FUNCTION_BLOCK "FB32_AXIS"   // FB32, LAD
{ S7_Optimized_Access := 'FALSE' }
AUTHOR : ETXETAR
VERSION : 1.0
// stored: AutoNumber false, IsIECCheckEnabled false, SetENOAutomatically false, UDAEnableTagReadback false
   VAR_INPUT
      OPTIONS_0 : Byte := 2#0000_0000;   // OPTIONS 0
      OPTIONS_1 : Byte := 2#0000_0000;   // OPTIONS 1
      SAFETY_BYPASS : Bool;   // MUST BE ALWAYS OFF, ACTIVATE ONLY FOR TEST
      OPTIMIZATION_BYPASS : Bool;   // MUST BE ALWAYS OFF, ACTIVATE ONLY FOR OPTIMIZATION TEST
      AX_ENABLE : Bool;   // AXIS ENABLE
      TEST_STOP_BRAKE_TEST_AX_NUM : Bool;   // TEST STOP BRAKE TEST AXIS NUMBER
      PARAMETER_SET_0 : Bool;   // PARAMETER SET [0] SELECTION
      PARAMETER_SET_1 : Bool;   // PARAMETER SET [1] SELECTION
      PARAMETER_SET_2 : Bool;   // PARAMETER SET [2] SELECTION
      PARAMETER_SET_3 : Bool;   // PARAMETER SET [3] SELECTION
      MOVE_AXIS : Bool;   // MOVE AXIS INPUT
      SAFE_ENABLED : Bool;   // SAFE ENABLED
      FEED_HOLD_COND : Bool;   // FEED HOLD CONDITIONS INPUT
      AX_TORQUE_ENABLE : Bool;   // AXIS TORQUE ENABLE
      MPP_AXIS_SELECTED : Bool;   // MPP AXIS SELECTED
      HMI_AXIS_SELECTED : Bool;   // HMI AXIS SELECTED
      HMI_REQ_LINE : Bool;   // HMI REQUEST LINE
      JOG_MINUS_REQ_NOT_FC18 : Bool;   // JOG MINUS REQUEST NOT FC18, THIS LINE MOVES THE AXIS WITHOUT FC18
      JOG_PLUS_REQ_NOT_FC18 : Bool;   // JOG PLUS REQUEST NOT FC18, THIS LINE MOVES THE AXIS WITHOUT FC18
      JOG_MINUS_REQ_FC18 : Bool;   // JOG MINUS REQUEST FOR FC18, THIS LINE MOVES THE AXIS WITH FC18
      JOG_PLUS_REQ_FC18 : Bool;   // JOG PLUS REQUEST FOR FC18, THIS LINE MOVES THE AXIS WITH FC18
      FC18_EXTERNAL_POS : Real;   // FC18 EXTERNAL POSITION
      AUTO_RETURN_COMMAND : Bool;   // AUTO RETURN COMMAND
      AUTO_ADVANCE_COMMAND : Bool;   // AUTO ADVANCE COMMAND
      DELETE_DISTANCE_TO_GO : Bool;   // DELETE DISTANCE TO GO CONDITIONS
      FEED_OVERRIDE : Byte;   // FEED OVERRIDE
      FEED_OVER_ACTIVE : Bool;   // FEED OVER ACTIVE
      READ_POS : DWord;   // READ POSITION
      UNIT_ALARM : UInt;   // UNIT NUMBER MIN. NUMBER=1 MAX. NUMBER=4
      STATION_ALARM : UInt;   // STATION NUMBER MIN. NUMBER=0 MAX. NUMBER=4
   END_VAR
   VAR_OUTPUT
      MOTOR_ACTIVE : Bool;   // MOTOR ACTIVE
      MOVE_AX : Bool;   // MOVE AXIS
      FEED_HOLD_CONDITIONS : Bool;   // FEED HOLD CONDITIONS
      ACTIVE_PARAMETER_SET : Byte;   // ACTIVE PARAMETER SET
      AX_NOT_REFERENCE_ALM : Bool;   // AXIS NOT REFERENCE / AXIS NOT REFERENCED ALARM
      AX_B_NOT_IN_PST_180_90_ALM : Bool;   // AXIS B NO IN POSITION 180º-90ª / AXIS B NOT IN PST 180 90 ALARM
      MAST_SLAVE_MODE_NOT_ACTIV_ALM : Bool;   // MASTER SLAVE MODE NOT ACTIVE ALARM
      AX_TORQUE_EXCEEDED_ALM : Bool;   // AXIS TORQUE EXCEEDED ALARM
      AXIS_POS : Real;   // AXIS POSITION
      HMI_MOTION_EXECUTABILITY_LEFT : Bool;   // HMI MOTION EXECUTABILITY LEFT
      HMI_MOTION_EXECUTABILITY_RIGHT : Bool;   // HMI MOTION EXECUTABILITY RIGHT
      HMI_MOTION_END_POS_LEFT : Bool;   // HMI MOTION END POSITION LEFT
      HMI_MOTION_END_POS_RIGHT : Bool;   // HMI MOTION END POSITION RIGHT
      HMI_MOTION_ACTIVE_LEFT : Bool;   // HMI MOTION ACTIVE LEFT
      HMI_MOTION_ACTIVE_RIGHT : Bool;   // HMI MOTION ACTIVE RIGHT
   END_VAR
   VAR_IN_OUT
      AxisDB : "LBP_typeAxisX";
   END_VAR
   VAR DB_SPECIFIC
      AXIS { S7_SetPoint := 'True'} : "AXIS";
      TIMER_PULSES_ENABLE { S7_SetPoint := 'True'} : TOF_TIME;
   END_VAR
   VAR
      SAFETY_POSITIONS { S7_SetPoint := 'True'} : "FB33_SAFETY_POSITIONS";
   END_VAR
   VAR_TEMP
      INPUTS_MASK : Byte;   // INPUT MASK
      O_BYTE_0 : Struct   // OPTIONS BYTE 0
         MEASURING_SYSTEM_2 : Bool;   // MEASURING SYSTEM 2 OPTION / ALWAYS ON OR ALWAYS OFF
         ENABLE_FC18 : Bool;   // ENABLE FC18 OPTION
         FC18_EXTERNAL_POSITION : Bool;   // FC18 EXTERNAL POSITION OPTION
         AXIS_B_ENABLE_FAULTS : Bool;   // AXIS B ENABLE FAULTS OPTION
         SPARE_4 : Bool;   // SPARE OPTION
         SPARE_5 : Bool;   // SPARE OPTION
         SPARE_6 : Bool;   // SPARE OPTION
         SPARE_7 : Bool;   // SPARE OPTION
      END_STRUCT;
      O_BYTE_1 : Struct   // OPTIONS BYTE 0
         AXIS_ROLLER : Bool;   // AXIS ROLLER OPTION / ALWAYS ON OR ALWAYS OFF
         MASTER_AXIS : Bool;   // MASTER AXIS OPTION
         SLAVE_AXIS : Bool;   // SLAVE AXIS OPTION
         MASTER_SLAVE_INDPNDNT_HT10 : Bool;   // MASTER SLAVE INDEPENDENT MOVEMENT HT10 OPTION
         GANTRY_MODE_MASTER_AXIS : Bool;   // GANTRY MODE MASTER AXIS OPTION
         SPARE_5 : Bool;   // SPARE OPTION
         SPARE_6 : Bool;   // SPARE OPTION
         SPARE_7 : Bool;   // SPARE OPTION
      END_STRUCT;
      FC18_STATE : Byte;   // FC 18 STATE
      DB_NUMBER : DInt;   // DB NUMBER FOR ALARMS AND HELP DECODING
      AXIS_NUMBER_FC18 : Int;   // AXIS NUMBER FC18
   END_VAR
   // TIMER_PULSES_ENABLE.PT := T#1s;
   VAR_TEMP   // added for the SCL form of the ladder/FBD networks
      _w1 : Bool;
      _w2 : Bool;
      _w3 : Bool;
      _w4 : Bool;
      _w5 : Bool;
      _w6 : Bool;
      _w7 : Bool;
      _w8 : Bool;
      _w9 : Bool;
      _w10 : Bool;
      _w11 : Bool;
      _w12 : Bool;
      _w13 : Bool;
      _w14 : Bool;
      _w15 : Bool;
   END_VAR
BEGIN

NETWORK
TITLE = READ INSTANCE DB
//READ DB NUMBER
      L     DINO;
      +     10#800000;
      T     #DB_NUMBER;
//READ AXIS NUMBER
      L     DINO;
      L     10#130;
      -I;
      T     #AXIS_NUMBER_FC18;


REGION Network 2: OPTIONS
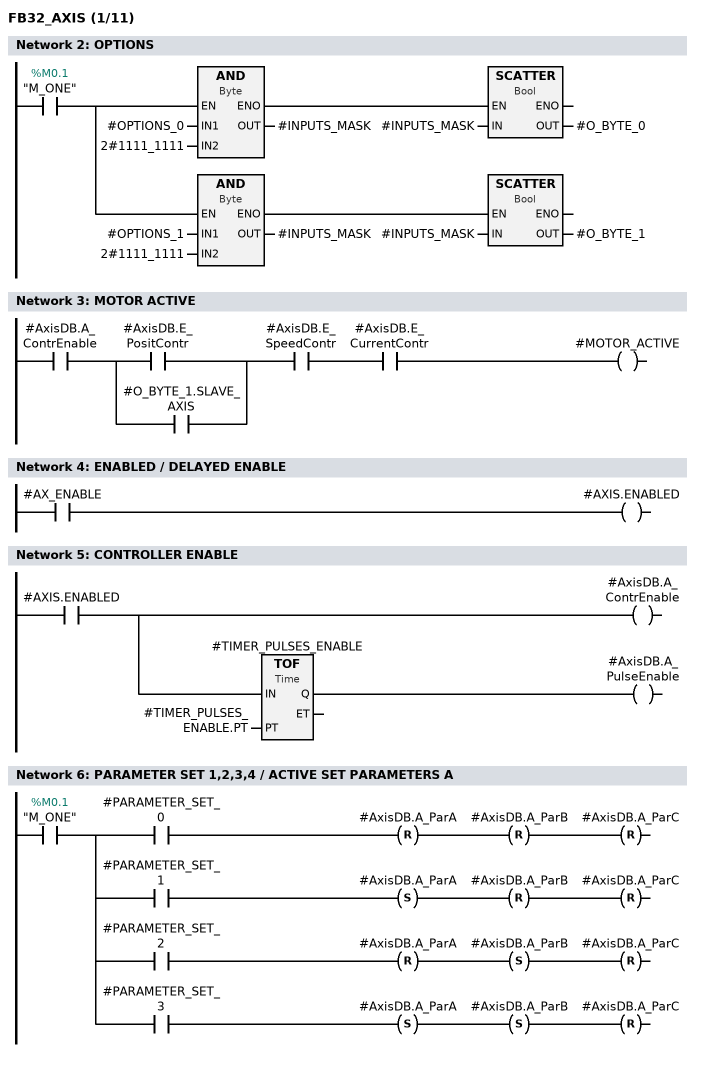
   RUNG wire#powerrail
      Contact( "M_ONE" )
      wire#w1
      { S7_Templates := "SrcType := Byte"; S7_GenerateENO := "TRUE" } And(in1 := #OPTIONS_0, in2 := 2#1111_1111, out => #INPUTS_MASK)
      { S7_Templates := "[dest_type := Bool, src_type := Byte]" } SCATTER(IN := #INPUTS_MASK, OUT => #O_BYTE_0)
   END_RUNG
   RUNG wire#w1
      { S7_Templates := "SrcType := Byte"; S7_GenerateENO := "TRUE" } And(in1 := #OPTIONS_1, in2 := 2#1111_1111, out => #INPUTS_MASK)
      { S7_Templates := "[dest_type := Bool, src_type := Byte]" } SCATTER(IN := #INPUTS_MASK, OUT => #O_BYTE_1)
   END_RUNG
   // the same network as SCL:
   IF "M_ONE" THEN #INPUTS_MASK := #OPTIONS_0 AND 2#1111_1111; END_IF;
   #_w1 := "M_ONE";
   IF #_w1 THEN
       SCATTER(IN := #INPUTS_MASK, OUT => #O_BYTE_0);
       #INPUTS_MASK := #OPTIONS_1 AND 2#1111_1111;
       SCATTER(IN := #INPUTS_MASK, OUT => #O_BYTE_1);
   END_IF;
END_REGION

REGION Network 3: MOTOR ACTIVE
   RUNG wire#powerrail
      Contact( #AxisDB.A_ContrEnable )
      wire#w1
      Contact( #AxisDB.E_PositContr )
      wire#w2
      Contact( #AxisDB.E_SpeedContr )
      Contact( #AxisDB.E_CurrentContr )
      Coil( #MOTOR_ACTIVE )
   END_RUNG
   RUNG wire#w1
      Contact( #O_BYTE_1.SLAVE_AXIS )
   END_RUNG wire#w2
   // the same network as SCL:
   #MOTOR_ACTIVE := #AxisDB.A_ContrEnable AND (#AxisDB.E_PositContr OR #O_BYTE_1.SLAVE_AXIS) AND #AxisDB.E_SpeedContr AND #AxisDB.E_CurrentContr;
END_REGION

REGION Network 4: ENABLED / DELAYED ENABLE
   RUNG wire#powerrail
      Contact( #AX_ENABLE )
      Coil( #AXIS.ENABLED )
   END_RUNG
   // the same network as SCL:
   #AXIS.ENABLED := #AX_ENABLE;
END_REGION

REGION Network 5: CONTROLLER ENABLE
   RUNG wire#powerrail
      Contact( #AXIS.ENABLED )
      wire#w1
      Coil( #AxisDB.A_ContrEnable )
   END_RUNG
   RUNG wire#w1
      { S7_Templates := "time_type := Time" } #TIMER_PULSES_ENABLE.TOF(pt := #TIMER_PULSES_ENABLE.PT, et =>)
      Coil( #AxisDB.A_PulseEnable )
   END_RUNG
   // the same network as SCL:
   #AxisDB.A_ContrEnable := #AXIS.ENABLED;
   #TIMER_PULSES_ENABLE(IN := #AXIS.ENABLED, PT := #TIMER_PULSES_ENABLE.PT);   // TOF
   #AxisDB.A_PulseEnable := #TIMER_PULSES_ENABLE.Q;
END_REGION

REGION Network 6: PARAMETER SET 1,2,3,4 / ACTIVE SET PARAMETERS A
   RUNG wire#powerrail
      Contact( "M_ONE" )
      wire#w1
      Contact( #PARAMETER_SET_0 )
      R_Coil( #AxisDB.A_ParA )
      R_Coil( #AxisDB.A_ParB )
      R_Coil( #AxisDB.A_ParC )
   END_RUNG
   RUNG wire#w1
      Contact( #PARAMETER_SET_1 )
      S_Coil( #AxisDB.A_ParA )
      R_Coil( #AxisDB.A_ParB )
      R_Coil( #AxisDB.A_ParC )
   END_RUNG
   RUNG wire#w1
      Contact( #PARAMETER_SET_2 )
      R_Coil( #AxisDB.A_ParA )
      S_Coil( #AxisDB.A_ParB )
      R_Coil( #AxisDB.A_ParC )
   END_RUNG
   RUNG wire#w1
      Contact( #PARAMETER_SET_3 )
      S_Coil( #AxisDB.A_ParA )
      S_Coil( #AxisDB.A_ParB )
      R_Coil( #AxisDB.A_ParC )
   END_RUNG
   // the same network as SCL:
   IF "M_ONE" AND #PARAMETER_SET_0 THEN
       #AxisDB.A_ParA := FALSE;
       #AxisDB.A_ParB := FALSE;
       #AxisDB.A_ParC := FALSE;
   END_IF;
   IF "M_ONE" AND #PARAMETER_SET_1 THEN
       #AxisDB.A_ParA := TRUE;
       #AxisDB.A_ParB := FALSE;
       #AxisDB.A_ParC := FALSE;
   END_IF;
   IF "M_ONE" AND #PARAMETER_SET_2 THEN
       #AxisDB.A_ParA := FALSE;
       #AxisDB.A_ParB := TRUE;
       #AxisDB.A_ParC := FALSE;
   END_IF;
   IF "M_ONE" AND #PARAMETER_SET_3 THEN
       #AxisDB.A_ParA := TRUE;
       #AxisDB.A_ParB := TRUE;
       #AxisDB.A_ParC := FALSE;
   END_IF;
END_REGION

REGION Network 7: ACTIVE PARAMETER SET 1,2,3,4
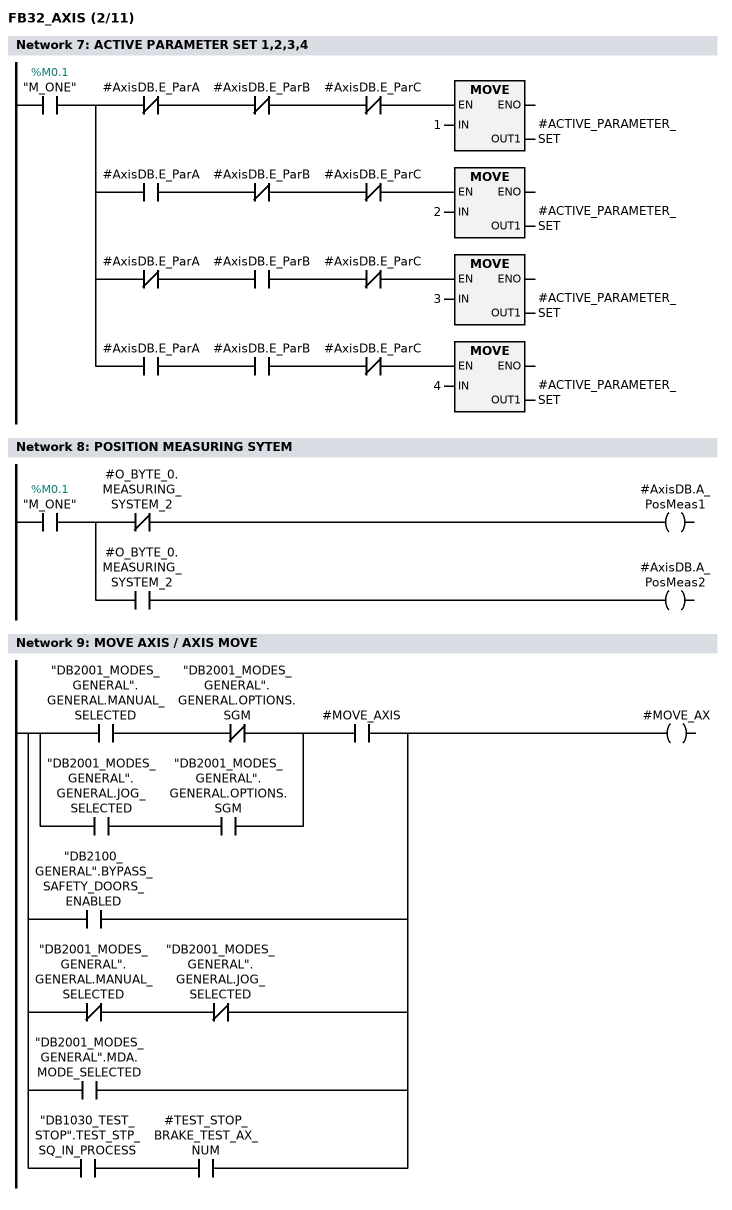
   RUNG wire#powerrail
      Contact( "M_ONE" )
      wire#w1
      I_Contact( #AxisDB.E_ParA )
      I_Contact( #AxisDB.E_ParB )
      I_Contact( #AxisDB.E_ParC )
      Move(in := 1, out1 => #ACTIVE_PARAMETER_SET)
   END_RUNG
   RUNG wire#w1
      Contact( #AxisDB.E_ParA )
      I_Contact( #AxisDB.E_ParB )
      I_Contact( #AxisDB.E_ParC )
      Move(in := 2, out1 => #ACTIVE_PARAMETER_SET)
   END_RUNG
   RUNG wire#w1
      I_Contact( #AxisDB.E_ParA )
      Contact( #AxisDB.E_ParB )
      I_Contact( #AxisDB.E_ParC )
      Move(in := 3, out1 => #ACTIVE_PARAMETER_SET)
   END_RUNG
   RUNG wire#w1
      Contact( #AxisDB.E_ParA )
      Contact( #AxisDB.E_ParB )
      I_Contact( #AxisDB.E_ParC )
      Move(in := 4, out1 => #ACTIVE_PARAMETER_SET)
   END_RUNG
   // the same network as SCL:
   IF "M_ONE" AND NOT #AxisDB.E_ParA AND NOT #AxisDB.E_ParB AND NOT #AxisDB.E_ParC THEN
       #ACTIVE_PARAMETER_SET := 1;
   END_IF;
   IF "M_ONE" AND #AxisDB.E_ParA AND NOT #AxisDB.E_ParB AND NOT #AxisDB.E_ParC THEN
       #ACTIVE_PARAMETER_SET := 2;
   END_IF;
   IF "M_ONE" AND NOT #AxisDB.E_ParA AND #AxisDB.E_ParB AND NOT #AxisDB.E_ParC THEN
       #ACTIVE_PARAMETER_SET := 3;
   END_IF;
   IF "M_ONE" AND #AxisDB.E_ParA AND #AxisDB.E_ParB AND NOT #AxisDB.E_ParC THEN
       #ACTIVE_PARAMETER_SET := 4;
   END_IF;
END_REGION

REGION Network 8: POSITION MEASURING SYTEM
   RUNG wire#powerrail
      Contact( "M_ONE" )
      wire#w1
      I_Contact( #O_BYTE_0.MEASURING_SYSTEM_2 )
      Coil( #AxisDB.A_PosMeas1 )
   END_RUNG
   RUNG wire#w1
      Contact( #O_BYTE_0.MEASURING_SYSTEM_2 )
      Coil( #AxisDB.A_PosMeas2 )
   END_RUNG
   // the same network as SCL:
   #AxisDB.A_PosMeas1 := "M_ONE" AND NOT #O_BYTE_0.MEASURING_SYSTEM_2;
   #AxisDB.A_PosMeas2 := "M_ONE" AND #O_BYTE_0.MEASURING_SYSTEM_2;
END_REGION

REGION Network 9: MOVE AXIS / AXIS MOVE
   RUNG wire#powerrail
      Contact( "DB2001_MODES_GENERAL".GENERAL.MANUAL_SELECTED )
      I_Contact( "DB2001_MODES_GENERAL".GENERAL.OPTIONS.SGM )
      wire#w1
      Contact( #MOVE_AXIS )
      wire#w2
      Coil( #MOVE_AX )
   END_RUNG
   RUNG wire#powerrail
      Contact( "DB2001_MODES_GENERAL".GENERAL.JOG_SELECTED )
      Contact( "DB2001_MODES_GENERAL".GENERAL.OPTIONS.SGM )
   END_RUNG wire#w1
   RUNG wire#powerrail
      Contact( "DB2100_GENERAL".BYPASS_SAFETY_DOORS_ENABLED )
   END_RUNG wire#w2
   RUNG wire#powerrail
      I_Contact( "DB2001_MODES_GENERAL".GENERAL.MANUAL_SELECTED )
      I_Contact( "DB2001_MODES_GENERAL".GENERAL.JOG_SELECTED )
   END_RUNG wire#w2
   RUNG wire#powerrail
      Contact( "DB2001_MODES_GENERAL".MDA.MODE_SELECTED )
   END_RUNG wire#w2
   RUNG wire#powerrail
      Contact( "DB1030_TEST_STOP".TEST_STP_SQ_IN_PROCESS )
      Contact( #TEST_STOP_BRAKE_TEST_AX_NUM )
   END_RUNG wire#w2
   // the same network as SCL:
   #MOVE_AX := ((("DB2001_MODES_GENERAL".GENERAL.MANUAL_SELECTED AND NOT "DB2001_MODES_GENERAL".GENERAL.OPTIONS.SGM) OR ("DB2001_MODES_GENERAL".GENERAL.JOG_SELECTED AND "DB2001_MODES_GENERAL".GENERAL.OPTIONS.SGM)) AND #MOVE_AXIS) OR "DB2100_GENERAL".BYPASS_SAFETY_DOORS_ENABLED OR (NOT "DB2001_MODES_GENERAL".GENERAL.MANUAL_SELECTED AND NOT "DB2001_MODES_GENERAL".GENERAL.JOG_SELECTED) OR "DB2001_MODES_GENERAL".MDA.MODE_SELECTED OR ("DB1030_TEST_STOP".TEST_STP_SQ_IN_PROCESS AND #TEST_STOP_BRAKE_TEST_AX_NUM);
END_REGION

REGION Network 10: FEED HOLD CONDITIONS
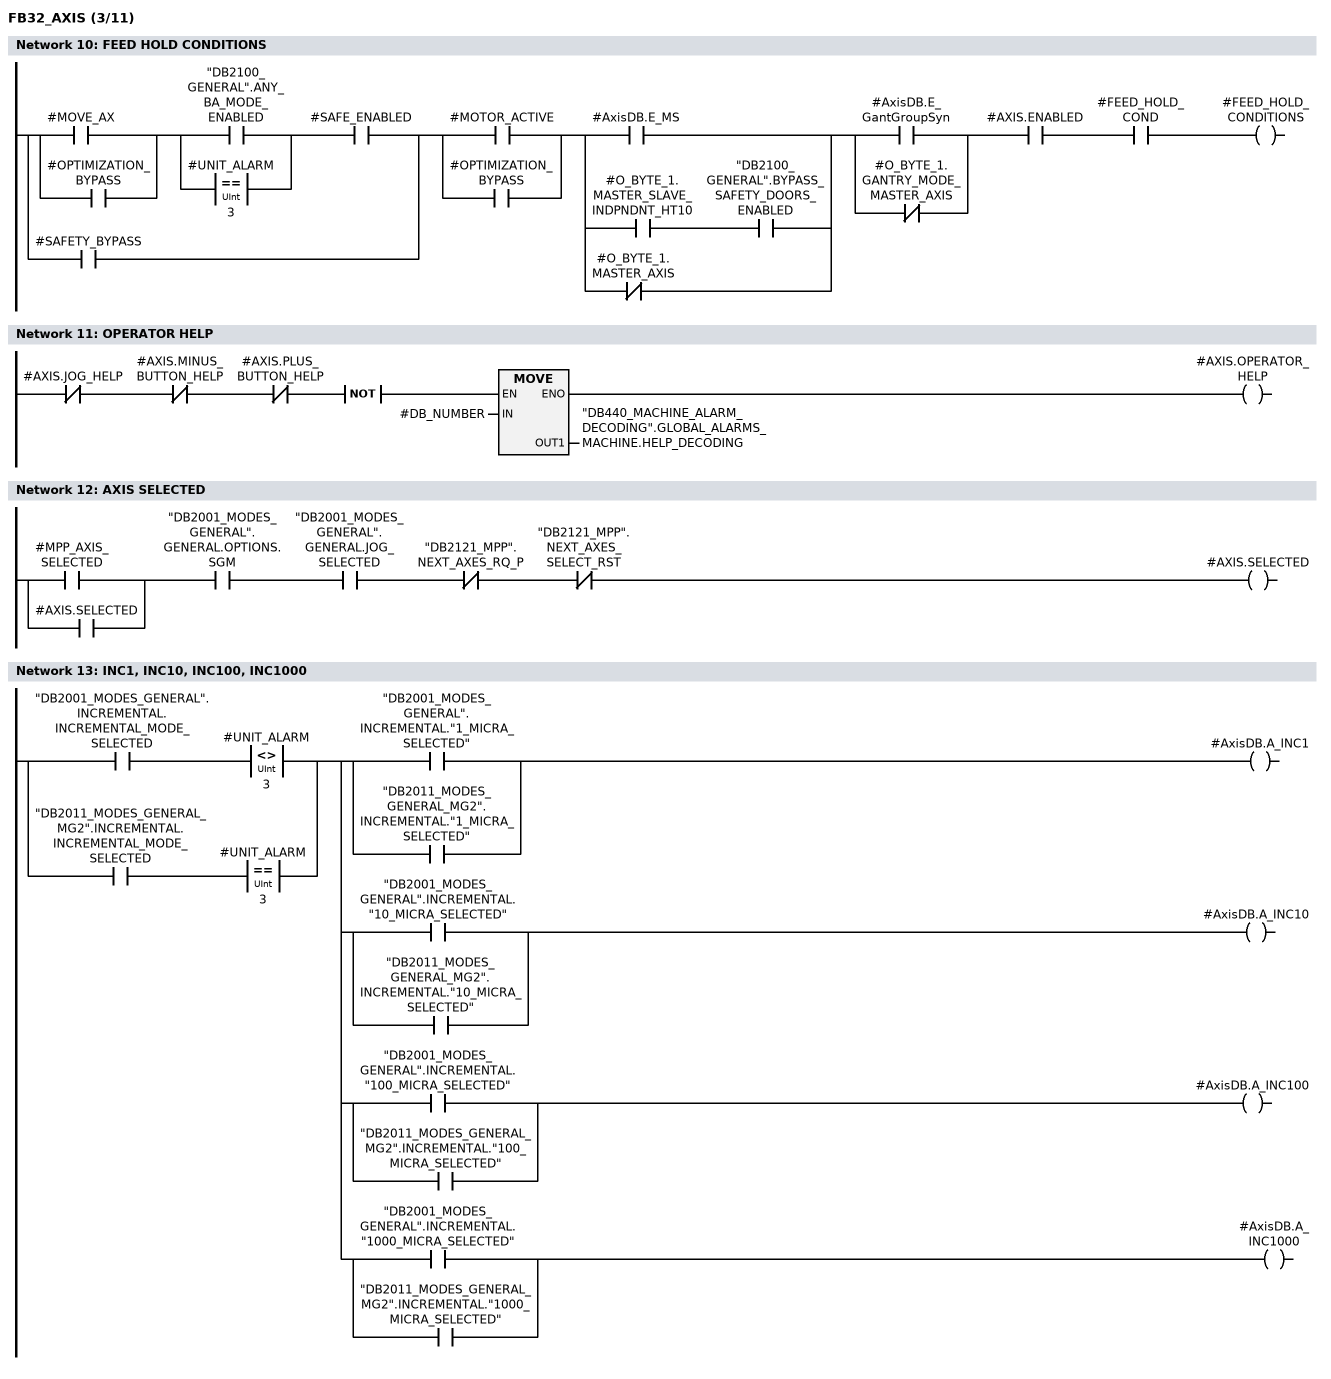
   RUNG wire#powerrail
      Contact( #MOVE_AX )
      wire#w1
      Contact( "DB2100_GENERAL".ANY_BA_MODE_ENABLED )
      wire#w2
      Contact( #SAFE_ENABLED )
      wire#w3
      Contact( #MOTOR_ACTIVE )
      wire#w4
      Contact( #AxisDB.E_MS )
      wire#w5
      Contact( #AxisDB.E_GantGroupSyn )
      wire#w6
      Contact( #AXIS.ENABLED )
      Contact( #FEED_HOLD_COND )
      Coil( #FEED_HOLD_CONDITIONS )
   END_RUNG
   RUNG wire#powerrail
      Contact( #OPTIMIZATION_BYPASS )
   END_RUNG wire#w1
   RUNG wire#w1
      { S7_Templates := "SrcType := UInt" } EQ_Contact(in1 := #UNIT_ALARM, in2 := 3)
   END_RUNG wire#w2
   RUNG wire#powerrail
      Contact( #SAFETY_BYPASS )
   END_RUNG wire#w3
   RUNG wire#w3
      Contact( #OPTIMIZATION_BYPASS )
   END_RUNG wire#w4
   RUNG wire#w4
      Contact( #O_BYTE_1.MASTER_SLAVE_INDPNDNT_HT10 )
      Contact( "DB2100_GENERAL".BYPASS_SAFETY_DOORS_ENABLED )
   END_RUNG wire#w5
   RUNG wire#w4
      I_Contact( #O_BYTE_1.MASTER_AXIS )
   END_RUNG wire#w5
   RUNG wire#w5
      I_Contact( #O_BYTE_1.GANTRY_MODE_MASTER_AXIS )
   END_RUNG wire#w6
   // the same network as SCL:
   #FEED_HOLD_CONDITIONS := (((#MOVE_AX OR #OPTIMIZATION_BYPASS) AND ("DB2100_GENERAL".ANY_BA_MODE_ENABLED OR (#UNIT_ALARM = 3)) AND #SAFE_ENABLED) OR #SAFETY_BYPASS) AND (#MOTOR_ACTIVE OR #OPTIMIZATION_BYPASS) AND (#AxisDB.E_MS OR (#O_BYTE_1.MASTER_SLAVE_INDPNDNT_HT10 AND "DB2100_GENERAL".BYPASS_SAFETY_DOORS_ENABLED) OR NOT #O_BYTE_1.MASTER_AXIS) AND (#AxisDB.E_GantGroupSyn OR NOT #O_BYTE_1.GANTRY_MODE_MASTER_AXIS) AND #AXIS.ENABLED AND #FEED_HOLD_COND;
END_REGION

REGION Network 11: OPERATOR HELP
   RUNG wire#powerrail
      I_Contact( #AXIS.JOG_HELP )
      I_Contact( #AXIS.MINUS_BUTTON_HELP )
      I_Contact( #AXIS.PLUS_BUTTON_HELP )
      Not()
      { S7_GenerateENO := "TRUE" } Move(in := #DB_NUMBER, out1 => "DB440_MACHINE_ALARM_DECODING".GLOBAL_ALARMS_MACHINE.HELP_DECODING)
      Coil( #AXIS.OPERATOR_HELP )
   END_RUNG
   // the same network as SCL:
   // ENO of a box is taken as its EN; it also drops when the box reports an error
   #_w1 := NOT (NOT #AXIS.JOG_HELP AND NOT #AXIS.MINUS_BUTTON_HELP AND NOT #AXIS.PLUS_BUTTON_HELP);
   IF #_w1 THEN "DB440_MACHINE_ALARM_DECODING".GLOBAL_ALARMS_MACHINE.HELP_DECODING := #DB_NUMBER; END_IF;
   #AXIS.OPERATOR_HELP := #_w1;
END_REGION

REGION Network 12: AXIS SELECTED
   RUNG wire#powerrail
      Contact( #MPP_AXIS_SELECTED )
      wire#w1
      Contact( "DB2001_MODES_GENERAL".GENERAL.OPTIONS.SGM )
      Contact( "DB2001_MODES_GENERAL".GENERAL.JOG_SELECTED )
      I_Contact( "DB2121_MPP".NEXT_AXES_RQ_P )
      I_Contact( "DB2121_MPP".NEXT_AXES_SELECT_RST )
      Coil( #AXIS.SELECTED )
   END_RUNG
   RUNG wire#powerrail
      Contact( #AXIS.SELECTED )
   END_RUNG wire#w1
   // the same network as SCL:
   #AXIS.SELECTED := (#MPP_AXIS_SELECTED OR #AXIS.SELECTED) AND "DB2001_MODES_GENERAL".GENERAL.OPTIONS.SGM AND "DB2001_MODES_GENERAL".GENERAL.JOG_SELECTED AND NOT "DB2121_MPP".NEXT_AXES_RQ_P AND NOT "DB2121_MPP".NEXT_AXES_SELECT_RST;
END_REGION

REGION Network 13: INC1, INC10, INC100, INC1000
   RUNG wire#powerrail
      Contact( "DB2001_MODES_GENERAL".INCREMENTAL.INCREMENTAL_MODE_SELECTED )
      { S7_Templates := "SrcType := UInt" } NE_Contact(in1 := #UNIT_ALARM, in2 := 3)
      wire#w1
      Contact( "DB2001_MODES_GENERAL".INCREMENTAL."1_MICRA_SELECTED" )
      wire#w2
      Coil( #AxisDB.A_INC1 )
   END_RUNG
   RUNG wire#powerrail
      Contact( "DB2011_MODES_GENERAL_MG2".INCREMENTAL.INCREMENTAL_MODE_SELECTED )
      { S7_Templates := "SrcType := UInt" } EQ_Contact(in1 := #UNIT_ALARM, in2 := 3)
   END_RUNG wire#w1
   RUNG wire#w1
      Contact( "DB2011_MODES_GENERAL_MG2".INCREMENTAL."1_MICRA_SELECTED" )
   END_RUNG wire#w2
   RUNG wire#w1
      Contact( "DB2001_MODES_GENERAL".INCREMENTAL."10_MICRA_SELECTED" )
      wire#w3
      Coil( #AxisDB.A_INC10 )
   END_RUNG
   RUNG wire#w1
      Contact( "DB2011_MODES_GENERAL_MG2".INCREMENTAL."10_MICRA_SELECTED" )
   END_RUNG wire#w3
   RUNG wire#w1
      Contact( "DB2001_MODES_GENERAL".INCREMENTAL."100_MICRA_SELECTED" )
      wire#w4
      Coil( #AxisDB.A_INC100 )
   END_RUNG
   RUNG wire#w1
      Contact( "DB2011_MODES_GENERAL_MG2".INCREMENTAL."100_MICRA_SELECTED" )
   END_RUNG wire#w4
   RUNG wire#w1
      Contact( "DB2001_MODES_GENERAL".INCREMENTAL."1000_MICRA_SELECTED" )
      wire#w5
      Coil( #AxisDB.A_INC1000 )
   END_RUNG
   RUNG wire#w1
      Contact( "DB2011_MODES_GENERAL_MG2".INCREMENTAL."1000_MICRA_SELECTED" )
   END_RUNG wire#w5
   // the same network as SCL:
   #_w1 := ("DB2001_MODES_GENERAL".INCREMENTAL.INCREMENTAL_MODE_SELECTED AND (#UNIT_ALARM <> 3)) OR ("DB2011_MODES_GENERAL_MG2".INCREMENTAL.INCREMENTAL_MODE_SELECTED AND (#UNIT_ALARM = 3));
   #AxisDB.A_INC1 := #_w1 AND ("DB2001_MODES_GENERAL".INCREMENTAL."1_MICRA_SELECTED" OR "DB2011_MODES_GENERAL_MG2".INCREMENTAL."1_MICRA_SELECTED");
   #AxisDB.A_INC10 := #_w1 AND ("DB2001_MODES_GENERAL".INCREMENTAL."10_MICRA_SELECTED" OR "DB2011_MODES_GENERAL_MG2".INCREMENTAL."10_MICRA_SELECTED");
   #AxisDB.A_INC100 := #_w1 AND ("DB2001_MODES_GENERAL".INCREMENTAL."100_MICRA_SELECTED" OR "DB2011_MODES_GENERAL_MG2".INCREMENTAL."100_MICRA_SELECTED");
   #AxisDB.A_INC1000 := #_w1 AND ("DB2001_MODES_GENERAL".INCREMENTAL."1000_MICRA_SELECTED" OR "DB2011_MODES_GENERAL_MG2".INCREMENTAL."1000_MICRA_SELECTED");
END_REGION

REGION Network 14: ACTIVATE HANDWHEEL / ACTIVATE HANDWHEEL 1
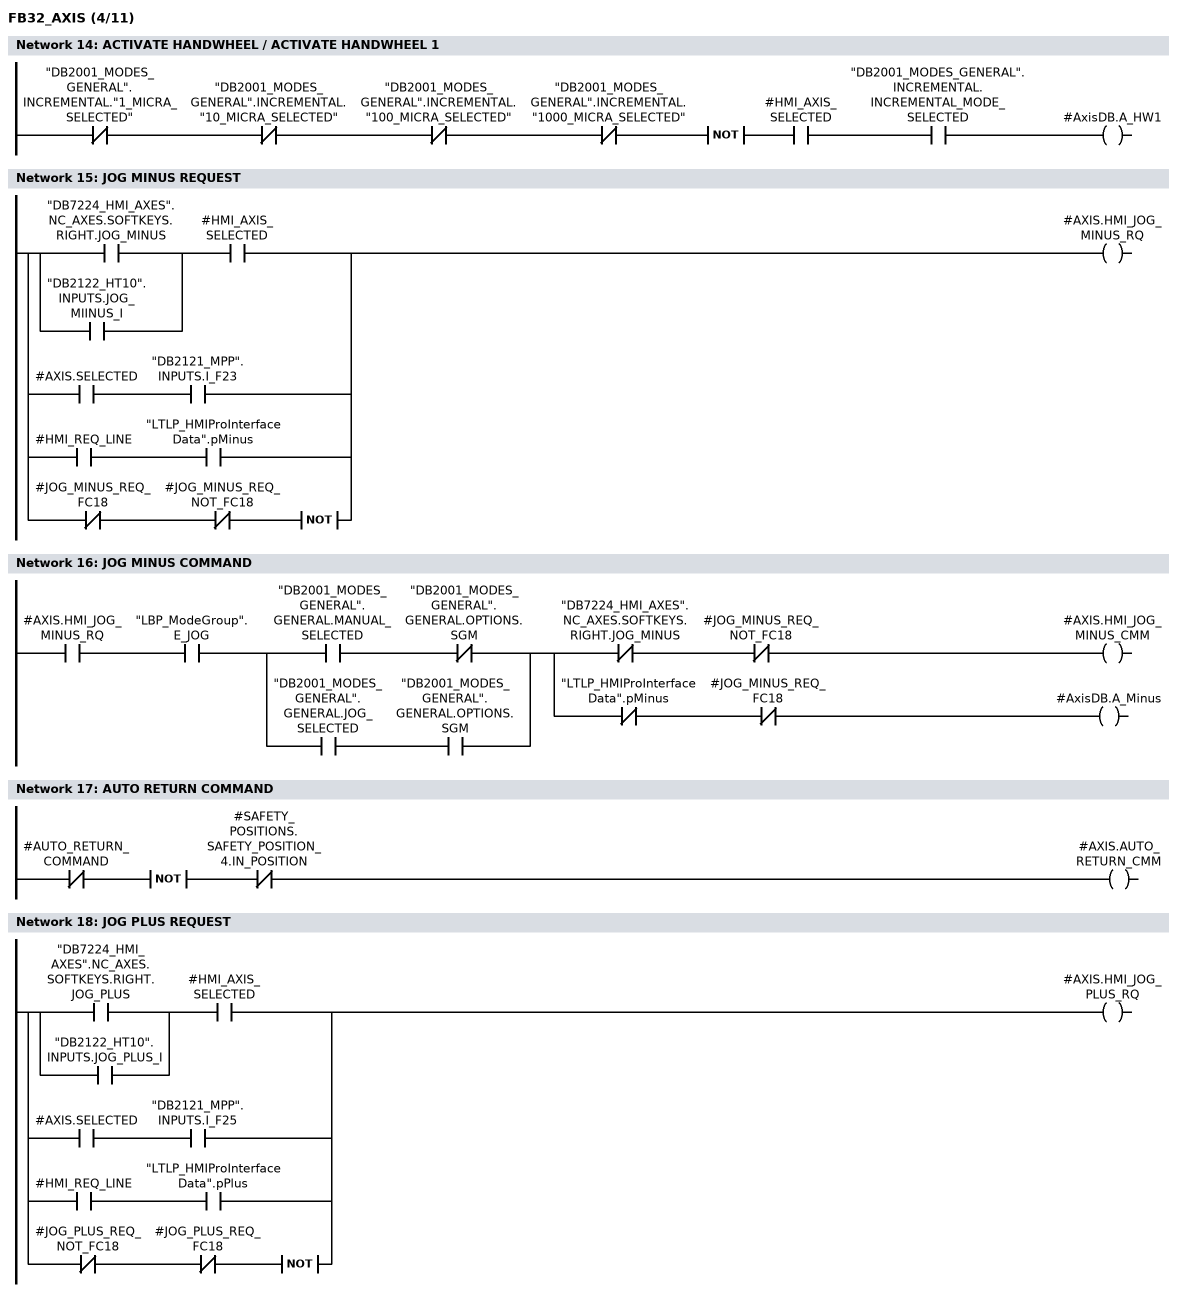
   RUNG wire#powerrail
      I_Contact( "DB2001_MODES_GENERAL".INCREMENTAL."1_MICRA_SELECTED" )
      I_Contact( "DB2001_MODES_GENERAL".INCREMENTAL."10_MICRA_SELECTED" )
      I_Contact( "DB2001_MODES_GENERAL".INCREMENTAL."100_MICRA_SELECTED" )
      I_Contact( "DB2001_MODES_GENERAL".INCREMENTAL."1000_MICRA_SELECTED" )
      Not()
      Contact( #HMI_AXIS_SELECTED )
      Contact( "DB2001_MODES_GENERAL".INCREMENTAL.INCREMENTAL_MODE_SELECTED )
      Coil( #AxisDB.A_HW1 )
   END_RUNG
   // the same network as SCL:
   #AxisDB.A_HW1 := NOT (NOT "DB2001_MODES_GENERAL".INCREMENTAL."1_MICRA_SELECTED" AND NOT "DB2001_MODES_GENERAL".INCREMENTAL."10_MICRA_SELECTED" AND NOT "DB2001_MODES_GENERAL".INCREMENTAL."100_MICRA_SELECTED" AND NOT "DB2001_MODES_GENERAL".INCREMENTAL."1000_MICRA_SELECTED") AND #HMI_AXIS_SELECTED AND "DB2001_MODES_GENERAL".INCREMENTAL.INCREMENTAL_MODE_SELECTED;
END_REGION

REGION Network 15: JOG MINUS REQUEST
   RUNG wire#powerrail
      Contact( "DB7224_HMI_AXES".NC_AXES.SOFTKEYS.RIGHT.JOG_MINUS )
      wire#w1
      Contact( #HMI_AXIS_SELECTED )
      wire#w2
      Coil( #AXIS.HMI_JOG_MINUS_RQ )
   END_RUNG
   RUNG wire#powerrail
      Contact( "DB2122_HT10".INPUTS.JOG_MIINUS_I )
   END_RUNG wire#w1
   RUNG wire#powerrail
      Contact( #AXIS.SELECTED )
      Contact( "DB2121_MPP".INPUTS.I_F23 )
   END_RUNG wire#w2
   RUNG wire#powerrail
      Contact( #HMI_REQ_LINE )
      Contact( "LTLP_HMIProInterfaceData".pMinus )
   END_RUNG wire#w2
   RUNG wire#powerrail
      I_Contact( #JOG_MINUS_REQ_FC18 )
      I_Contact( #JOG_MINUS_REQ_NOT_FC18 )
      Not()
   END_RUNG wire#w2
   // the same network as SCL:
   #AXIS.HMI_JOG_MINUS_RQ := (("DB7224_HMI_AXES".NC_AXES.SOFTKEYS.RIGHT.JOG_MINUS OR "DB2122_HT10".INPUTS.JOG_MIINUS_I) AND #HMI_AXIS_SELECTED) OR (#AXIS.SELECTED AND "DB2121_MPP".INPUTS.I_F23) OR (#HMI_REQ_LINE AND "LTLP_HMIProInterfaceData".pMinus) OR NOT (NOT #JOG_MINUS_REQ_FC18 AND NOT #JOG_MINUS_REQ_NOT_FC18);
END_REGION

REGION Network 16: JOG MINUS COMMAND
   RUNG wire#powerrail
      Contact( #AXIS.HMI_JOG_MINUS_RQ )
      Contact( "LBP_ModeGroup".E_JOG )
      wire#w1
      Contact( "DB2001_MODES_GENERAL".GENERAL.MANUAL_SELECTED )
      I_Contact( "DB2001_MODES_GENERAL".GENERAL.OPTIONS.SGM )
      wire#w2
      I_Contact( "DB7224_HMI_AXES".NC_AXES.SOFTKEYS.RIGHT.JOG_MINUS )
      I_Contact( #JOG_MINUS_REQ_NOT_FC18 )
      Coil( #AXIS.HMI_JOG_MINUS_CMM )
   END_RUNG
   RUNG wire#w1
      Contact( "DB2001_MODES_GENERAL".GENERAL.JOG_SELECTED )
      Contact( "DB2001_MODES_GENERAL".GENERAL.OPTIONS.SGM )
   END_RUNG wire#w2
   RUNG wire#w2
      I_Contact( "LTLP_HMIProInterfaceData".pMinus )
      I_Contact( #JOG_MINUS_REQ_FC18 )
      Coil( #AxisDB.A_Minus )
   END_RUNG
   // the same network as SCL:
   #_w1 := #AXIS.HMI_JOG_MINUS_RQ AND "LBP_ModeGroup".E_JOG AND (("DB2001_MODES_GENERAL".GENERAL.MANUAL_SELECTED AND NOT "DB2001_MODES_GENERAL".GENERAL.OPTIONS.SGM) OR ("DB2001_MODES_GENERAL".GENERAL.JOG_SELECTED AND "DB2001_MODES_GENERAL".GENERAL.OPTIONS.SGM));
   #AXIS.HMI_JOG_MINUS_CMM := #_w1 AND NOT "DB7224_HMI_AXES".NC_AXES.SOFTKEYS.RIGHT.JOG_MINUS AND NOT #JOG_MINUS_REQ_NOT_FC18;
   #AxisDB.A_Minus := #_w1 AND NOT "LTLP_HMIProInterfaceData".pMinus AND NOT #JOG_MINUS_REQ_FC18;
END_REGION

REGION Network 17: AUTO RETURN COMMAND
   RUNG wire#powerrail
      I_Contact( #AUTO_RETURN_COMMAND )
      Not()
      I_Contact( #SAFETY_POSITIONS.SAFETY_POSITION_4.IN_POSITION )
      Coil( #AXIS.AUTO_RETURN_CMM )
   END_RUNG
   // the same network as SCL:
   #AXIS.AUTO_RETURN_CMM := NOT (NOT #AUTO_RETURN_COMMAND) AND NOT #SAFETY_POSITIONS.SAFETY_POSITION_4.IN_POSITION;
END_REGION

REGION Network 18: JOG PLUS REQUEST
   RUNG wire#powerrail
      Contact( "DB7224_HMI_AXES".NC_AXES.SOFTKEYS.RIGHT.JOG_PLUS )
      wire#w1
      Contact( #HMI_AXIS_SELECTED )
      wire#w2
      Coil( #AXIS.HMI_JOG_PLUS_RQ )
   END_RUNG
   RUNG wire#powerrail
      Contact( "DB2122_HT10".INPUTS.JOG_PLUS_I )
   END_RUNG wire#w1
   RUNG wire#powerrail
      Contact( #AXIS.SELECTED )
      Contact( "DB2121_MPP".INPUTS.I_F25 )
   END_RUNG wire#w2
   RUNG wire#powerrail
      Contact( #HMI_REQ_LINE )
      Contact( "LTLP_HMIProInterfaceData".pPlus )
   END_RUNG wire#w2
   RUNG wire#powerrail
      I_Contact( #JOG_PLUS_REQ_NOT_FC18 )
      I_Contact( #JOG_PLUS_REQ_FC18 )
      Not()
   END_RUNG wire#w2
   // the same network as SCL:
   #AXIS.HMI_JOG_PLUS_RQ := (("DB7224_HMI_AXES".NC_AXES.SOFTKEYS.RIGHT.JOG_PLUS OR "DB2122_HT10".INPUTS.JOG_PLUS_I) AND #HMI_AXIS_SELECTED) OR (#AXIS.SELECTED AND "DB2121_MPP".INPUTS.I_F25) OR (#HMI_REQ_LINE AND "LTLP_HMIProInterfaceData".pPlus) OR NOT (NOT #JOG_PLUS_REQ_NOT_FC18 AND NOT #JOG_PLUS_REQ_FC18);
END_REGION

REGION Network 19: JOG PLUS COMMAND
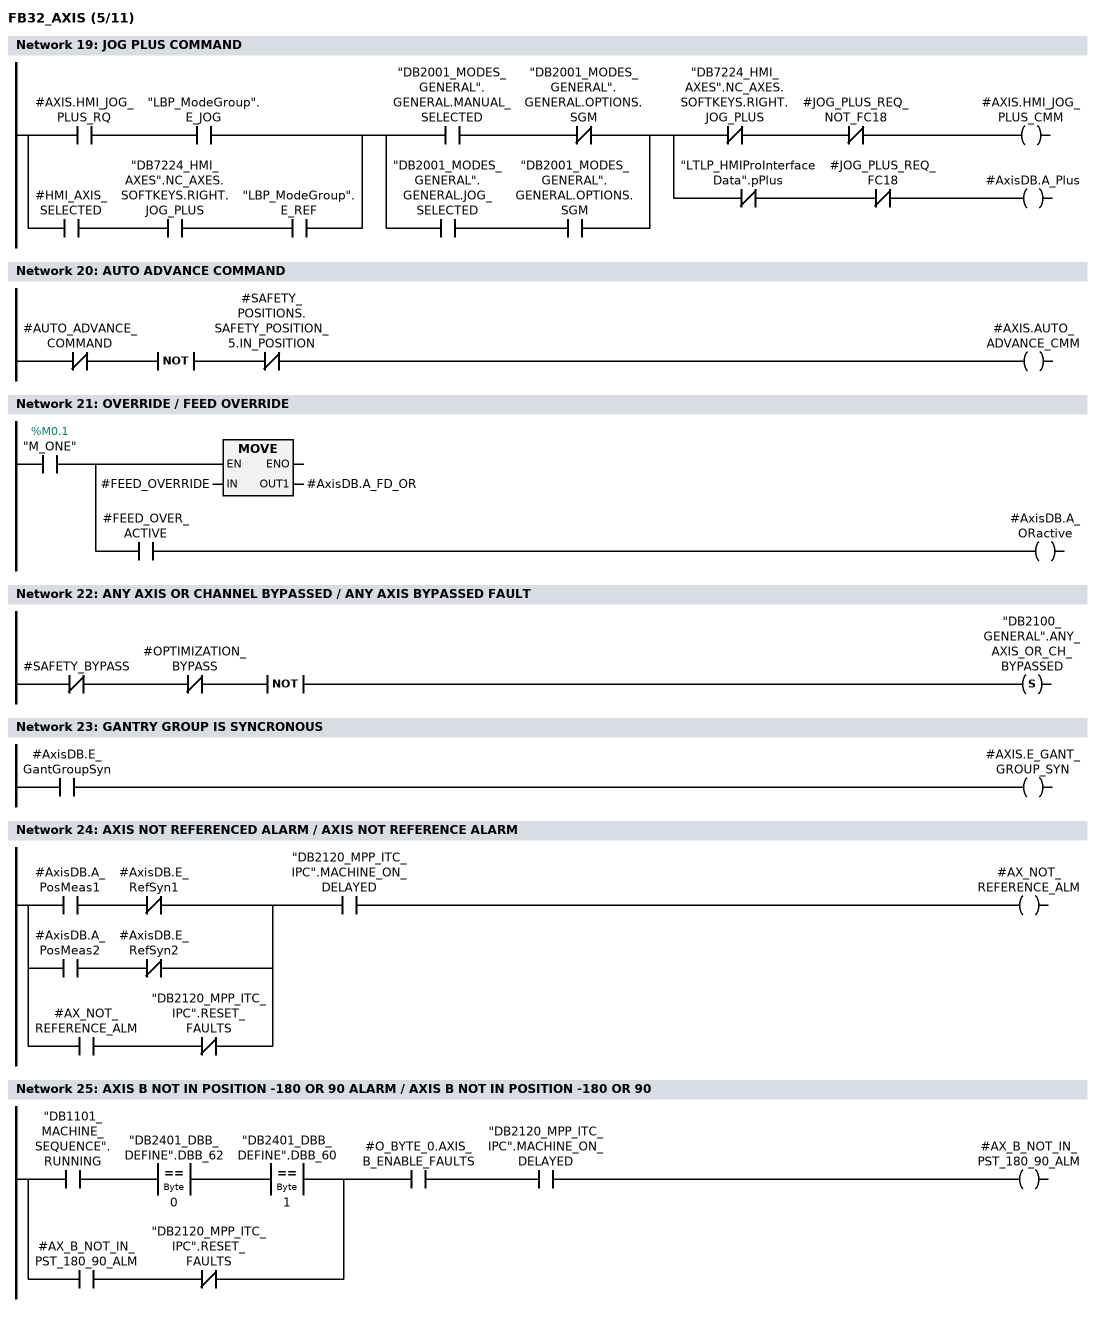
   RUNG wire#powerrail
      Contact( #AXIS.HMI_JOG_PLUS_RQ )
      Contact( "LBP_ModeGroup".E_JOG )
      wire#w1
      Contact( "DB2001_MODES_GENERAL".GENERAL.MANUAL_SELECTED )
      I_Contact( "DB2001_MODES_GENERAL".GENERAL.OPTIONS.SGM )
      wire#w2
      I_Contact( "DB7224_HMI_AXES".NC_AXES.SOFTKEYS.RIGHT.JOG_PLUS )
      I_Contact( #JOG_PLUS_REQ_NOT_FC18 )
      Coil( #AXIS.HMI_JOG_PLUS_CMM )
   END_RUNG
   RUNG wire#powerrail
      Contact( #HMI_AXIS_SELECTED )
      Contact( "DB7224_HMI_AXES".NC_AXES.SOFTKEYS.RIGHT.JOG_PLUS )
      Contact( "LBP_ModeGroup".E_REF )
   END_RUNG wire#w1
   RUNG wire#w1
      Contact( "DB2001_MODES_GENERAL".GENERAL.JOG_SELECTED )
      Contact( "DB2001_MODES_GENERAL".GENERAL.OPTIONS.SGM )
   END_RUNG wire#w2
   RUNG wire#w2
      I_Contact( "LTLP_HMIProInterfaceData".pPlus )
      I_Contact( #JOG_PLUS_REQ_FC18 )
      Coil( #AxisDB.A_Plus )
   END_RUNG
   // the same network as SCL:
   #_w1 := ((#AXIS.HMI_JOG_PLUS_RQ AND "LBP_ModeGroup".E_JOG) OR (#HMI_AXIS_SELECTED AND "DB7224_HMI_AXES".NC_AXES.SOFTKEYS.RIGHT.JOG_PLUS AND "LBP_ModeGroup".E_REF)) AND (("DB2001_MODES_GENERAL".GENERAL.MANUAL_SELECTED AND NOT "DB2001_MODES_GENERAL".GENERAL.OPTIONS.SGM) OR ("DB2001_MODES_GENERAL".GENERAL.JOG_SELECTED AND "DB2001_MODES_GENERAL".GENERAL.OPTIONS.SGM));
   #AXIS.HMI_JOG_PLUS_CMM := #_w1 AND NOT "DB7224_HMI_AXES".NC_AXES.SOFTKEYS.RIGHT.JOG_PLUS AND NOT #JOG_PLUS_REQ_NOT_FC18;
   #AxisDB.A_Plus := #_w1 AND NOT "LTLP_HMIProInterfaceData".pPlus AND NOT #JOG_PLUS_REQ_FC18;
END_REGION

REGION Network 20: AUTO ADVANCE COMMAND
   RUNG wire#powerrail
      I_Contact( #AUTO_ADVANCE_COMMAND )
      Not()
      I_Contact( #SAFETY_POSITIONS.SAFETY_POSITION_5.IN_POSITION )
      Coil( #AXIS.AUTO_ADVANCE_CMM )
   END_RUNG
   // the same network as SCL:
   #AXIS.AUTO_ADVANCE_CMM := NOT (NOT #AUTO_ADVANCE_COMMAND) AND NOT #SAFETY_POSITIONS.SAFETY_POSITION_5.IN_POSITION;
END_REGION

REGION Network 21: OVERRIDE / FEED OVERRIDE
   RUNG wire#powerrail
      Contact( "M_ONE" )
      wire#w1
      { S7_GenerateENO := "TRUE" } Move(in := #FEED_OVERRIDE, out1 => #AxisDB.A_FD_OR)
   END_RUNG
   RUNG wire#w1
      Contact( #FEED_OVER_ACTIVE )
      Coil( #AxisDB.A_ORactive )
   END_RUNG
   // the same network as SCL:
   IF "M_ONE" THEN #AxisDB.A_FD_OR := #FEED_OVERRIDE; END_IF;
   #AxisDB.A_ORactive := "M_ONE" AND #FEED_OVER_ACTIVE;
END_REGION

REGION Network 22: ANY AXIS OR CHANNEL BYPASSED / ANY AXIS BYPASSED FAULT
   RUNG wire#powerrail
      I_Contact( #SAFETY_BYPASS )
      I_Contact( #OPTIMIZATION_BYPASS )
      Not()
      S_Coil( "DB2100_GENERAL".ANY_AXIS_OR_CH_BYPASSED )
   END_RUNG
   // the same network as SCL:
   IF NOT (NOT #SAFETY_BYPASS AND NOT #OPTIMIZATION_BYPASS) THEN
       "DB2100_GENERAL".ANY_AXIS_OR_CH_BYPASSED := TRUE;
   END_IF;
END_REGION

REGION Network 23: GANTRY GROUP IS SYNCRONOUS
   RUNG wire#powerrail
      Contact( #AxisDB.E_GantGroupSyn )
      Coil( #AXIS.E_GANT_GROUP_SYN )
   END_RUNG
   // the same network as SCL:
   #AXIS.E_GANT_GROUP_SYN := #AxisDB.E_GantGroupSyn;
END_REGION

REGION Network 24: AXIS NOT REFERENCED ALARM / AXIS NOT REFERENCE ALARM
   RUNG wire#powerrail
      Contact( #AxisDB.A_PosMeas1 )
      I_Contact( #AxisDB.E_RefSyn1 )
      wire#w1
      Contact( "DB2120_MPP_ITC_IPC".MACHINE_ON_DELAYED )
      Coil( #AX_NOT_REFERENCE_ALM )
   END_RUNG
   RUNG wire#powerrail
      Contact( #AxisDB.A_PosMeas2 )
      I_Contact( #AxisDB.E_RefSyn2 )
   END_RUNG wire#w1
   RUNG wire#powerrail
      Contact( #AX_NOT_REFERENCE_ALM )
      I_Contact( "DB2120_MPP_ITC_IPC".RESET_FAULTS )
   END_RUNG wire#w1
   // the same network as SCL:
   #AX_NOT_REFERENCE_ALM := ((#AxisDB.A_PosMeas1 AND NOT #AxisDB.E_RefSyn1) OR (#AxisDB.A_PosMeas2 AND NOT #AxisDB.E_RefSyn2) OR (#AX_NOT_REFERENCE_ALM AND NOT "DB2120_MPP_ITC_IPC".RESET_FAULTS)) AND "DB2120_MPP_ITC_IPC".MACHINE_ON_DELAYED;
END_REGION

REGION Network 25: AXIS B NOT IN POSITION -180 OR 90 ALARM / AXIS B NOT IN POSITION -180 OR 90
   RUNG wire#powerrail
      Contact( "DB1101_MACHINE_SEQUENCE".RUNNING )
      { S7_Templates := "SrcType := Byte" } EQ_Contact(in1 := "DB2401_DBB_DEFINE".DBB_62, in2 := 0)
      { S7_Templates := "SrcType := Byte" } EQ_Contact(in1 := "DB2401_DBB_DEFINE".DBB_60, in2 := 1)
      wire#w1
      Contact( #O_BYTE_0.AXIS_B_ENABLE_FAULTS )
      Contact( "DB2120_MPP_ITC_IPC".MACHINE_ON_DELAYED )
      Coil( #AX_B_NOT_IN_PST_180_90_ALM )
   END_RUNG
   RUNG wire#powerrail
      Contact( #AX_B_NOT_IN_PST_180_90_ALM )
      I_Contact( "DB2120_MPP_ITC_IPC".RESET_FAULTS )
   END_RUNG wire#w1
   // the same network as SCL:
   #AX_B_NOT_IN_PST_180_90_ALM := (("DB1101_MACHINE_SEQUENCE".RUNNING AND ("DB2401_DBB_DEFINE".DBB_62 = 0) AND ("DB2401_DBB_DEFINE".DBB_60 = 1)) OR (#AX_B_NOT_IN_PST_180_90_ALM AND NOT "DB2120_MPP_ITC_IPC".RESET_FAULTS)) AND #O_BYTE_0.AXIS_B_ENABLE_FAULTS AND "DB2120_MPP_ITC_IPC".MACHINE_ON_DELAYED;
END_REGION

REGION Network 26: MASTER SLAVE MODE NOT ACTIVE ALARM / AXIS NOT REFERENCE ALARM
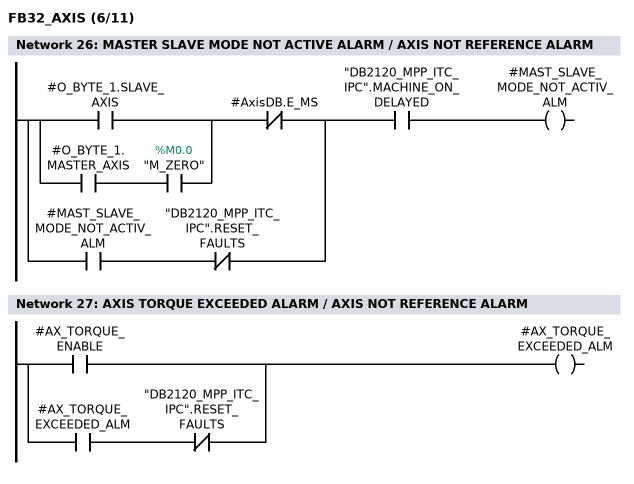
   RUNG wire#powerrail
      Contact( #O_BYTE_1.SLAVE_AXIS )
      wire#w1
      I_Contact( #AxisDB.E_MS )
      wire#w2
      Contact( "DB2120_MPP_ITC_IPC".MACHINE_ON_DELAYED )
      Coil( #MAST_SLAVE_MODE_NOT_ACTIV_ALM )
   END_RUNG
   RUNG wire#powerrail
      Contact( #O_BYTE_1.MASTER_AXIS )
      Contact( "M_ZERO" )
   END_RUNG wire#w1
   RUNG wire#powerrail
      Contact( #MAST_SLAVE_MODE_NOT_ACTIV_ALM )
      I_Contact( "DB2120_MPP_ITC_IPC".RESET_FAULTS )
   END_RUNG wire#w2
   // the same network as SCL:
   #MAST_SLAVE_MODE_NOT_ACTIV_ALM := (((#O_BYTE_1.SLAVE_AXIS OR (#O_BYTE_1.MASTER_AXIS AND "M_ZERO")) AND NOT #AxisDB.E_MS) OR (#MAST_SLAVE_MODE_NOT_ACTIV_ALM AND NOT "DB2120_MPP_ITC_IPC".RESET_FAULTS)) AND "DB2120_MPP_ITC_IPC".MACHINE_ON_DELAYED;
END_REGION

REGION Network 27: AXIS TORQUE EXCEEDED ALARM / AXIS NOT REFERENCE ALARM
   RUNG wire#powerrail
      Contact( #AX_TORQUE_ENABLE )
      wire#w1
      Coil( #AX_TORQUE_EXCEEDED_ALM )
   END_RUNG
   RUNG wire#powerrail
      Contact( #AX_TORQUE_EXCEEDED_ALM )
      I_Contact( "DB2120_MPP_ITC_IPC".RESET_FAULTS )
   END_RUNG wire#w1
   // the same network as SCL:
   #AX_TORQUE_EXCEEDED_ALM := #AX_TORQUE_ENABLE OR (#AX_TORQUE_EXCEEDED_ALM AND NOT "DB2120_MPP_ITC_IPC".RESET_FAULTS);
END_REGION

REGION Network 28: IMMEDIATE STOP AND STOP END OF CYCLE ALARMS / IMMEDIATE STOP & STOP END OF CYCLE ALARMS
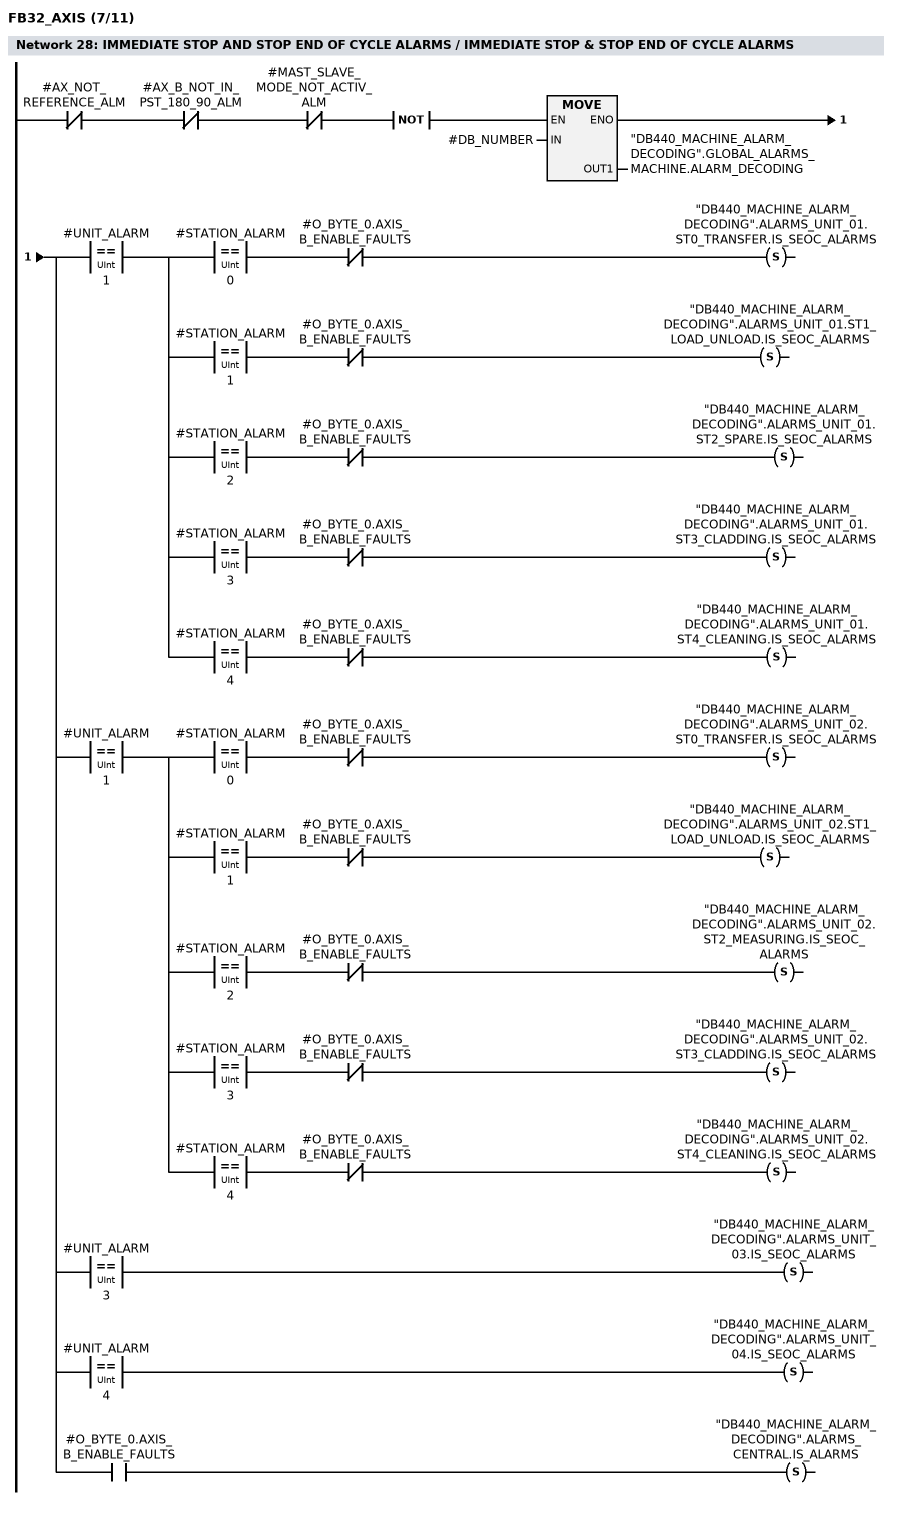
   RUNG wire#powerrail
      I_Contact( #AX_NOT_REFERENCE_ALM )
      I_Contact( #AX_B_NOT_IN_PST_180_90_ALM )
      I_Contact( #MAST_SLAVE_MODE_NOT_ACTIV_ALM )
      Not()
      { S7_GenerateENO := "TRUE" } Move(in := #DB_NUMBER, out1 => "DB440_MACHINE_ALARM_DECODING".GLOBAL_ALARMS_MACHINE.ALARM_DECODING)
      wire#w1
      { S7_Templates := "SrcType := UInt" } EQ_Contact(in1 := #UNIT_ALARM, in2 := 1)
      wire#w2
      { S7_Templates := "SrcType := UInt" } EQ_Contact(in1 := #STATION_ALARM, in2 := 0)
      I_Contact( #O_BYTE_0.AXIS_B_ENABLE_FAULTS )
      S_Coil( "DB440_MACHINE_ALARM_DECODING".ALARMS_UNIT_01.ST0_TRANSFER.IS_SEOC_ALARMS )
   END_RUNG
   RUNG wire#w2
      { S7_Templates := "SrcType := UInt" } EQ_Contact(in1 := #STATION_ALARM, in2 := 1)
      I_Contact( #O_BYTE_0.AXIS_B_ENABLE_FAULTS )
      S_Coil( "DB440_MACHINE_ALARM_DECODING".ALARMS_UNIT_01.ST1_LOAD_UNLOAD.IS_SEOC_ALARMS )
   END_RUNG
   RUNG wire#w2
      { S7_Templates := "SrcType := UInt" } EQ_Contact(in1 := #STATION_ALARM, in2 := 2)
      I_Contact( #O_BYTE_0.AXIS_B_ENABLE_FAULTS )
      S_Coil( "DB440_MACHINE_ALARM_DECODING".ALARMS_UNIT_01.ST2_SPARE.IS_SEOC_ALARMS )
   END_RUNG
   RUNG wire#w2
      { S7_Templates := "SrcType := UInt" } EQ_Contact(in1 := #STATION_ALARM, in2 := 3)
      I_Contact( #O_BYTE_0.AXIS_B_ENABLE_FAULTS )
      S_Coil( "DB440_MACHINE_ALARM_DECODING".ALARMS_UNIT_01.ST3_CLADDING.IS_SEOC_ALARMS )
   END_RUNG
   RUNG wire#w2
      { S7_Templates := "SrcType := UInt" } EQ_Contact(in1 := #STATION_ALARM, in2 := 4)
      I_Contact( #O_BYTE_0.AXIS_B_ENABLE_FAULTS )
      S_Coil( "DB440_MACHINE_ALARM_DECODING".ALARMS_UNIT_01.ST4_CLEANING.IS_SEOC_ALARMS )
   END_RUNG
   RUNG wire#w1
      { S7_Templates := "SrcType := UInt" } EQ_Contact(in1 := #UNIT_ALARM, in2 := 1)
      wire#w3
      { S7_Templates := "SrcType := UInt" } EQ_Contact(in1 := #STATION_ALARM, in2 := 0)
      I_Contact( #O_BYTE_0.AXIS_B_ENABLE_FAULTS )
      S_Coil( "DB440_MACHINE_ALARM_DECODING".ALARMS_UNIT_02.ST0_TRANSFER.IS_SEOC_ALARMS )
   END_RUNG
   RUNG wire#w3
      { S7_Templates := "SrcType := UInt" } EQ_Contact(in1 := #STATION_ALARM, in2 := 1)
      I_Contact( #O_BYTE_0.AXIS_B_ENABLE_FAULTS )
      S_Coil( "DB440_MACHINE_ALARM_DECODING".ALARMS_UNIT_02.ST1_LOAD_UNLOAD.IS_SEOC_ALARMS )
   END_RUNG
   RUNG wire#w3
      { S7_Templates := "SrcType := UInt" } EQ_Contact(in1 := #STATION_ALARM, in2 := 2)
      I_Contact( #O_BYTE_0.AXIS_B_ENABLE_FAULTS )
      S_Coil( "DB440_MACHINE_ALARM_DECODING".ALARMS_UNIT_02.ST2_MEASURING.IS_SEOC_ALARMS )
   END_RUNG
   RUNG wire#w3
      { S7_Templates := "SrcType := UInt" } EQ_Contact(in1 := #STATION_ALARM, in2 := 3)
      I_Contact( #O_BYTE_0.AXIS_B_ENABLE_FAULTS )
      S_Coil( "DB440_MACHINE_ALARM_DECODING".ALARMS_UNIT_02.ST3_CLADDING.IS_SEOC_ALARMS )
   END_RUNG
   RUNG wire#w3
      { S7_Templates := "SrcType := UInt" } EQ_Contact(in1 := #STATION_ALARM, in2 := 4)
      I_Contact( #O_BYTE_0.AXIS_B_ENABLE_FAULTS )
      S_Coil( "DB440_MACHINE_ALARM_DECODING".ALARMS_UNIT_02.ST4_CLEANING.IS_SEOC_ALARMS )
   END_RUNG
   RUNG wire#w1
      { S7_Templates := "SrcType := UInt" } EQ_Contact(in1 := #UNIT_ALARM, in2 := 3)
      S_Coil( "DB440_MACHINE_ALARM_DECODING".ALARMS_UNIT_03.IS_SEOC_ALARMS )
   END_RUNG
   RUNG wire#w1
      { S7_Templates := "SrcType := UInt" } EQ_Contact(in1 := #UNIT_ALARM, in2 := 4)
      S_Coil( "DB440_MACHINE_ALARM_DECODING".ALARMS_UNIT_04.IS_SEOC_ALARMS )
   END_RUNG
   RUNG wire#w1
      Contact( #O_BYTE_0.AXIS_B_ENABLE_FAULTS )
      S_Coil( "DB440_MACHINE_ALARM_DECODING".ALARMS_CENTRAL.IS_ALARMS )
   END_RUNG
   // the same network as SCL:
   // ENO of a box is taken as its EN; it also drops when the box reports an error
   #_w1 := NOT (NOT #AX_NOT_REFERENCE_ALM AND NOT #AX_B_NOT_IN_PST_180_90_ALM AND NOT #MAST_SLAVE_MODE_NOT_ACTIV_ALM);
   IF #_w1 THEN "DB440_MACHINE_ALARM_DECODING".GLOBAL_ALARMS_MACHINE.ALARM_DECODING := #DB_NUMBER; END_IF;
   #_w2 := #_w1 AND (#UNIT_ALARM = 1);
   IF #_w2 AND (#STATION_ALARM = 0) AND NOT #O_BYTE_0.AXIS_B_ENABLE_FAULTS THEN
       "DB440_MACHINE_ALARM_DECODING".ALARMS_UNIT_01.ST0_TRANSFER.IS_SEOC_ALARMS := TRUE;
   END_IF;
   IF #_w2 AND (#STATION_ALARM = 1) AND NOT #O_BYTE_0.AXIS_B_ENABLE_FAULTS THEN
       "DB440_MACHINE_ALARM_DECODING".ALARMS_UNIT_01.ST1_LOAD_UNLOAD.IS_SEOC_ALARMS := TRUE;
   END_IF;
   IF #_w2 AND (#STATION_ALARM = 2) AND NOT #O_BYTE_0.AXIS_B_ENABLE_FAULTS THEN
       "DB440_MACHINE_ALARM_DECODING".ALARMS_UNIT_01.ST2_SPARE.IS_SEOC_ALARMS := TRUE;
   END_IF;
   IF #_w2 AND (#STATION_ALARM = 3) AND NOT #O_BYTE_0.AXIS_B_ENABLE_FAULTS THEN
       "DB440_MACHINE_ALARM_DECODING".ALARMS_UNIT_01.ST3_CLADDING.IS_SEOC_ALARMS := TRUE;
   END_IF;
   IF #_w2 AND (#STATION_ALARM = 4) AND NOT #O_BYTE_0.AXIS_B_ENABLE_FAULTS THEN
       "DB440_MACHINE_ALARM_DECODING".ALARMS_UNIT_01.ST4_CLEANING.IS_SEOC_ALARMS := TRUE;
   END_IF;
   #_w3 := #_w1 AND (#UNIT_ALARM = 1);
   IF #_w3 AND (#STATION_ALARM = 0) AND NOT #O_BYTE_0.AXIS_B_ENABLE_FAULTS THEN
       "DB440_MACHINE_ALARM_DECODING".ALARMS_UNIT_02.ST0_TRANSFER.IS_SEOC_ALARMS := TRUE;
   END_IF;
   IF #_w3 AND (#STATION_ALARM = 1) AND NOT #O_BYTE_0.AXIS_B_ENABLE_FAULTS THEN
       "DB440_MACHINE_ALARM_DECODING".ALARMS_UNIT_02.ST1_LOAD_UNLOAD.IS_SEOC_ALARMS := TRUE;
   END_IF;
   IF #_w3 AND (#STATION_ALARM = 2) AND NOT #O_BYTE_0.AXIS_B_ENABLE_FAULTS THEN
       "DB440_MACHINE_ALARM_DECODING".ALARMS_UNIT_02.ST2_MEASURING.IS_SEOC_ALARMS := TRUE;
   END_IF;
   IF #_w3 AND (#STATION_ALARM = 3) AND NOT #O_BYTE_0.AXIS_B_ENABLE_FAULTS THEN
       "DB440_MACHINE_ALARM_DECODING".ALARMS_UNIT_02.ST3_CLADDING.IS_SEOC_ALARMS := TRUE;
   END_IF;
   IF #_w3 AND (#STATION_ALARM = 4) AND NOT #O_BYTE_0.AXIS_B_ENABLE_FAULTS THEN
       "DB440_MACHINE_ALARM_DECODING".ALARMS_UNIT_02.ST4_CLEANING.IS_SEOC_ALARMS := TRUE;
   END_IF;
   IF #_w1 AND (#UNIT_ALARM = 3) THEN
       "DB440_MACHINE_ALARM_DECODING".ALARMS_UNIT_03.IS_SEOC_ALARMS := TRUE;
   END_IF;
   IF #_w1 AND (#UNIT_ALARM = 4) THEN
       "DB440_MACHINE_ALARM_DECODING".ALARMS_UNIT_04.IS_SEOC_ALARMS := TRUE;
   END_IF;
   IF #_w1 AND #O_BYTE_0.AXIS_B_ENABLE_FAULTS THEN
       "DB440_MACHINE_ALARM_DECODING".ALARMS_CENTRAL.IS_ALARMS := TRUE;
   END_IF;
END_REGION

REGION Network 29: RETURN HOME POSITION AND STOP END OF CYCLE ALARMS
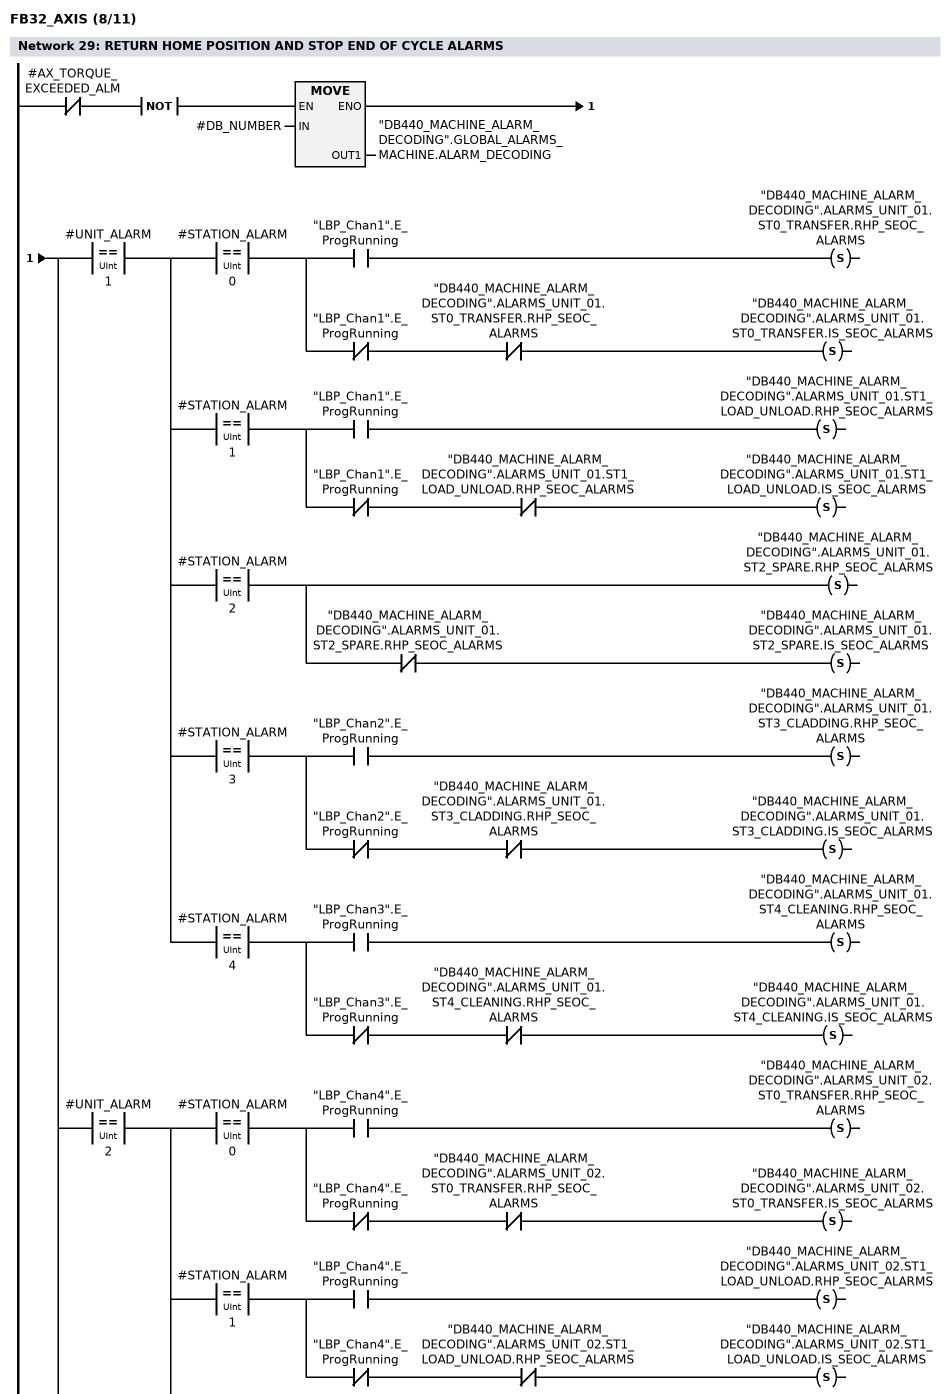
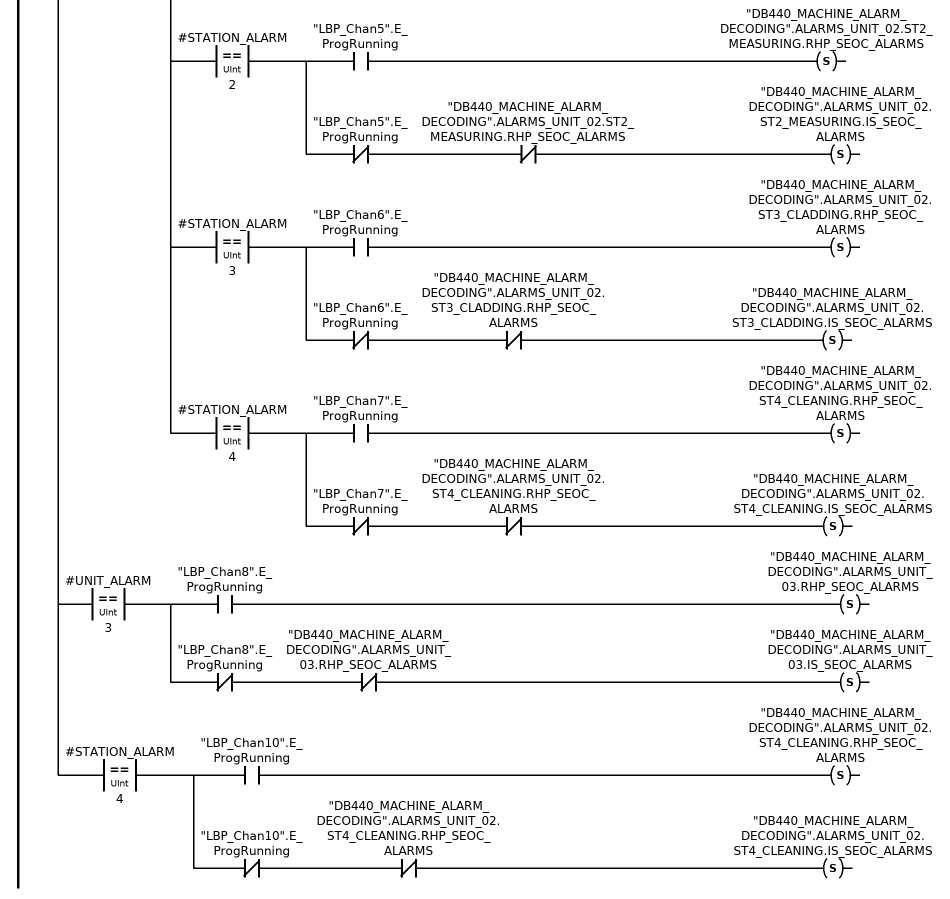
   RUNG wire#powerrail
      I_Contact( #AX_TORQUE_EXCEEDED_ALM )
      Not()
      { S7_GenerateENO := "TRUE" } Move(in := #DB_NUMBER, out1 => "DB440_MACHINE_ALARM_DECODING".GLOBAL_ALARMS_MACHINE.ALARM_DECODING)
      wire#w1
      { S7_Templates := "SrcType := UInt" } EQ_Contact(in1 := #UNIT_ALARM, in2 := 1)
      wire#w2
      { S7_Templates := "SrcType := UInt" } EQ_Contact(in1 := #STATION_ALARM, in2 := 0)
      wire#w3
      Contact( "LBP_Chan1".E_ProgRunning )
      S_Coil( "DB440_MACHINE_ALARM_DECODING".ALARMS_UNIT_01.ST0_TRANSFER.RHP_SEOC_ALARMS )
   END_RUNG
   RUNG wire#w3
      I_Contact( "LBP_Chan1".E_ProgRunning )
      I_Contact( "DB440_MACHINE_ALARM_DECODING".ALARMS_UNIT_01.ST0_TRANSFER.RHP_SEOC_ALARMS )
      S_Coil( "DB440_MACHINE_ALARM_DECODING".ALARMS_UNIT_01.ST0_TRANSFER.IS_SEOC_ALARMS )
   END_RUNG
   RUNG wire#w2
      { S7_Templates := "SrcType := UInt" } EQ_Contact(in1 := #STATION_ALARM, in2 := 1)
      wire#w4
      Contact( "LBP_Chan1".E_ProgRunning )
      S_Coil( "DB440_MACHINE_ALARM_DECODING".ALARMS_UNIT_01.ST1_LOAD_UNLOAD.RHP_SEOC_ALARMS )
   END_RUNG
   RUNG wire#w4
      I_Contact( "LBP_Chan1".E_ProgRunning )
      I_Contact( "DB440_MACHINE_ALARM_DECODING".ALARMS_UNIT_01.ST1_LOAD_UNLOAD.RHP_SEOC_ALARMS )
      S_Coil( "DB440_MACHINE_ALARM_DECODING".ALARMS_UNIT_01.ST1_LOAD_UNLOAD.IS_SEOC_ALARMS )
   END_RUNG
   RUNG wire#w2
      { S7_Templates := "SrcType := UInt" } EQ_Contact(in1 := #STATION_ALARM, in2 := 2)
      wire#w5
      S_Coil( "DB440_MACHINE_ALARM_DECODING".ALARMS_UNIT_01.ST2_SPARE.RHP_SEOC_ALARMS )
   END_RUNG
   RUNG wire#w5
      I_Contact( "DB440_MACHINE_ALARM_DECODING".ALARMS_UNIT_01.ST2_SPARE.RHP_SEOC_ALARMS )
      S_Coil( "DB440_MACHINE_ALARM_DECODING".ALARMS_UNIT_01.ST2_SPARE.IS_SEOC_ALARMS )
   END_RUNG
   RUNG wire#w2
      { S7_Templates := "SrcType := UInt" } EQ_Contact(in1 := #STATION_ALARM, in2 := 3)
      wire#w6
      Contact( "LBP_Chan2".E_ProgRunning )
      S_Coil( "DB440_MACHINE_ALARM_DECODING".ALARMS_UNIT_01.ST3_CLADDING.RHP_SEOC_ALARMS )
   END_RUNG
   RUNG wire#w6
      I_Contact( "LBP_Chan2".E_ProgRunning )
      I_Contact( "DB440_MACHINE_ALARM_DECODING".ALARMS_UNIT_01.ST3_CLADDING.RHP_SEOC_ALARMS )
      S_Coil( "DB440_MACHINE_ALARM_DECODING".ALARMS_UNIT_01.ST3_CLADDING.IS_SEOC_ALARMS )
   END_RUNG
   RUNG wire#w2
      { S7_Templates := "SrcType := UInt" } EQ_Contact(in1 := #STATION_ALARM, in2 := 4)
      wire#w7
      Contact( "LBP_Chan3".E_ProgRunning )
      S_Coil( "DB440_MACHINE_ALARM_DECODING".ALARMS_UNIT_01.ST4_CLEANING.RHP_SEOC_ALARMS )
   END_RUNG
   RUNG wire#w7
      I_Contact( "LBP_Chan3".E_ProgRunning )
      I_Contact( "DB440_MACHINE_ALARM_DECODING".ALARMS_UNIT_01.ST4_CLEANING.RHP_SEOC_ALARMS )
      S_Coil( "DB440_MACHINE_ALARM_DECODING".ALARMS_UNIT_01.ST4_CLEANING.IS_SEOC_ALARMS )
   END_RUNG
   RUNG wire#w1
      { S7_Templates := "SrcType := UInt" } EQ_Contact(in1 := #UNIT_ALARM, in2 := 2)
      wire#w8
      { S7_Templates := "SrcType := UInt" } EQ_Contact(in1 := #STATION_ALARM, in2 := 0)
      wire#w9
      Contact( "LBP_Chan4".E_ProgRunning )
      S_Coil( "DB440_MACHINE_ALARM_DECODING".ALARMS_UNIT_02.ST0_TRANSFER.RHP_SEOC_ALARMS )
   END_RUNG
   RUNG wire#w9
      I_Contact( "LBP_Chan4".E_ProgRunning )
      I_Contact( "DB440_MACHINE_ALARM_DECODING".ALARMS_UNIT_02.ST0_TRANSFER.RHP_SEOC_ALARMS )
      S_Coil( "DB440_MACHINE_ALARM_DECODING".ALARMS_UNIT_02.ST0_TRANSFER.IS_SEOC_ALARMS )
   END_RUNG
   RUNG wire#w8
      { S7_Templates := "SrcType := UInt" } EQ_Contact(in1 := #STATION_ALARM, in2 := 1)
      wire#w10
      Contact( "LBP_Chan4".E_ProgRunning )
      S_Coil( "DB440_MACHINE_ALARM_DECODING".ALARMS_UNIT_02.ST1_LOAD_UNLOAD.RHP_SEOC_ALARMS )
   END_RUNG
   RUNG wire#w10
      I_Contact( "LBP_Chan4".E_ProgRunning )
      I_Contact( "DB440_MACHINE_ALARM_DECODING".ALARMS_UNIT_02.ST1_LOAD_UNLOAD.RHP_SEOC_ALARMS )
      S_Coil( "DB440_MACHINE_ALARM_DECODING".ALARMS_UNIT_02.ST1_LOAD_UNLOAD.IS_SEOC_ALARMS )
   END_RUNG
   RUNG wire#w8
      { S7_Templates := "SrcType := UInt" } EQ_Contact(in1 := #STATION_ALARM, in2 := 2)
      wire#w11
      Contact( "LBP_Chan5".E_ProgRunning )
      S_Coil( "DB440_MACHINE_ALARM_DECODING".ALARMS_UNIT_02.ST2_MEASURING.RHP_SEOC_ALARMS )
   END_RUNG
   RUNG wire#w11
      I_Contact( "LBP_Chan5".E_ProgRunning )
      I_Contact( "DB440_MACHINE_ALARM_DECODING".ALARMS_UNIT_02.ST2_MEASURING.RHP_SEOC_ALARMS )
      S_Coil( "DB440_MACHINE_ALARM_DECODING".ALARMS_UNIT_02.ST2_MEASURING.IS_SEOC_ALARMS )
   END_RUNG
   RUNG wire#w8
      { S7_Templates := "SrcType := UInt" } EQ_Contact(in1 := #STATION_ALARM, in2 := 3)
      wire#w12
      Contact( "LBP_Chan6".E_ProgRunning )
      S_Coil( "DB440_MACHINE_ALARM_DECODING".ALARMS_UNIT_02.ST3_CLADDING.RHP_SEOC_ALARMS )
   END_RUNG
   RUNG wire#w12
      I_Contact( "LBP_Chan6".E_ProgRunning )
      I_Contact( "DB440_MACHINE_ALARM_DECODING".ALARMS_UNIT_02.ST3_CLADDING.RHP_SEOC_ALARMS )
      S_Coil( "DB440_MACHINE_ALARM_DECODING".ALARMS_UNIT_02.ST3_CLADDING.IS_SEOC_ALARMS )
   END_RUNG
   RUNG wire#w8
      { S7_Templates := "SrcType := UInt" } EQ_Contact(in1 := #STATION_ALARM, in2 := 4)
      wire#w13
      Contact( "LBP_Chan7".E_ProgRunning )
      S_Coil( "DB440_MACHINE_ALARM_DECODING".ALARMS_UNIT_02.ST4_CLEANING.RHP_SEOC_ALARMS )
   END_RUNG
   RUNG wire#w13
      I_Contact( "LBP_Chan7".E_ProgRunning )
      I_Contact( "DB440_MACHINE_ALARM_DECODING".ALARMS_UNIT_02.ST4_CLEANING.RHP_SEOC_ALARMS )
      S_Coil( "DB440_MACHINE_ALARM_DECODING".ALARMS_UNIT_02.ST4_CLEANING.IS_SEOC_ALARMS )
   END_RUNG
   RUNG wire#w1
      { S7_Templates := "SrcType := UInt" } EQ_Contact(in1 := #UNIT_ALARM, in2 := 3)
      wire#w14
      Contact( "LBP_Chan8".E_ProgRunning )
      S_Coil( "DB440_MACHINE_ALARM_DECODING".ALARMS_UNIT_03.RHP_SEOC_ALARMS )
   END_RUNG
   RUNG wire#w14
      I_Contact( "LBP_Chan8".E_ProgRunning )
      I_Contact( "DB440_MACHINE_ALARM_DECODING".ALARMS_UNIT_03.RHP_SEOC_ALARMS )
      S_Coil( "DB440_MACHINE_ALARM_DECODING".ALARMS_UNIT_03.IS_SEOC_ALARMS )
   END_RUNG
   RUNG wire#w1
      { S7_Templates := "SrcType := UInt" } EQ_Contact(in1 := #STATION_ALARM, in2 := 4)
      wire#w15
      Contact( "LBP_Chan10".E_ProgRunning )
      S_Coil( "DB440_MACHINE_ALARM_DECODING".ALARMS_UNIT_02.ST4_CLEANING.RHP_SEOC_ALARMS )
   END_RUNG
   RUNG wire#w15
      I_Contact( "LBP_Chan10".E_ProgRunning )
      I_Contact( "DB440_MACHINE_ALARM_DECODING".ALARMS_UNIT_02.ST4_CLEANING.RHP_SEOC_ALARMS )
      S_Coil( "DB440_MACHINE_ALARM_DECODING".ALARMS_UNIT_02.ST4_CLEANING.IS_SEOC_ALARMS )
   END_RUNG
   // the same network as SCL:
   // ENO of a box is taken as its EN; it also drops when the box reports an error
   #_w1 := NOT (NOT #AX_TORQUE_EXCEEDED_ALM);
   IF #_w1 THEN "DB440_MACHINE_ALARM_DECODING".GLOBAL_ALARMS_MACHINE.ALARM_DECODING := #DB_NUMBER; END_IF;
   #_w2 := #_w1 AND (#UNIT_ALARM = 1);
   #_w3 := #_w2 AND (#STATION_ALARM = 0);
   IF #_w3 AND "LBP_Chan1".E_ProgRunning THEN
       "DB440_MACHINE_ALARM_DECODING".ALARMS_UNIT_01.ST0_TRANSFER.RHP_SEOC_ALARMS := TRUE;
   END_IF;
   IF #_w3 AND NOT "LBP_Chan1".E_ProgRunning AND NOT "DB440_MACHINE_ALARM_DECODING".ALARMS_UNIT_01.ST0_TRANSFER.RHP_SEOC_ALARMS THEN
       "DB440_MACHINE_ALARM_DECODING".ALARMS_UNIT_01.ST0_TRANSFER.IS_SEOC_ALARMS := TRUE;
   END_IF;
   #_w4 := #_w2 AND (#STATION_ALARM = 1);
   IF #_w4 AND "LBP_Chan1".E_ProgRunning THEN
       "DB440_MACHINE_ALARM_DECODING".ALARMS_UNIT_01.ST1_LOAD_UNLOAD.RHP_SEOC_ALARMS := TRUE;
   END_IF;
   IF #_w4 AND NOT "LBP_Chan1".E_ProgRunning AND NOT "DB440_MACHINE_ALARM_DECODING".ALARMS_UNIT_01.ST1_LOAD_UNLOAD.RHP_SEOC_ALARMS THEN
       "DB440_MACHINE_ALARM_DECODING".ALARMS_UNIT_01.ST1_LOAD_UNLOAD.IS_SEOC_ALARMS := TRUE;
   END_IF;
   #_w5 := #_w2 AND (#STATION_ALARM = 2);
   IF #_w5 THEN "DB440_MACHINE_ALARM_DECODING".ALARMS_UNIT_01.ST2_SPARE.RHP_SEOC_ALARMS := TRUE; END_IF;
   IF #_w5 AND NOT "DB440_MACHINE_ALARM_DECODING".ALARMS_UNIT_01.ST2_SPARE.RHP_SEOC_ALARMS THEN
       "DB440_MACHINE_ALARM_DECODING".ALARMS_UNIT_01.ST2_SPARE.IS_SEOC_ALARMS := TRUE;
   END_IF;
   #_w6 := #_w2 AND (#STATION_ALARM = 3);
   IF #_w6 AND "LBP_Chan2".E_ProgRunning THEN
       "DB440_MACHINE_ALARM_DECODING".ALARMS_UNIT_01.ST3_CLADDING.RHP_SEOC_ALARMS := TRUE;
   END_IF;
   IF #_w6 AND NOT "LBP_Chan2".E_ProgRunning AND NOT "DB440_MACHINE_ALARM_DECODING".ALARMS_UNIT_01.ST3_CLADDING.RHP_SEOC_ALARMS THEN
       "DB440_MACHINE_ALARM_DECODING".ALARMS_UNIT_01.ST3_CLADDING.IS_SEOC_ALARMS := TRUE;
   END_IF;
   #_w7 := #_w2 AND (#STATION_ALARM = 4);
   IF #_w7 AND "LBP_Chan3".E_ProgRunning THEN
       "DB440_MACHINE_ALARM_DECODING".ALARMS_UNIT_01.ST4_CLEANING.RHP_SEOC_ALARMS := TRUE;
   END_IF;
   IF #_w7 AND NOT "LBP_Chan3".E_ProgRunning AND NOT "DB440_MACHINE_ALARM_DECODING".ALARMS_UNIT_01.ST4_CLEANING.RHP_SEOC_ALARMS THEN
       "DB440_MACHINE_ALARM_DECODING".ALARMS_UNIT_01.ST4_CLEANING.IS_SEOC_ALARMS := TRUE;
   END_IF;
   #_w8 := #_w1 AND (#UNIT_ALARM = 2);
   #_w9 := #_w8 AND (#STATION_ALARM = 0);
   IF #_w9 AND "LBP_Chan4".E_ProgRunning THEN
       "DB440_MACHINE_ALARM_DECODING".ALARMS_UNIT_02.ST0_TRANSFER.RHP_SEOC_ALARMS := TRUE;
   END_IF;
   IF #_w9 AND NOT "LBP_Chan4".E_ProgRunning AND NOT "DB440_MACHINE_ALARM_DECODING".ALARMS_UNIT_02.ST0_TRANSFER.RHP_SEOC_ALARMS THEN
       "DB440_MACHINE_ALARM_DECODING".ALARMS_UNIT_02.ST0_TRANSFER.IS_SEOC_ALARMS := TRUE;
   END_IF;
   #_w10 := #_w8 AND (#STATION_ALARM = 1);
   IF #_w10 AND "LBP_Chan4".E_ProgRunning THEN
       "DB440_MACHINE_ALARM_DECODING".ALARMS_UNIT_02.ST1_LOAD_UNLOAD.RHP_SEOC_ALARMS := TRUE;
   END_IF;
   IF #_w10 AND NOT "LBP_Chan4".E_ProgRunning AND NOT "DB440_MACHINE_ALARM_DECODING".ALARMS_UNIT_02.ST1_LOAD_UNLOAD.RHP_SEOC_ALARMS THEN
       "DB440_MACHINE_ALARM_DECODING".ALARMS_UNIT_02.ST1_LOAD_UNLOAD.IS_SEOC_ALARMS := TRUE;
   END_IF;
   #_w11 := #_w8 AND (#STATION_ALARM = 2);
   IF #_w11 AND "LBP_Chan5".E_ProgRunning THEN
       "DB440_MACHINE_ALARM_DECODING".ALARMS_UNIT_02.ST2_MEASURING.RHP_SEOC_ALARMS := TRUE;
   END_IF;
   IF #_w11 AND NOT "LBP_Chan5".E_ProgRunning AND NOT "DB440_MACHINE_ALARM_DECODING".ALARMS_UNIT_02.ST2_MEASURING.RHP_SEOC_ALARMS THEN
       "DB440_MACHINE_ALARM_DECODING".ALARMS_UNIT_02.ST2_MEASURING.IS_SEOC_ALARMS := TRUE;
   END_IF;
   #_w12 := #_w8 AND (#STATION_ALARM = 3);
   IF #_w12 AND "LBP_Chan6".E_ProgRunning THEN
       "DB440_MACHINE_ALARM_DECODING".ALARMS_UNIT_02.ST3_CLADDING.RHP_SEOC_ALARMS := TRUE;
   END_IF;
   IF #_w12 AND NOT "LBP_Chan6".E_ProgRunning AND NOT "DB440_MACHINE_ALARM_DECODING".ALARMS_UNIT_02.ST3_CLADDING.RHP_SEOC_ALARMS THEN
       "DB440_MACHINE_ALARM_DECODING".ALARMS_UNIT_02.ST3_CLADDING.IS_SEOC_ALARMS := TRUE;
   END_IF;
   #_w13 := #_w8 AND (#STATION_ALARM = 4);
   IF #_w13 AND "LBP_Chan7".E_ProgRunning THEN
       "DB440_MACHINE_ALARM_DECODING".ALARMS_UNIT_02.ST4_CLEANING.RHP_SEOC_ALARMS := TRUE;
   END_IF;
   IF #_w13 AND NOT "LBP_Chan7".E_ProgRunning AND NOT "DB440_MACHINE_ALARM_DECODING".ALARMS_UNIT_02.ST4_CLEANING.RHP_SEOC_ALARMS THEN
       "DB440_MACHINE_ALARM_DECODING".ALARMS_UNIT_02.ST4_CLEANING.IS_SEOC_ALARMS := TRUE;
   END_IF;
   #_w14 := #_w1 AND (#UNIT_ALARM = 3);
   IF #_w14 AND "LBP_Chan8".E_ProgRunning THEN
       "DB440_MACHINE_ALARM_DECODING".ALARMS_UNIT_03.RHP_SEOC_ALARMS := TRUE;
   END_IF;
   IF #_w14 AND NOT "LBP_Chan8".E_ProgRunning AND NOT "DB440_MACHINE_ALARM_DECODING".ALARMS_UNIT_03.RHP_SEOC_ALARMS THEN
       "DB440_MACHINE_ALARM_DECODING".ALARMS_UNIT_03.IS_SEOC_ALARMS := TRUE;
   END_IF;
   #_w15 := #_w1 AND (#STATION_ALARM = 4);
   IF #_w15 AND "LBP_Chan10".E_ProgRunning THEN
       "DB440_MACHINE_ALARM_DECODING".ALARMS_UNIT_02.ST4_CLEANING.RHP_SEOC_ALARMS := TRUE;
   END_IF;
   IF #_w15 AND NOT "LBP_Chan10".E_ProgRunning AND NOT "DB440_MACHINE_ALARM_DECODING".ALARMS_UNIT_02.ST4_CLEANING.RHP_SEOC_ALARMS THEN
       "DB440_MACHINE_ALARM_DECODING".ALARMS_UNIT_02.ST4_CLEANING.IS_SEOC_ALARMS := TRUE;
   END_IF;
END_REGION

REGION Network 30: PROGRAMMING FAULT
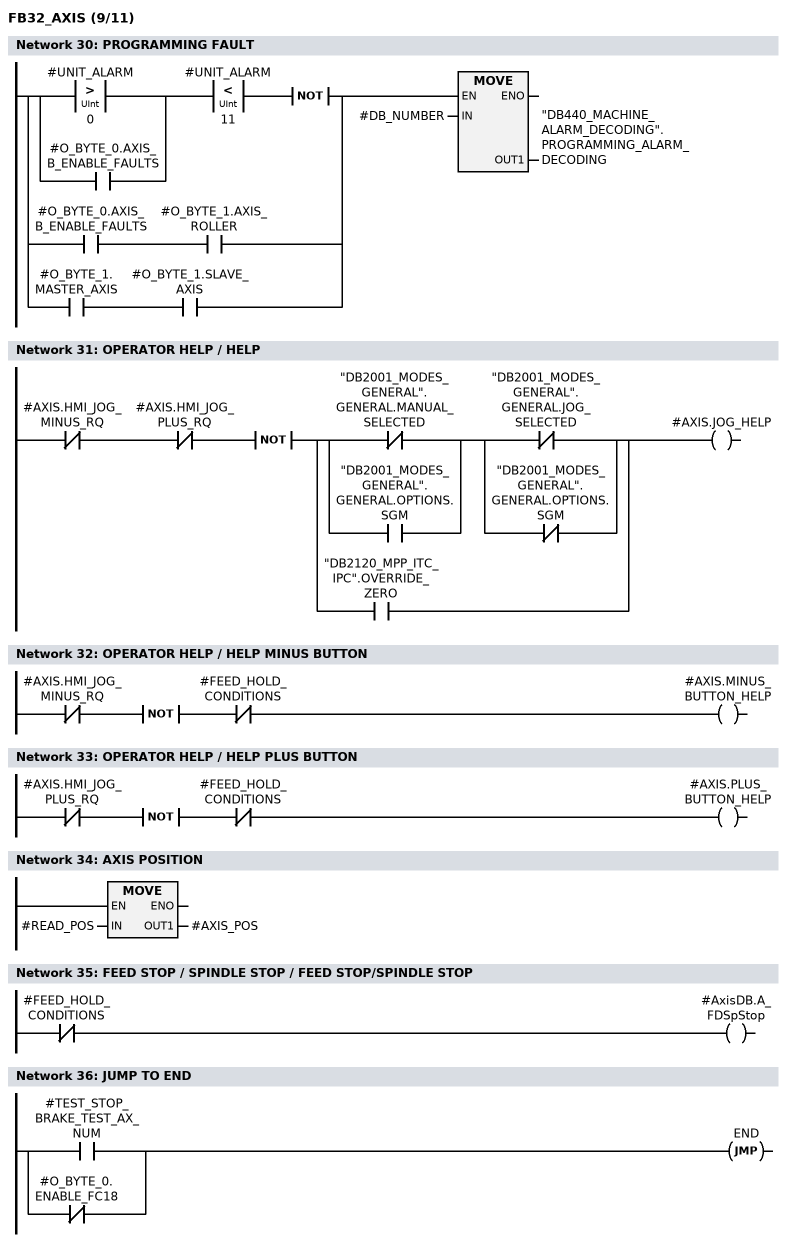
   RUNG wire#powerrail
      { S7_Templates := "SrcType := UInt" } GT_Contact(in1 := #UNIT_ALARM, in2 := 0)
      wire#w1
      { S7_Templates := "SrcType := UInt" } LT_Contact(in1 := #UNIT_ALARM, in2 := 11)
      Not()
      wire#w2
      Move(in := #DB_NUMBER, out1 => "DB440_MACHINE_ALARM_DECODING".PROGRAMMING_ALARM_DECODING)
   END_RUNG
   RUNG wire#powerrail
      Contact( #O_BYTE_0.AXIS_B_ENABLE_FAULTS )
   END_RUNG wire#w1
   RUNG wire#powerrail
      Contact( #O_BYTE_0.AXIS_B_ENABLE_FAULTS )
      Contact( #O_BYTE_1.AXIS_ROLLER )
   END_RUNG wire#w2
   RUNG wire#powerrail
      Contact( #O_BYTE_1.MASTER_AXIS )
      Contact( #O_BYTE_1.SLAVE_AXIS )
   END_RUNG wire#w2
   // the same network as SCL:
   IF NOT (((#UNIT_ALARM > 0) OR #O_BYTE_0.AXIS_B_ENABLE_FAULTS) AND (#UNIT_ALARM < 11)) OR (#O_BYTE_0.AXIS_B_ENABLE_FAULTS AND #O_BYTE_1.AXIS_ROLLER) OR (#O_BYTE_1.MASTER_AXIS AND #O_BYTE_1.SLAVE_AXIS) THEN
       "DB440_MACHINE_ALARM_DECODING".PROGRAMMING_ALARM_DECODING := #DB_NUMBER;
   END_IF;
END_REGION

REGION Network 31: OPERATOR HELP / HELP
   RUNG wire#powerrail
      I_Contact( #AXIS.HMI_JOG_MINUS_RQ )
      I_Contact( #AXIS.HMI_JOG_PLUS_RQ )
      Not()
      wire#w1
      I_Contact( "DB2001_MODES_GENERAL".GENERAL.MANUAL_SELECTED )
      wire#w2
      I_Contact( "DB2001_MODES_GENERAL".GENERAL.JOG_SELECTED )
      wire#w3
      Coil( #AXIS.JOG_HELP )
   END_RUNG
   RUNG wire#w1
      Contact( "DB2001_MODES_GENERAL".GENERAL.OPTIONS.SGM )
   END_RUNG wire#w2
   RUNG wire#w2
      I_Contact( "DB2001_MODES_GENERAL".GENERAL.OPTIONS.SGM )
   END_RUNG wire#w3
   RUNG wire#w1
      Contact( "DB2120_MPP_ITC_IPC".OVERRIDE_ZERO )
   END_RUNG wire#w3
   // the same network as SCL:
   #AXIS.JOG_HELP := NOT (NOT #AXIS.HMI_JOG_MINUS_RQ AND NOT #AXIS.HMI_JOG_PLUS_RQ) AND (((NOT "DB2001_MODES_GENERAL".GENERAL.MANUAL_SELECTED OR "DB2001_MODES_GENERAL".GENERAL.OPTIONS.SGM) AND (NOT "DB2001_MODES_GENERAL".GENERAL.JOG_SELECTED OR NOT "DB2001_MODES_GENERAL".GENERAL.OPTIONS.SGM)) OR "DB2120_MPP_ITC_IPC".OVERRIDE_ZERO);
END_REGION

REGION Network 32: OPERATOR HELP / HELP MINUS BUTTON
   RUNG wire#powerrail
      I_Contact( #AXIS.HMI_JOG_MINUS_RQ )
      Not()
      I_Contact( #FEED_HOLD_CONDITIONS )
      Coil( #AXIS.MINUS_BUTTON_HELP )
   END_RUNG
   // the same network as SCL:
   #AXIS.MINUS_BUTTON_HELP := NOT (NOT #AXIS.HMI_JOG_MINUS_RQ) AND NOT #FEED_HOLD_CONDITIONS;
END_REGION

REGION Network 33: OPERATOR HELP / HELP PLUS BUTTON
   RUNG wire#powerrail
      I_Contact( #AXIS.HMI_JOG_PLUS_RQ )
      Not()
      I_Contact( #FEED_HOLD_CONDITIONS )
      Coil( #AXIS.PLUS_BUTTON_HELP )
   END_RUNG
   // the same network as SCL:
   #AXIS.PLUS_BUTTON_HELP := NOT (NOT #AXIS.HMI_JOG_PLUS_RQ) AND NOT #FEED_HOLD_CONDITIONS;
END_REGION

REGION Network 34: AXIS POSITION
   RUNG wire#powerrail
      { S7_GenerateENO := "TRUE" } Move(in := #READ_POS, out1 => #AXIS_POS)
   END_RUNG
   // the same network as SCL:
   #AXIS_POS := #READ_POS;
END_REGION

REGION Network 35: FEED STOP / SPINDLE STOP / FEED STOP/SPINDLE STOP
   RUNG wire#powerrail
      I_Contact( #FEED_HOLD_CONDITIONS )
      Coil( #AxisDB.A_FDSpStop )
   END_RUNG
   // the same network as SCL:
   #AxisDB.A_FDSpStop := NOT #FEED_HOLD_CONDITIONS;
END_REGION

REGION Network 36: JUMP TO END
   RUNG wire#powerrail
      Contact( #TEST_STOP_BRAKE_TEST_AX_NUM )
      wire#w1
      JumpCoil( END )
   END_RUNG
   RUNG wire#powerrail
      I_Contact( #O_BYTE_0.ENABLE_FC18 )
   END_RUNG wire#w1
   // the same network as SCL:
   IF #TEST_STOP_BRAKE_TEST_AX_NUM OR NOT #O_BYTE_0.ENABLE_FC18 THEN GOTO END; END_IF;
END_REGION

REGION Network 37: POS TO GO / AXIS POSITION TO GO
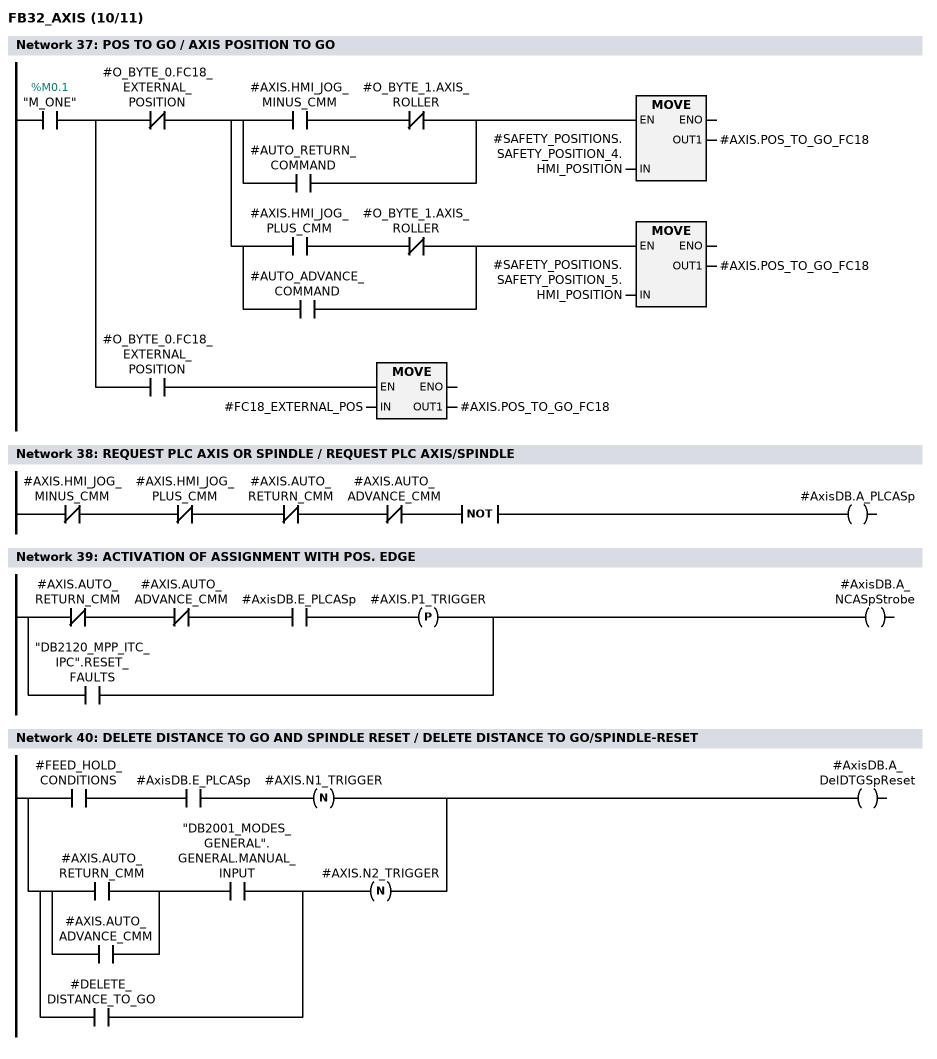
   RUNG wire#powerrail
      Contact( "M_ONE" )
      wire#w1
      I_Contact( #O_BYTE_0.FC18_EXTERNAL_POSITION )
      wire#w2
      Contact( #AXIS.HMI_JOG_MINUS_CMM )
      I_Contact( #O_BYTE_1.AXIS_ROLLER )
      wire#w3
      { S7_GenerateENO := "TRUE" } Move(in := #SAFETY_POSITIONS.SAFETY_POSITION_4.HMI_POSITION, out1 => #AXIS.POS_TO_GO_FC18)
   END_RUNG
   RUNG wire#w2
      Contact( #AUTO_RETURN_COMMAND )
   END_RUNG wire#w3
   RUNG wire#w2
      Contact( #AXIS.HMI_JOG_PLUS_CMM )
      I_Contact( #O_BYTE_1.AXIS_ROLLER )
      wire#w4
      { S7_GenerateENO := "TRUE" } Move(in := #SAFETY_POSITIONS.SAFETY_POSITION_5.HMI_POSITION, out1 => #AXIS.POS_TO_GO_FC18)
   END_RUNG
   RUNG wire#w2
      Contact( #AUTO_ADVANCE_COMMAND )
   END_RUNG wire#w4
   RUNG wire#w1
      Contact( #O_BYTE_0.FC18_EXTERNAL_POSITION )
      { S7_GenerateENO := "TRUE" } Move(in := #FC18_EXTERNAL_POS, out1 => #AXIS.POS_TO_GO_FC18)
   END_RUNG
   // the same network as SCL:
   #_w1 := "M_ONE" AND NOT #O_BYTE_0.FC18_EXTERNAL_POSITION;
   IF #_w1 AND ((#AXIS.HMI_JOG_MINUS_CMM AND NOT #O_BYTE_1.AXIS_ROLLER) OR #AUTO_RETURN_COMMAND) THEN
       #AXIS.POS_TO_GO_FC18 := #SAFETY_POSITIONS.SAFETY_POSITION_4.HMI_POSITION;
   END_IF;
   IF #_w1 AND ((#AXIS.HMI_JOG_PLUS_CMM AND NOT #O_BYTE_1.AXIS_ROLLER) OR #AUTO_ADVANCE_COMMAND) THEN
       #AXIS.POS_TO_GO_FC18 := #SAFETY_POSITIONS.SAFETY_POSITION_5.HMI_POSITION;
   END_IF;
   IF "M_ONE" AND #O_BYTE_0.FC18_EXTERNAL_POSITION THEN #AXIS.POS_TO_GO_FC18 := #FC18_EXTERNAL_POS; END_IF;
END_REGION

REGION Network 38: REQUEST PLC AXIS OR SPINDLE / REQUEST PLC AXIS/SPINDLE
   RUNG wire#powerrail
      I_Contact( #AXIS.HMI_JOG_MINUS_CMM )
      I_Contact( #AXIS.HMI_JOG_PLUS_CMM )
      I_Contact( #AXIS.AUTO_RETURN_CMM )
      I_Contact( #AXIS.AUTO_ADVANCE_CMM )
      Not()
      Coil( #AxisDB.A_PLCASp )
   END_RUNG
   // the same network as SCL:
   #AxisDB.A_PLCASp := NOT (NOT #AXIS.HMI_JOG_MINUS_CMM AND NOT #AXIS.HMI_JOG_PLUS_CMM AND NOT #AXIS.AUTO_RETURN_CMM AND NOT #AXIS.AUTO_ADVANCE_CMM);
END_REGION

REGION Network 39: ACTIVATION OF ASSIGNMENT WITH POS. EDGE
   RUNG wire#powerrail
      I_Contact( #AXIS.AUTO_RETURN_CMM )
      I_Contact( #AXIS.AUTO_ADVANCE_CMM )
      Contact( #AxisDB.E_PLCASp )
      P_Trig( #AXIS.P1_TRIGGER )
      wire#w1
      Coil( #AxisDB.A_NCASpStrobe )
   END_RUNG
   RUNG wire#powerrail
      Contact( "DB2120_MPP_ITC_IPC".RESET_FAULTS )
   END_RUNG wire#w1
   // the same network as SCL:
   #_w1 := NOT #AXIS.AUTO_RETURN_CMM AND NOT #AXIS.AUTO_ADVANCE_CMM AND #AxisDB.E_PLCASp;
   #_w2 := #_w1 AND NOT #AXIS.P1_TRIGGER;   // rising edge
   #AXIS.P1_TRIGGER := #_w1;
   #AxisDB.A_NCASpStrobe := #_w2 OR "DB2120_MPP_ITC_IPC".RESET_FAULTS;
END_REGION

REGION Network 40: DELETE DISTANCE TO GO AND SPINDLE RESET / DELETE DISTANCE TO GO/SPINDLE-RESET
   RUNG wire#powerrail
      Contact( #FEED_HOLD_CONDITIONS )
      Contact( #AxisDB.E_PLCASp )
      N_Trig( #AXIS.N1_TRIGGER )
      wire#w1
      Coil( #AxisDB.A_DelDTGSpReset )
   END_RUNG
   RUNG wire#powerrail
      Contact( #AXIS.AUTO_RETURN_CMM )
      wire#w2
      Contact( "DB2001_MODES_GENERAL".GENERAL.MANUAL_INPUT )
      wire#w3
      N_Trig( #AXIS.N2_TRIGGER )
   END_RUNG wire#w1
   RUNG wire#powerrail
      Contact( #AXIS.AUTO_ADVANCE_CMM )
   END_RUNG wire#w2
   RUNG wire#powerrail
      Contact( #DELETE_DISTANCE_TO_GO )
   END_RUNG wire#w3
   // the same network as SCL:
   #_w1 := #FEED_HOLD_CONDITIONS AND #AxisDB.E_PLCASp;
   #_w2 := NOT #_w1 AND #AXIS.N1_TRIGGER;   // falling edge
   #AXIS.N1_TRIGGER := #_w1;
   #_w3 := ((#AXIS.AUTO_RETURN_CMM OR #AXIS.AUTO_ADVANCE_CMM) AND "DB2001_MODES_GENERAL".GENERAL.MANUAL_INPUT) OR #DELETE_DISTANCE_TO_GO;
   #_w4 := NOT #_w3 AND #AXIS.N2_TRIGGER;   // falling edge
   #AXIS.N2_TRIGGER := #_w3;
   #AxisDB.A_DelDTGSpReset := #_w2 OR #_w4;
END_REGION

REGION Network 41: FC18
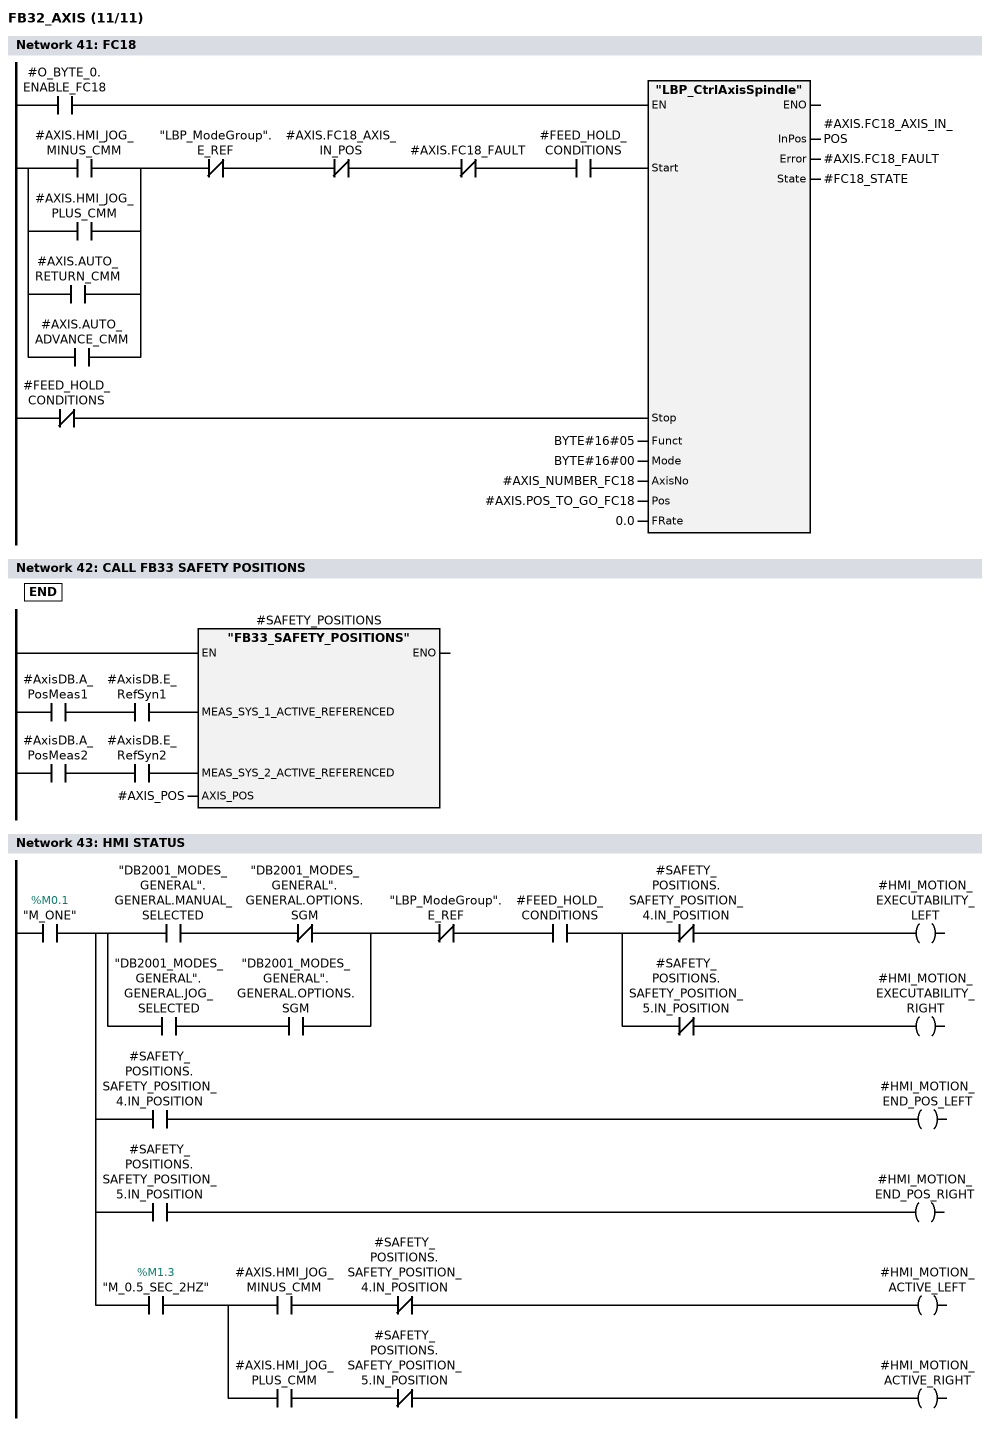
   RUNG wire#powerrail
      Contact( #O_BYTE_0.ENABLE_FC18 )
      "LBP_CtrlAxisSpindle"(Start := wire#w2, Stop := wire#w3, Funct := BYTE#16#05, Mode := BYTE#16#00, AxisNo := #AXIS_NUMBER_FC18, Pos := #AXIS.POS_TO_GO_FC18, FRate := 0.0, InPos => #AXIS.FC18_AXIS_IN_POS, Error => #AXIS.FC18_FAULT, State => #FC18_STATE)
   END_RUNG
   RUNG wire#powerrail
      Contact( #AXIS.HMI_JOG_MINUS_CMM )
      wire#w1
      I_Contact( "LBP_ModeGroup".E_REF )
      I_Contact( #AXIS.FC18_AXIS_IN_POS )
      I_Contact( #AXIS.FC18_FAULT )
      Contact( #FEED_HOLD_CONDITIONS )
   END_RUNG wire#w2
   RUNG wire#powerrail
      Contact( #AXIS.HMI_JOG_PLUS_CMM )
   END_RUNG wire#w1
   RUNG wire#powerrail
      Contact( #AXIS.AUTO_RETURN_CMM )
   END_RUNG wire#w1
   RUNG wire#powerrail
      Contact( #AXIS.AUTO_ADVANCE_CMM )
   END_RUNG wire#w1
   RUNG wire#powerrail
      I_Contact( #FEED_HOLD_CONDITIONS )
   END_RUNG wire#w3
   // the same network as SCL:
   IF #O_BYTE_0.ENABLE_FC18 THEN
       "LBP_CtrlAxisSpindle"(Start := (#AXIS.HMI_JOG_MINUS_CMM OR #AXIS.HMI_JOG_PLUS_CMM OR #AXIS.AUTO_RETURN_CMM OR #AXIS.AUTO_ADVANCE_CMM) AND NOT "LBP_ModeGroup".E_REF AND NOT #AXIS.FC18_AXIS_IN_POS AND NOT #AXIS.FC18_FAULT AND #FEED_HOLD_CONDITIONS,
                             Stop := NOT #FEED_HOLD_CONDITIONS,
                             Funct := BYTE#16#05,
                             Mode := BYTE#16#00,
                             AxisNo := #AXIS_NUMBER_FC18,
                             Pos := #AXIS.POS_TO_GO_FC18,
                             FRate := 0.0,
                             InPos => #AXIS.FC18_AXIS_IN_POS,
                             Error => #AXIS.FC18_FAULT,
                             State => #FC18_STATE);
   END_IF;
END_REGION

REGION Network 42: CALL FB33 SAFETY POSITIONS
   Label( END )
   RUNG wire#powerrail
      #SAFETY_POSITIONS(MEAS_SYS_1_ACTIVE_REFERENCED := wire#w1, MEAS_SYS_2_ACTIVE_REFERENCED := wire#w2, AXIS_POS := #AXIS_POS)
   END_RUNG
   RUNG wire#powerrail
      Contact( #AxisDB.A_PosMeas1 )
      Contact( #AxisDB.E_RefSyn1 )
   END_RUNG wire#w1
   RUNG wire#powerrail
      Contact( #AxisDB.A_PosMeas2 )
      Contact( #AxisDB.E_RefSyn2 )
   END_RUNG wire#w2
   // the same network as SCL:
   END:
   #SAFETY_POSITIONS(MEAS_SYS_1_ACTIVE_REFERENCED := #AxisDB.A_PosMeas1 AND #AxisDB.E_RefSyn1,   // "FB33_SAFETY_POSITIONS"
                     MEAS_SYS_2_ACTIVE_REFERENCED := #AxisDB.A_PosMeas2 AND #AxisDB.E_RefSyn2,
                     AXIS_POS := #AXIS_POS);
END_REGION

REGION Network 43: HMI STATUS
   RUNG wire#powerrail
      Contact( "M_ONE" )
      wire#w1
      Contact( "DB2001_MODES_GENERAL".GENERAL.MANUAL_SELECTED )
      I_Contact( "DB2001_MODES_GENERAL".GENERAL.OPTIONS.SGM )
      wire#w2
      I_Contact( "LBP_ModeGroup".E_REF )
      Contact( #FEED_HOLD_CONDITIONS )
      wire#w3
      I_Contact( #SAFETY_POSITIONS.SAFETY_POSITION_4.IN_POSITION )
      Coil( #HMI_MOTION_EXECUTABILITY_LEFT )
   END_RUNG
   RUNG wire#w1
      Contact( "DB2001_MODES_GENERAL".GENERAL.JOG_SELECTED )
      Contact( "DB2001_MODES_GENERAL".GENERAL.OPTIONS.SGM )
   END_RUNG wire#w2
   RUNG wire#w3
      I_Contact( #SAFETY_POSITIONS.SAFETY_POSITION_5.IN_POSITION )
      Coil( #HMI_MOTION_EXECUTABILITY_RIGHT )
   END_RUNG
   RUNG wire#w1
      Contact( #SAFETY_POSITIONS.SAFETY_POSITION_4.IN_POSITION )
      Coil( #HMI_MOTION_END_POS_LEFT )
   END_RUNG
   RUNG wire#w1
      Contact( #SAFETY_POSITIONS.SAFETY_POSITION_5.IN_POSITION )
      Coil( #HMI_MOTION_END_POS_RIGHT )
   END_RUNG
   RUNG wire#w1
      Contact( "M_0.5_SEC_2HZ" )
      wire#w4
      Contact( #AXIS.HMI_JOG_MINUS_CMM )
      I_Contact( #SAFETY_POSITIONS.SAFETY_POSITION_4.IN_POSITION )
      Coil( #HMI_MOTION_ACTIVE_LEFT )
   END_RUNG
   RUNG wire#w4
      Contact( #AXIS.HMI_JOG_PLUS_CMM )
      I_Contact( #SAFETY_POSITIONS.SAFETY_POSITION_5.IN_POSITION )
      Coil( #HMI_MOTION_ACTIVE_RIGHT )
   END_RUNG
   // the same network as SCL:
   #_w1 := "M_ONE" AND (("DB2001_MODES_GENERAL".GENERAL.MANUAL_SELECTED AND NOT "DB2001_MODES_GENERAL".GENERAL.OPTIONS.SGM) OR ("DB2001_MODES_GENERAL".GENERAL.JOG_SELECTED AND "DB2001_MODES_GENERAL".GENERAL.OPTIONS.SGM)) AND NOT "LBP_ModeGroup".E_REF AND #FEED_HOLD_CONDITIONS;
   #HMI_MOTION_EXECUTABILITY_LEFT := #_w1 AND NOT #SAFETY_POSITIONS.SAFETY_POSITION_4.IN_POSITION;
   #HMI_MOTION_EXECUTABILITY_RIGHT := #_w1 AND NOT #SAFETY_POSITIONS.SAFETY_POSITION_5.IN_POSITION;
   #HMI_MOTION_END_POS_LEFT := "M_ONE" AND #SAFETY_POSITIONS.SAFETY_POSITION_4.IN_POSITION;
   #HMI_MOTION_END_POS_RIGHT := "M_ONE" AND #SAFETY_POSITIONS.SAFETY_POSITION_5.IN_POSITION;
   #_w2 := "M_ONE" AND "M_0.5_SEC_2HZ";
   #HMI_MOTION_ACTIVE_LEFT := #_w2 AND #AXIS.HMI_JOG_MINUS_CMM AND NOT #SAFETY_POSITIONS.SAFETY_POSITION_4.IN_POSITION;
   #HMI_MOTION_ACTIVE_RIGHT := #_w2 AND #AXIS.HMI_JOG_PLUS_CMM AND NOT #SAFETY_POSITIONS.SAFETY_POSITION_5.IN_POSITION;
END_REGION
END_FUNCTION_BLOCK

FUNCTION "FC301_ALARMS_OPERATOR_HELP" : Void   // FC301, LAD
{ S7_Optimized_Access := 'TRUE' }
VERSION : 0.1
// stored: AutoNumber false, IsIECCheckEnabled false, SetENOAutomatically false, UDAEnableTagReadback false
   VAR_TEMP
      PART_TYPE : Int;
   END_VAR
   VAR_TEMP   // added for the SCL form of the ladder/FBD networks
      _w1 : Bool;
   END_VAR
BEGIN

REGION Network 1: FC421 HOLA PC ALARM
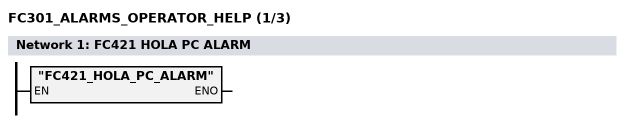
   RUNG wire#powerrail
      "FC421_HOLA_PC_ALARM"()
   END_RUNG
   // the same network as SCL:
   "FC421_HOLA_PC_ALARM"();
END_REGION

REGION Network 2: OPERATOR HELP
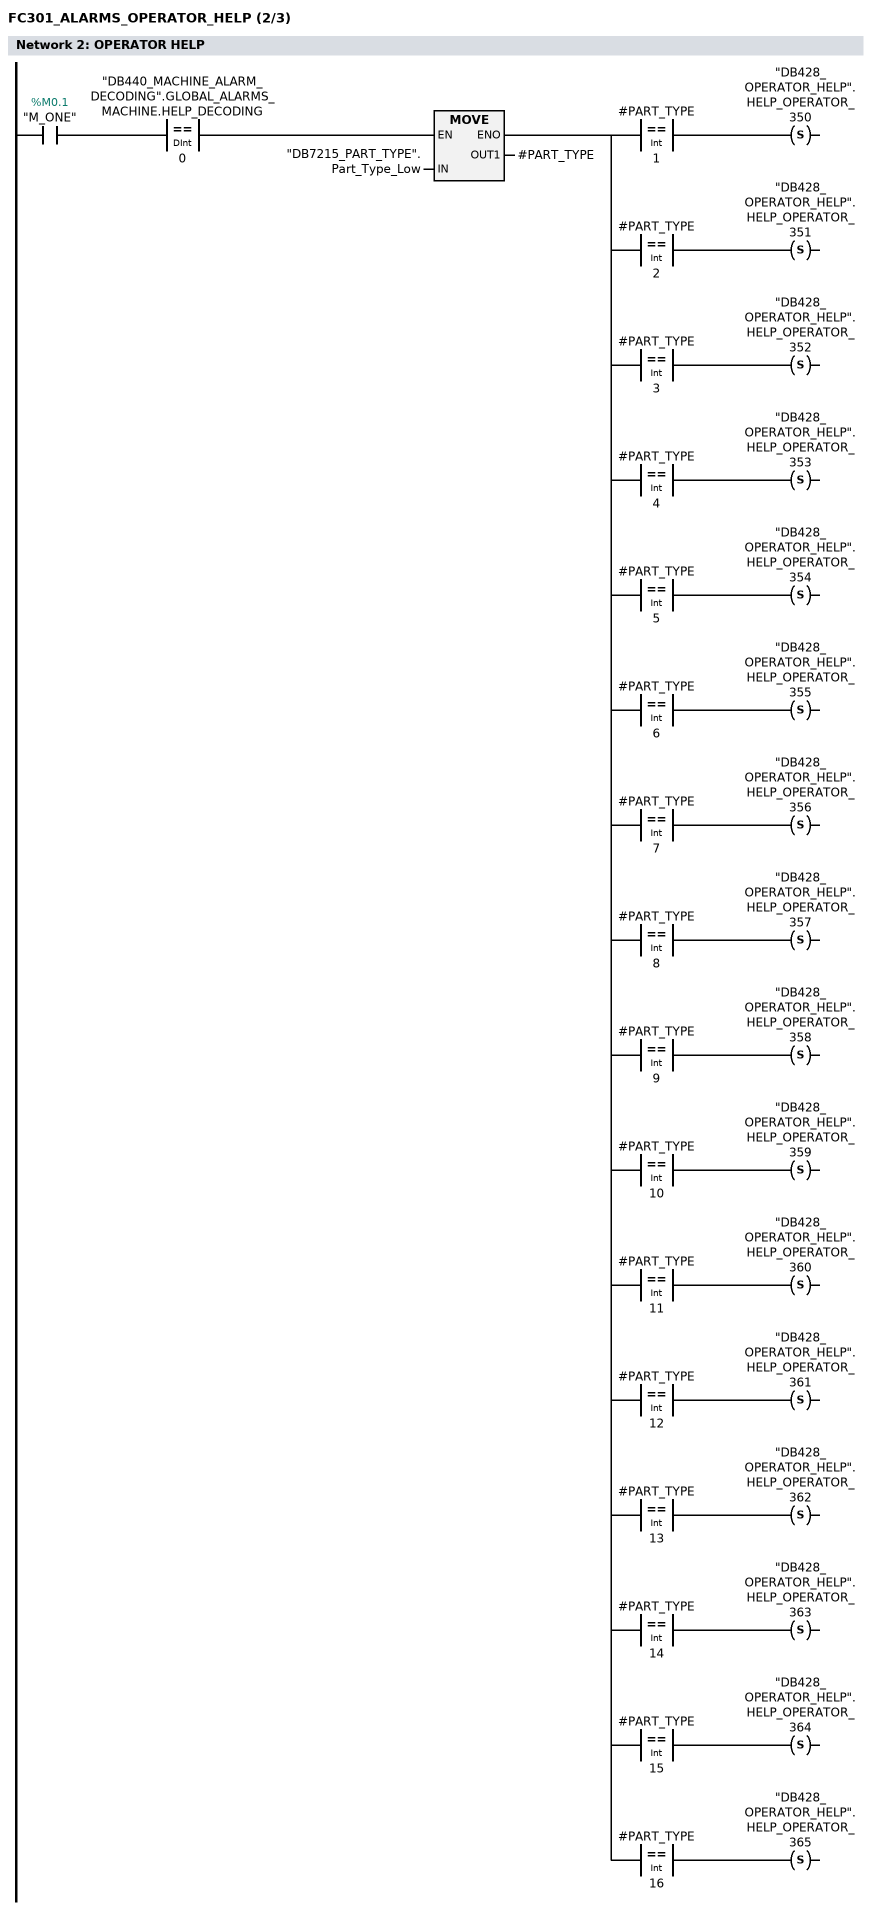
   RUNG wire#powerrail
      Contact( "M_ONE" )
      { S7_Templates := "SrcType := DInt" } EQ_Contact(in1 := "DB440_MACHINE_ALARM_DECODING".GLOBAL_ALARMS_MACHINE.HELP_DECODING, in2 := 0)
      { S7_GenerateENO := "TRUE" } Move(in := "DB7215_PART_TYPE".Part_Type_Low, out1 => #PART_TYPE)
      wire#w1
      { S7_Templates := "SrcType := Int" } EQ_Contact(in1 := #PART_TYPE, in2 := 1)
      S_Coil( "DB428_OPERATOR_HELP".HELP_OPERATOR_350 )
   END_RUNG
   RUNG wire#w1
      { S7_Templates := "SrcType := Int" } EQ_Contact(in1 := #PART_TYPE, in2 := 2)
      S_Coil( "DB428_OPERATOR_HELP".HELP_OPERATOR_351 )
   END_RUNG
   RUNG wire#w1
      { S7_Templates := "SrcType := Int" } EQ_Contact(in1 := #PART_TYPE, in2 := 3)
      S_Coil( "DB428_OPERATOR_HELP".HELP_OPERATOR_352 )
   END_RUNG
   RUNG wire#w1
      { S7_Templates := "SrcType := Int" } EQ_Contact(in1 := #PART_TYPE, in2 := 4)
      S_Coil( "DB428_OPERATOR_HELP".HELP_OPERATOR_353 )
   END_RUNG
   RUNG wire#w1
      { S7_Templates := "SrcType := Int" } EQ_Contact(in1 := #PART_TYPE, in2 := 5)
      S_Coil( "DB428_OPERATOR_HELP".HELP_OPERATOR_354 )
   END_RUNG
   RUNG wire#w1
      { S7_Templates := "SrcType := Int" } EQ_Contact(in1 := #PART_TYPE, in2 := 6)
      S_Coil( "DB428_OPERATOR_HELP".HELP_OPERATOR_355 )
   END_RUNG
   RUNG wire#w1
      { S7_Templates := "SrcType := Int" } EQ_Contact(in1 := #PART_TYPE, in2 := 7)
      S_Coil( "DB428_OPERATOR_HELP".HELP_OPERATOR_356 )
   END_RUNG
   RUNG wire#w1
      { S7_Templates := "SrcType := Int" } EQ_Contact(in1 := #PART_TYPE, in2 := 8)
      S_Coil( "DB428_OPERATOR_HELP".HELP_OPERATOR_357 )
   END_RUNG
   RUNG wire#w1
      { S7_Templates := "SrcType := Int" } EQ_Contact(in1 := #PART_TYPE, in2 := 9)
      S_Coil( "DB428_OPERATOR_HELP".HELP_OPERATOR_358 )
   END_RUNG
   RUNG wire#w1
      { S7_Templates := "SrcType := Int" } EQ_Contact(in1 := #PART_TYPE, in2 := 10)
      S_Coil( "DB428_OPERATOR_HELP".HELP_OPERATOR_359 )
   END_RUNG
   RUNG wire#w1
      { S7_Templates := "SrcType := Int" } EQ_Contact(in1 := #PART_TYPE, in2 := 11)
      S_Coil( "DB428_OPERATOR_HELP".HELP_OPERATOR_360 )
   END_RUNG
   RUNG wire#w1
      { S7_Templates := "SrcType := Int" } EQ_Contact(in1 := #PART_TYPE, in2 := 12)
      S_Coil( "DB428_OPERATOR_HELP".HELP_OPERATOR_361 )
   END_RUNG
   RUNG wire#w1
      { S7_Templates := "SrcType := Int" } EQ_Contact(in1 := #PART_TYPE, in2 := 13)
      S_Coil( "DB428_OPERATOR_HELP".HELP_OPERATOR_362 )
   END_RUNG
   RUNG wire#w1
      { S7_Templates := "SrcType := Int" } EQ_Contact(in1 := #PART_TYPE, in2 := 14)
      S_Coil( "DB428_OPERATOR_HELP".HELP_OPERATOR_363 )
   END_RUNG
   RUNG wire#w1
      { S7_Templates := "SrcType := Int" } EQ_Contact(in1 := #PART_TYPE, in2 := 15)
      S_Coil( "DB428_OPERATOR_HELP".HELP_OPERATOR_364 )
   END_RUNG
   RUNG wire#w1
      { S7_Templates := "SrcType := Int" } EQ_Contact(in1 := #PART_TYPE, in2 := 16)
      S_Coil( "DB428_OPERATOR_HELP".HELP_OPERATOR_365 )
   END_RUNG
   // the same network as SCL:
   // ENO of a box is taken as its EN; it also drops when the box reports an error
   #_w1 := "M_ONE" AND ("DB440_MACHINE_ALARM_DECODING".GLOBAL_ALARMS_MACHINE.HELP_DECODING = 0);
   IF #_w1 THEN #PART_TYPE := "DB7215_PART_TYPE".Part_Type_Low; END_IF;
   IF #_w1 AND (#PART_TYPE = 1) THEN "DB428_OPERATOR_HELP".HELP_OPERATOR_350 := TRUE; END_IF;
   IF #_w1 AND (#PART_TYPE = 2) THEN "DB428_OPERATOR_HELP".HELP_OPERATOR_351 := TRUE; END_IF;
   IF #_w1 AND (#PART_TYPE = 3) THEN "DB428_OPERATOR_HELP".HELP_OPERATOR_352 := TRUE; END_IF;
   IF #_w1 AND (#PART_TYPE = 4) THEN "DB428_OPERATOR_HELP".HELP_OPERATOR_353 := TRUE; END_IF;
   IF #_w1 AND (#PART_TYPE = 5) THEN "DB428_OPERATOR_HELP".HELP_OPERATOR_354 := TRUE; END_IF;
   IF #_w1 AND (#PART_TYPE = 6) THEN "DB428_OPERATOR_HELP".HELP_OPERATOR_355 := TRUE; END_IF;
   IF #_w1 AND (#PART_TYPE = 7) THEN "DB428_OPERATOR_HELP".HELP_OPERATOR_356 := TRUE; END_IF;
   IF #_w1 AND (#PART_TYPE = 8) THEN "DB428_OPERATOR_HELP".HELP_OPERATOR_357 := TRUE; END_IF;
   IF #_w1 AND (#PART_TYPE = 9) THEN "DB428_OPERATOR_HELP".HELP_OPERATOR_358 := TRUE; END_IF;
   IF #_w1 AND (#PART_TYPE = 10) THEN "DB428_OPERATOR_HELP".HELP_OPERATOR_359 := TRUE; END_IF;
   IF #_w1 AND (#PART_TYPE = 11) THEN "DB428_OPERATOR_HELP".HELP_OPERATOR_360 := TRUE; END_IF;
   IF #_w1 AND (#PART_TYPE = 12) THEN "DB428_OPERATOR_HELP".HELP_OPERATOR_361 := TRUE; END_IF;
   IF #_w1 AND (#PART_TYPE = 13) THEN "DB428_OPERATOR_HELP".HELP_OPERATOR_362 := TRUE; END_IF;
   IF #_w1 AND (#PART_TYPE = 14) THEN "DB428_OPERATOR_HELP".HELP_OPERATOR_363 := TRUE; END_IF;
   IF #_w1 AND (#PART_TYPE = 15) THEN "DB428_OPERATOR_HELP".HELP_OPERATOR_364 := TRUE; END_IF;
   IF #_w1 AND (#PART_TYPE = 16) THEN "DB428_OPERATOR_HELP".HELP_OPERATOR_365 := TRUE; END_IF;
END_REGION

REGION Network 3: CALL FC428 OPERATOR HELP
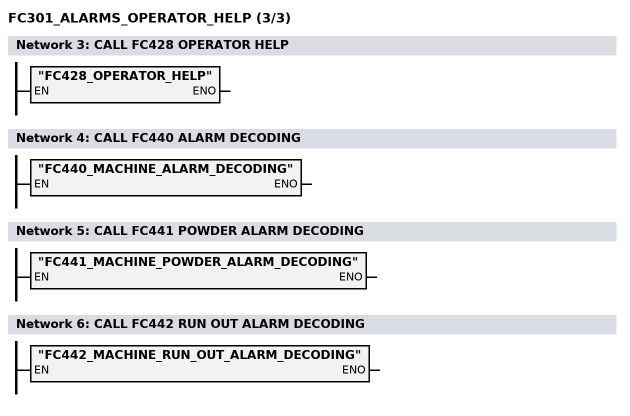
   RUNG wire#powerrail
      "FC428_OPERATOR_HELP"()
   END_RUNG
   // the same network as SCL:
   "FC428_OPERATOR_HELP"();
END_REGION

REGION Network 4: CALL FC440 ALARM DECODING
   RUNG wire#powerrail
      "FC440_MACHINE_ALARM_DECODING"()
   END_RUNG
   // the same network as SCL:
   "FC440_MACHINE_ALARM_DECODING"();
END_REGION

REGION Network 5: CALL FC441 POWDER ALARM DECODING
   RUNG wire#powerrail
      "FC441_MACHINE_POWDER_ALARM_DECODING"()
   END_RUNG
   // the same network as SCL:
   "FC441_MACHINE_POWDER_ALARM_DECODING"();
END_REGION

REGION Network 6: CALL FC442 RUN OUT ALARM DECODING
   RUNG wire#powerrail
      "FC442_MACHINE_RUN_OUT_ALARM_DECODING"()
   END_RUNG
   // the same network as SCL:
   "FC442_MACHINE_RUN_OUT_ALARM_DECODING"();
END_REGION
END_FUNCTION

FUNCTION_BLOCK "FB301_CHANNEL_READ_AXES_POSITIONS"   // FB301, LAD
{ S7_Optimized_Access := 'FALSE' }
AUTHOR : ETXETAR
VERSION : 1.0
// stored: AutoNumber false, IsIECCheckEnabled false, SetENOAutomatically false, UDAEnableTagReadback false
   VAR_INPUT
      NUMBER_AXES_GROUP_1 : Int;   // MAX. VALUE 8 / NUMBER AXES GROUP 1, MAX=8
      NUMBER_AXES_GROUP_2 : Int;   // MAX. VALUE 7 / NUMBER AXES GROUP 2, MAX=8
      NUMBER_AXES_GROUP_3 : Int;   // MAX. VALUE 7 / NUMBER AXES GROUP 3, MAX=4
   END_VAR
   VAR_OUTPUT
      ALARM : Bool;   // ALARM
      AXIS_POSITION_1 : DWord;   // AXIS POSITION 1
      AXIS_POSITION_2 : DWord;   // AXIS POSITION 2
      AXIS_POSITION_3 : DWord;   // AXIS POSITION 3
      AXIS_POSITION_4 : DWord;   // AXIS POSITION 4
      AXIS_POSITION_5 : DWord;   // AXIS POSITION 5
      AXIS_POSITION_6 : DWord;   // AXIS POSITION 6
      AXIS_POSITION_7 : DWord;   // AXIS POSITION 7
      AXIS_POSITION_8 : DWord;   // AXIS POSITION 8
      AXIS_POSITION_9 : DWord;   // AXIS POSITION 9
      AXIS_POSITION_10 : DWord;   // AXIS POSITION 10
      AXIS_POSITION_11 : DWord;   // AXIS POSITION 11
      AXIS_POSITION_12 : DWord;   // AXIS POSITION 12
      AXIS_POSITION_13 : DWord;   // AXIS POSITION 13
      AXIS_POSITION_14 : DWord;   // AXIS POSITION 14
      AXIS_POSITION_15 : DWord;   // AXIS POSITION 15
      AXIS_POSITION_16 : DWord;   // AXIS POSITION 16
      AXIS_POSITION_17 : DWord;   // AXIS POSITION 17
      AXIS_POSITION_18 : DWord;   // AXIS POSITION 18
      AXIS_POSITION_19 : DWord;   // AXIS POSITION 19
      AXIS_POSITION_20 : DWord;   // AXIS POSITION 20
   END_VAR
   VAR DB_SPECIFIC
      readDB { S7_SetPoint := 'True'} : "READ_AXES_POSITIONS_CH";
   END_VAR
   VAR
      FB2_Instance_1 { S7_SetPoint := 'True'} : "LBP_ReadVar";
      FB2_Instance_2 { S7_SetPoint := 'True'} : "LBP_ReadVar";
      FB2_Instance_3 { S7_SetPoint := 'True'} : "LBP_ReadVar";
   END_VAR
   VAR DB_SPECIFIC
      FAULT_COUNTER { S7_SetPoint := 'True'} : CTU_INT;
   END_VAR
   VAR_TEMP
      DB_NUMBER : DInt;   // DB NUMBER FOR ALARM AND HELP DECODING
      CHANNEL : UInt;   // CHANNEL NUMBER MAX. NUMBER=10
      FAULT : Bool;   // FAULT
      COUNT_ERRORS : Int;   // COUNT_ERRORS
   END_VAR
   VAR_TEMP   // added for the SCL form of the ladder/FBD networks
      _w1 : Bool;
   END_VAR
BEGIN

NETWORK
TITLE = READ INSTANCE DB
      L     DINO;
      +     10#800000;
      T     #DB_NUMBER;
      L     DINO;
      L     10#300;
      -I;
      T     #CHANNEL;



REGION Network 2: FAULT / CHANNELS READING FAULT
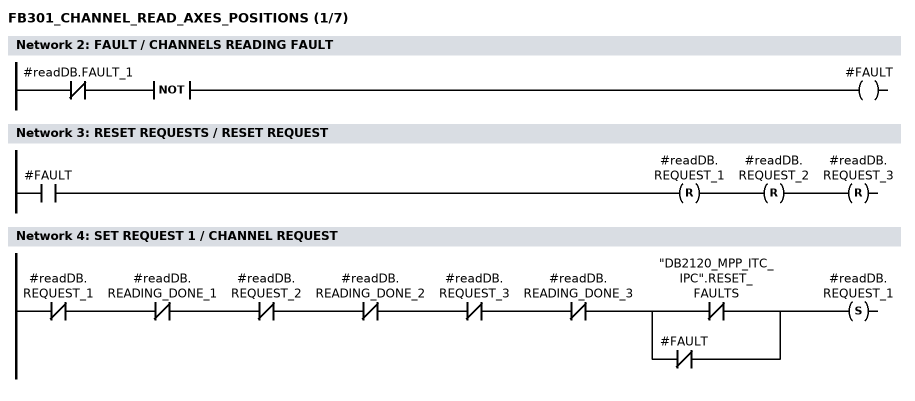
   RUNG wire#powerrail
      I_Contact( #readDB.FAULT_1 )
      Not()
      Coil( #FAULT )
   END_RUNG
   // the same network as SCL:
   #FAULT := NOT (NOT #readDB.FAULT_1);
END_REGION

REGION Network 3: RESET REQUESTS / RESET REQUEST
   RUNG wire#powerrail
      Contact( #FAULT )
      R_Coil( #readDB.REQUEST_1 )
      R_Coil( #readDB.REQUEST_2 )
      R_Coil( #readDB.REQUEST_3 )
   END_RUNG
   // the same network as SCL:
   IF #FAULT THEN
       #readDB.REQUEST_1 := FALSE;
       #readDB.REQUEST_2 := FALSE;
       #readDB.REQUEST_3 := FALSE;
   END_IF;
END_REGION

REGION Network 4: SET REQUEST 1 / CHANNEL REQUEST
   RUNG wire#powerrail
      I_Contact( #readDB.REQUEST_1 )
      I_Contact( #readDB.READING_DONE_1 )
      I_Contact( #readDB.REQUEST_2 )
      I_Contact( #readDB.READING_DONE_2 )
      I_Contact( #readDB.REQUEST_3 )
      I_Contact( #readDB.READING_DONE_3 )
      wire#w1
      I_Contact( "DB2120_MPP_ITC_IPC".RESET_FAULTS )
      wire#w2
      S_Coil( #readDB.REQUEST_1 )
   END_RUNG
   RUNG wire#w1
      I_Contact( #FAULT )
   END_RUNG wire#w2
   // the same network as SCL:
   IF NOT #readDB.REQUEST_1 AND NOT #readDB.READING_DONE_1 AND NOT #readDB.REQUEST_2 AND NOT #readDB.READING_DONE_2 AND NOT #readDB.REQUEST_3 AND NOT #readDB.READING_DONE_3 AND (NOT "DB2120_MPP_ITC_IPC".RESET_FAULTS OR NOT #FAULT) THEN
       #readDB.REQUEST_1 := TRUE;
   END_IF;
END_REGION

REGION Network 5: CALL FB2 GROUP 1 / READ AXES POSITIONS CHANNEL
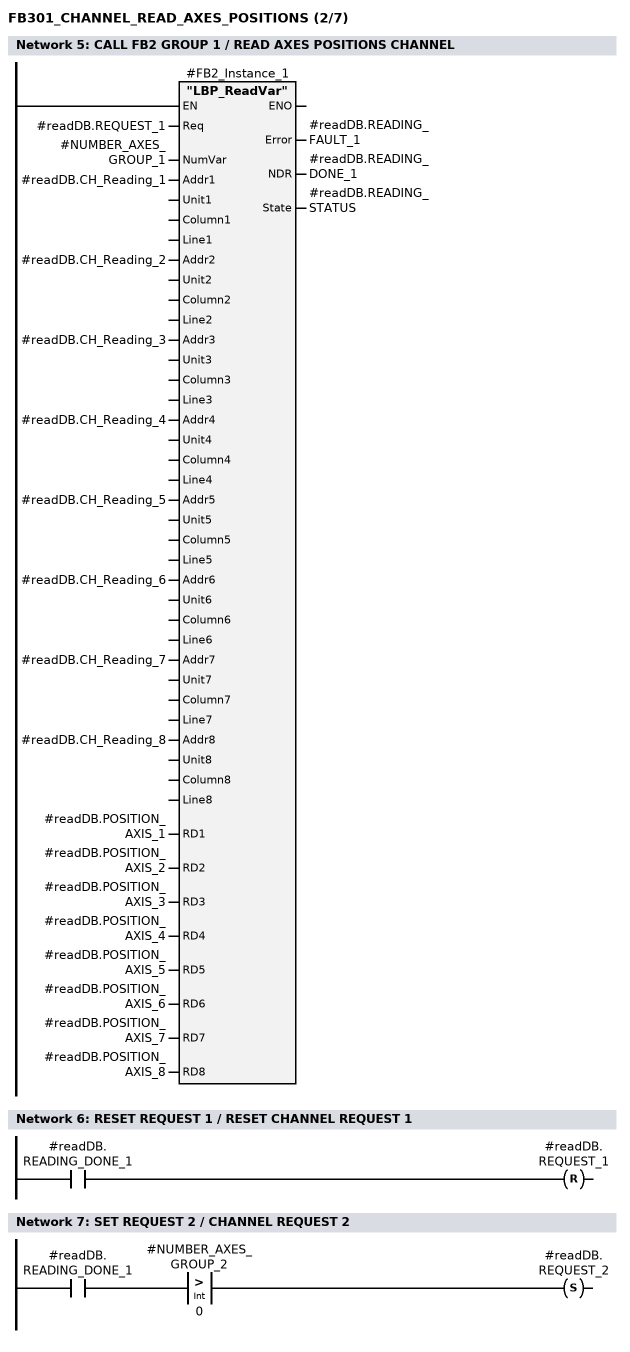
   RUNG wire#powerrail
      #FB2_Instance_1(Req := #readDB.REQUEST_1, NumVar := #NUMBER_AXES_GROUP_1, Addr1 := #readDB.CH_Reading_1, Unit1 :=, Column1 :=, Line1 :=, Addr2 := #readDB.CH_Reading_2, Unit2 :=, Column2 :=, Line2 :=, Addr3 := #readDB.CH_Reading_3, Unit3 :=, Column3 :=, Line3 :=, Addr4 := #readDB.CH_Reading_4, Unit4 :=, Column4 :=, Line4 :=, Addr5 := #readDB.CH_Reading_5, Unit5 :=, Column5 :=, Line5 :=, Addr6 := #readDB.CH_Reading_6, Unit6 :=, Column6 :=, Line6 :=, Addr7 := #readDB.CH_Reading_7, Unit7 :=, Column7 :=, Line7 :=, Addr8 := #readDB.CH_Reading_8, Unit8 :=, Column8 :=, Line8 :=, RD1 := #readDB.POSITION_AXIS_1, RD2 := #readDB.POSITION_AXIS_2, RD3 := #readDB.POSITION_AXIS_3, RD4 := #readDB.POSITION_AXIS_4, RD5 := #readDB.POSITION_AXIS_5, RD6 := #readDB.POSITION_AXIS_6, RD7 := #readDB.POSITION_AXIS_7, RD8 := #readDB.POSITION_AXIS_8, Error => #readDB.READING_FAULT_1, NDR => #readDB.READING_DONE_1, State => #readDB.READING_STATUS)
   END_RUNG
   // the same network as SCL:
   #FB2_Instance_1(Req := #readDB.REQUEST_1,   // "LBP_ReadVar"
                   NumVar := #NUMBER_AXES_GROUP_1,
                   Addr1 := #readDB.CH_Reading_1,
                   Addr2 := #readDB.CH_Reading_2,
                   Addr3 := #readDB.CH_Reading_3,
                   Addr4 := #readDB.CH_Reading_4,
                   Addr5 := #readDB.CH_Reading_5,
                   Addr6 := #readDB.CH_Reading_6,
                   Addr7 := #readDB.CH_Reading_7,
                   Addr8 := #readDB.CH_Reading_8,
                   RD1 := #readDB.POSITION_AXIS_1,
                   RD2 := #readDB.POSITION_AXIS_2,
                   RD3 := #readDB.POSITION_AXIS_3,
                   RD4 := #readDB.POSITION_AXIS_4,
                   RD5 := #readDB.POSITION_AXIS_5,
                   RD6 := #readDB.POSITION_AXIS_6,
                   RD7 := #readDB.POSITION_AXIS_7,
                   RD8 := #readDB.POSITION_AXIS_8,
                   Error => #readDB.READING_FAULT_1,
                   NDR => #readDB.READING_DONE_1,
                   State => #readDB.READING_STATUS);
END_REGION

REGION Network 6: RESET REQUEST 1 / RESET CHANNEL REQUEST 1
   RUNG wire#powerrail
      Contact( #readDB.READING_DONE_1 )
      R_Coil( #readDB.REQUEST_1 )
   END_RUNG
   // the same network as SCL:
   IF #readDB.READING_DONE_1 THEN #readDB.REQUEST_1 := FALSE; END_IF;
END_REGION

REGION Network 7: SET REQUEST 2 / CHANNEL REQUEST 2
   RUNG wire#powerrail
      Contact( #readDB.READING_DONE_1 )
      { S7_Templates := "SrcType := Int" } GT_Contact(in1 := #NUMBER_AXES_GROUP_2, in2 := 0)
      S_Coil( #readDB.REQUEST_2 )
   END_RUNG
   // the same network as SCL:
   IF #readDB.READING_DONE_1 AND (#NUMBER_AXES_GROUP_2 > 0) THEN #readDB.REQUEST_2 := TRUE; END_IF;
END_REGION

REGION Network 8: CALL FB2 GROUP 2 / READ AXES POSITIONS CHANNEL
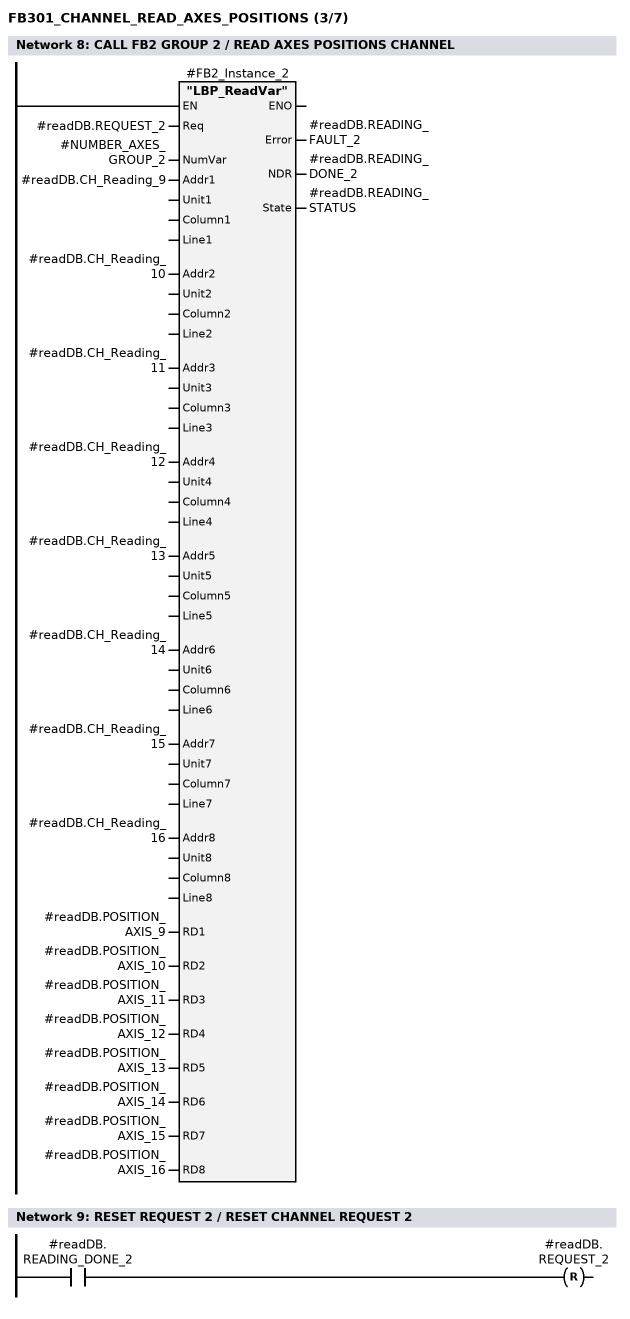
   RUNG wire#powerrail
      #FB2_Instance_2(Req := #readDB.REQUEST_2, NumVar := #NUMBER_AXES_GROUP_2, Addr1 := #readDB.CH_Reading_9, Unit1 :=, Column1 :=, Line1 :=, Addr2 := #readDB.CH_Reading_10, Unit2 :=, Column2 :=, Line2 :=, Addr3 := #readDB.CH_Reading_11, Unit3 :=, Column3 :=, Line3 :=, Addr4 := #readDB.CH_Reading_12, Unit4 :=, Column4 :=, Line4 :=, Addr5 := #readDB.CH_Reading_13, Unit5 :=, Column5 :=, Line5 :=, Addr6 := #readDB.CH_Reading_14, Unit6 :=, Column6 :=, Line6 :=, Addr7 := #readDB.CH_Reading_15, Unit7 :=, Column7 :=, Line7 :=, Addr8 := #readDB.CH_Reading_16, Unit8 :=, Column8 :=, Line8 :=, RD1 := #readDB.POSITION_AXIS_9, RD2 := #readDB.POSITION_AXIS_10, RD3 := #readDB.POSITION_AXIS_11, RD4 := #readDB.POSITION_AXIS_12, RD5 := #readDB.POSITION_AXIS_13, RD6 := #readDB.POSITION_AXIS_14, RD7 := #readDB.POSITION_AXIS_15, RD8 := #readDB.POSITION_AXIS_16, Error => #readDB.READING_FAULT_2, NDR => #readDB.READING_DONE_2, State => #readDB.READING_STATUS)
   END_RUNG
   // the same network as SCL:
   #FB2_Instance_2(Req := #readDB.REQUEST_2,   // "LBP_ReadVar"
                   NumVar := #NUMBER_AXES_GROUP_2,
                   Addr1 := #readDB.CH_Reading_9,
                   Addr2 := #readDB.CH_Reading_10,
                   Addr3 := #readDB.CH_Reading_11,
                   Addr4 := #readDB.CH_Reading_12,
                   Addr5 := #readDB.CH_Reading_13,
                   Addr6 := #readDB.CH_Reading_14,
                   Addr7 := #readDB.CH_Reading_15,
                   Addr8 := #readDB.CH_Reading_16,
                   RD1 := #readDB.POSITION_AXIS_9,
                   RD2 := #readDB.POSITION_AXIS_10,
                   RD3 := #readDB.POSITION_AXIS_11,
                   RD4 := #readDB.POSITION_AXIS_12,
                   RD5 := #readDB.POSITION_AXIS_13,
                   RD6 := #readDB.POSITION_AXIS_14,
                   RD7 := #readDB.POSITION_AXIS_15,
                   RD8 := #readDB.POSITION_AXIS_16,
                   Error => #readDB.READING_FAULT_2,
                   NDR => #readDB.READING_DONE_2,
                   State => #readDB.READING_STATUS);
END_REGION

REGION Network 9: RESET REQUEST 2 / RESET CHANNEL REQUEST 2
   RUNG wire#powerrail
      Contact( #readDB.READING_DONE_2 )
      R_Coil( #readDB.REQUEST_2 )
   END_RUNG
   // the same network as SCL:
   IF #readDB.READING_DONE_2 THEN #readDB.REQUEST_2 := FALSE; END_IF;
END_REGION

REGION Network 10: SET REQUEST 3 / RESET CHANNEL REQUEST 2
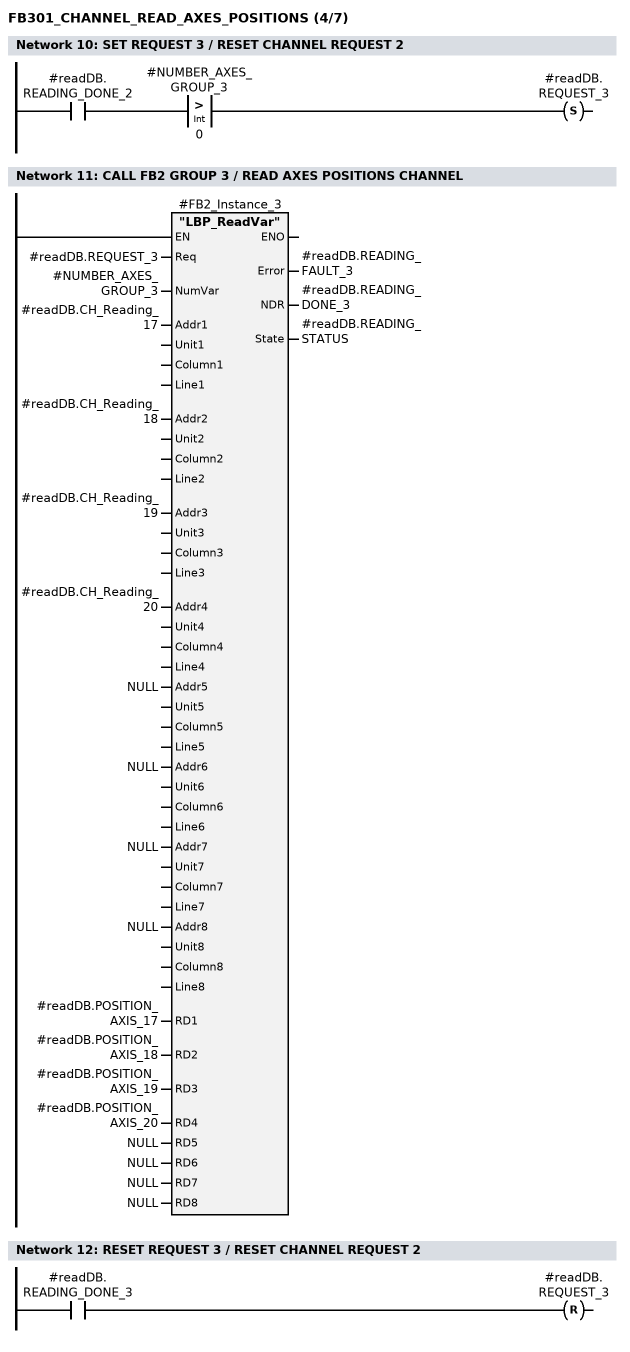
   RUNG wire#powerrail
      Contact( #readDB.READING_DONE_2 )
      { S7_Templates := "SrcType := Int" } GT_Contact(in1 := #NUMBER_AXES_GROUP_3, in2 := 0)
      S_Coil( #readDB.REQUEST_3 )
   END_RUNG
   // the same network as SCL:
   IF #readDB.READING_DONE_2 AND (#NUMBER_AXES_GROUP_3 > 0) THEN #readDB.REQUEST_3 := TRUE; END_IF;
END_REGION

REGION Network 11: CALL FB2 GROUP 3 / READ AXES POSITIONS CHANNEL
   RUNG wire#powerrail
      #FB2_Instance_3(Req := #readDB.REQUEST_3, NumVar := #NUMBER_AXES_GROUP_3, Addr1 := #readDB.CH_Reading_17, Unit1 :=, Column1 :=, Line1 :=, Addr2 := #readDB.CH_Reading_18, Unit2 :=, Column2 :=, Line2 :=, Addr3 := #readDB.CH_Reading_19, Unit3 :=, Column3 :=, Line3 :=, Addr4 := #readDB.CH_Reading_20, Unit4 :=, Column4 :=, Line4 :=, Addr5 := NULL, Unit5 :=, Column5 :=, Line5 :=, Addr6 := NULL, Unit6 :=, Column6 :=, Line6 :=, Addr7 := NULL, Unit7 :=, Column7 :=, Line7 :=, Addr8 := NULL, Unit8 :=, Column8 :=, Line8 :=, RD1 := #readDB.POSITION_AXIS_17, RD2 := #readDB.POSITION_AXIS_18, RD3 := #readDB.POSITION_AXIS_19, RD4 := #readDB.POSITION_AXIS_20, RD5 := NULL, RD6 := NULL, RD7 := NULL, RD8 := NULL, Error => #readDB.READING_FAULT_3, NDR => #readDB.READING_DONE_3, State => #readDB.READING_STATUS)
   END_RUNG
   // the same network as SCL:
   #FB2_Instance_3(Req := #readDB.REQUEST_3,   // "LBP_ReadVar"
                   NumVar := #NUMBER_AXES_GROUP_3,
                   Addr1 := #readDB.CH_Reading_17,
                   Addr2 := #readDB.CH_Reading_18,
                   Addr3 := #readDB.CH_Reading_19,
                   Addr4 := #readDB.CH_Reading_20,
                   Addr5 := NULL,
                   Addr6 := NULL,
                   Addr7 := NULL,
                   Addr8 := NULL,
                   RD1 := #readDB.POSITION_AXIS_17,
                   RD2 := #readDB.POSITION_AXIS_18,
                   RD3 := #readDB.POSITION_AXIS_19,
                   RD4 := #readDB.POSITION_AXIS_20,
                   RD5 := NULL,
                   RD6 := NULL,
                   RD7 := NULL,
                   RD8 := NULL,
                   Error => #readDB.READING_FAULT_3,
                   NDR => #readDB.READING_DONE_3,
                   State => #readDB.READING_STATUS);
END_REGION

REGION Network 12: RESET REQUEST 3 / RESET CHANNEL REQUEST 2
   RUNG wire#powerrail
      Contact( #readDB.READING_DONE_3 )
      R_Coil( #readDB.REQUEST_3 )
   END_RUNG
   // the same network as SCL:
   IF #readDB.READING_DONE_3 THEN #readDB.REQUEST_3 := FALSE; END_IF;
END_REGION

REGION Network 13: MOVE POSITIONS / AXES POSITIONS
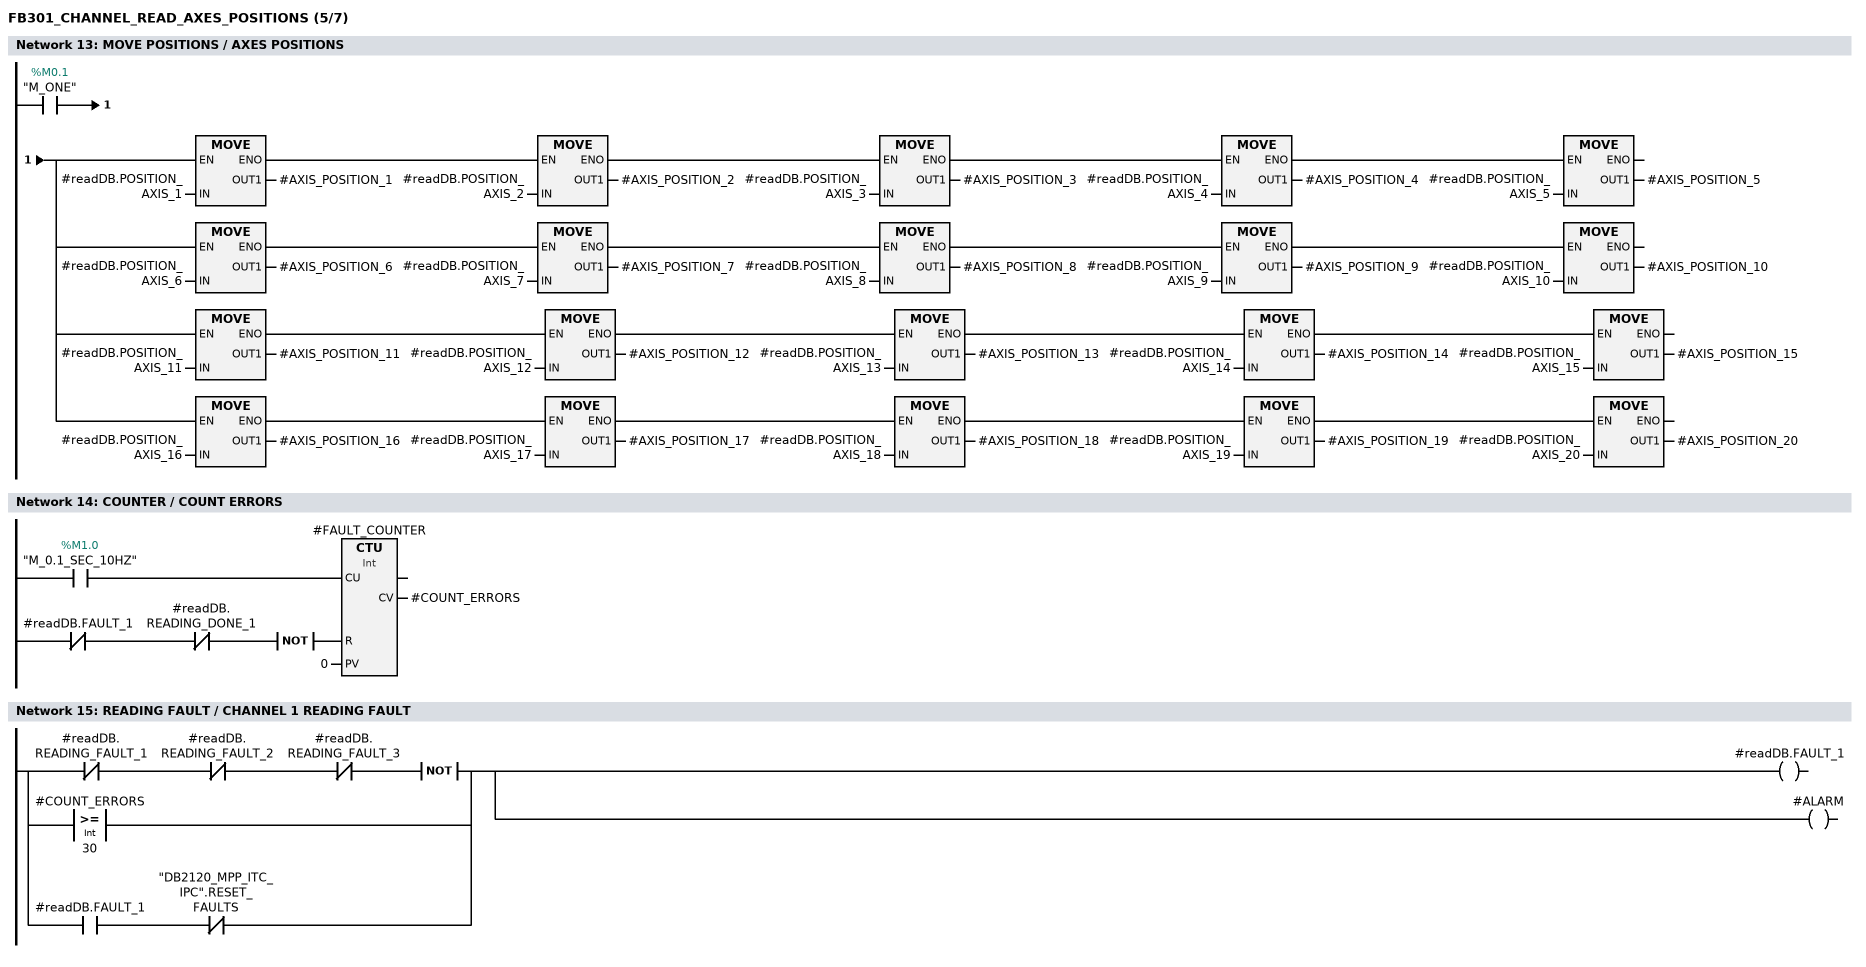
   RUNG wire#powerrail
      Contact( "M_ONE" )
      wire#w1
      { S7_GenerateENO := "TRUE" } Move(in := #readDB.POSITION_AXIS_1, out1 => #AXIS_POSITION_1)
      { S7_GenerateENO := "TRUE" } Move(in := #readDB.POSITION_AXIS_2, out1 => #AXIS_POSITION_2)
      { S7_GenerateENO := "TRUE" } Move(in := #readDB.POSITION_AXIS_3, out1 => #AXIS_POSITION_3)
      { S7_GenerateENO := "TRUE" } Move(in := #readDB.POSITION_AXIS_4, out1 => #AXIS_POSITION_4)
      { S7_GenerateENO := "TRUE" } Move(in := #readDB.POSITION_AXIS_5, out1 => #AXIS_POSITION_5)
   END_RUNG
   RUNG wire#w1
      { S7_GenerateENO := "TRUE" } Move(in := #readDB.POSITION_AXIS_6, out1 => #AXIS_POSITION_6)
      { S7_GenerateENO := "TRUE" } Move(in := #readDB.POSITION_AXIS_7, out1 => #AXIS_POSITION_7)
      { S7_GenerateENO := "TRUE" } Move(in := #readDB.POSITION_AXIS_8, out1 => #AXIS_POSITION_8)
      { S7_GenerateENO := "TRUE" } Move(in := #readDB.POSITION_AXIS_9, out1 => #AXIS_POSITION_9)
      { S7_GenerateENO := "TRUE" } Move(in := #readDB.POSITION_AXIS_10, out1 => #AXIS_POSITION_10)
   END_RUNG
   RUNG wire#w1
      { S7_GenerateENO := "TRUE" } Move(in := #readDB.POSITION_AXIS_11, out1 => #AXIS_POSITION_11)
      { S7_GenerateENO := "TRUE" } Move(in := #readDB.POSITION_AXIS_12, out1 => #AXIS_POSITION_12)
      { S7_GenerateENO := "TRUE" } Move(in := #readDB.POSITION_AXIS_13, out1 => #AXIS_POSITION_13)
      { S7_GenerateENO := "TRUE" } Move(in := #readDB.POSITION_AXIS_14, out1 => #AXIS_POSITION_14)
      { S7_GenerateENO := "TRUE" } Move(in := #readDB.POSITION_AXIS_15, out1 => #AXIS_POSITION_15)
   END_RUNG
   RUNG wire#w1
      { S7_GenerateENO := "TRUE" } Move(in := #readDB.POSITION_AXIS_16, out1 => #AXIS_POSITION_16)
      { S7_GenerateENO := "TRUE" } Move(in := #readDB.POSITION_AXIS_17, out1 => #AXIS_POSITION_17)
      { S7_GenerateENO := "TRUE" } Move(in := #readDB.POSITION_AXIS_18, out1 => #AXIS_POSITION_18)
      { S7_GenerateENO := "TRUE" } Move(in := #readDB.POSITION_AXIS_19, out1 => #AXIS_POSITION_19)
      { S7_GenerateENO := "TRUE" } Move(in := #readDB.POSITION_AXIS_20, out1 => #AXIS_POSITION_20)
   END_RUNG
   // the same network as SCL:
   // ENO of a box is taken as its EN; it also drops when the box reports an error
   IF "M_ONE" THEN
       #AXIS_POSITION_1 := #readDB.POSITION_AXIS_1;
       #AXIS_POSITION_2 := #readDB.POSITION_AXIS_2;
       #AXIS_POSITION_3 := #readDB.POSITION_AXIS_3;
       #AXIS_POSITION_4 := #readDB.POSITION_AXIS_4;
       #AXIS_POSITION_5 := #readDB.POSITION_AXIS_5;
       #AXIS_POSITION_6 := #readDB.POSITION_AXIS_6;
       #AXIS_POSITION_7 := #readDB.POSITION_AXIS_7;
       #AXIS_POSITION_8 := #readDB.POSITION_AXIS_8;
       #AXIS_POSITION_9 := #readDB.POSITION_AXIS_9;
       #AXIS_POSITION_10 := #readDB.POSITION_AXIS_10;
       #AXIS_POSITION_11 := #readDB.POSITION_AXIS_11;
       #AXIS_POSITION_12 := #readDB.POSITION_AXIS_12;
       #AXIS_POSITION_13 := #readDB.POSITION_AXIS_13;
       #AXIS_POSITION_14 := #readDB.POSITION_AXIS_14;
       #AXIS_POSITION_15 := #readDB.POSITION_AXIS_15;
       #AXIS_POSITION_16 := #readDB.POSITION_AXIS_16;
       #AXIS_POSITION_17 := #readDB.POSITION_AXIS_17;
       #AXIS_POSITION_18 := #readDB.POSITION_AXIS_18;
       #AXIS_POSITION_19 := #readDB.POSITION_AXIS_19;
       #AXIS_POSITION_20 := #readDB.POSITION_AXIS_20;
   END_IF;
END_REGION

REGION Network 14: COUNTER / COUNT ERRORS
   RUNG wire#powerrail
      Contact( "M_0.1_SEC_10HZ" )
      { S7_Templates := "value_type := Int" } #FAULT_COUNTER.CTU(r := wire#w1, pv := 0, cv => #COUNT_ERRORS)
   END_RUNG
   RUNG wire#powerrail
      I_Contact( #readDB.FAULT_1 )
      I_Contact( #readDB.READING_DONE_1 )
      Not()
   END_RUNG wire#w1
   // the same network as SCL:
   #FAULT_COUNTER(CU := "M_0.1_SEC_10HZ",   // CTU
                  R := NOT (NOT #readDB.FAULT_1 AND NOT #readDB.READING_DONE_1),
                  PV := 0,
                  CV => #COUNT_ERRORS);
END_REGION

REGION Network 15: READING FAULT / CHANNEL 1 READING FAULT
   RUNG wire#powerrail
      I_Contact( #readDB.READING_FAULT_1 )
      I_Contact( #readDB.READING_FAULT_2 )
      I_Contact( #readDB.READING_FAULT_3 )
      Not()
      wire#w1
      Coil( #readDB.FAULT_1 )
   END_RUNG
   RUNG wire#powerrail
      { S7_Templates := "SrcType := Int" } GE_Contact(in1 := #COUNT_ERRORS, in2 := 30)
   END_RUNG wire#w1
   RUNG wire#powerrail
      Contact( #readDB.FAULT_1 )
      I_Contact( "DB2120_MPP_ITC_IPC".RESET_FAULTS )
   END_RUNG wire#w1
   RUNG wire#w1
      Coil( #ALARM )
   END_RUNG
   // the same network as SCL:
   #readDB.FAULT_1 := NOT (NOT #readDB.READING_FAULT_1 AND NOT #readDB.READING_FAULT_2 AND NOT #readDB.READING_FAULT_3) OR (#COUNT_ERRORS >= 30) OR (#readDB.FAULT_1 AND NOT "DB2120_MPP_ITC_IPC".RESET_FAULTS);
   #ALARM := #readDB.FAULT_1;
END_REGION

REGION Network 16: IMMEDIATE STOP AND STOP END OF CYCLE ALARMS / IMMEDIATE STOP ALARMS
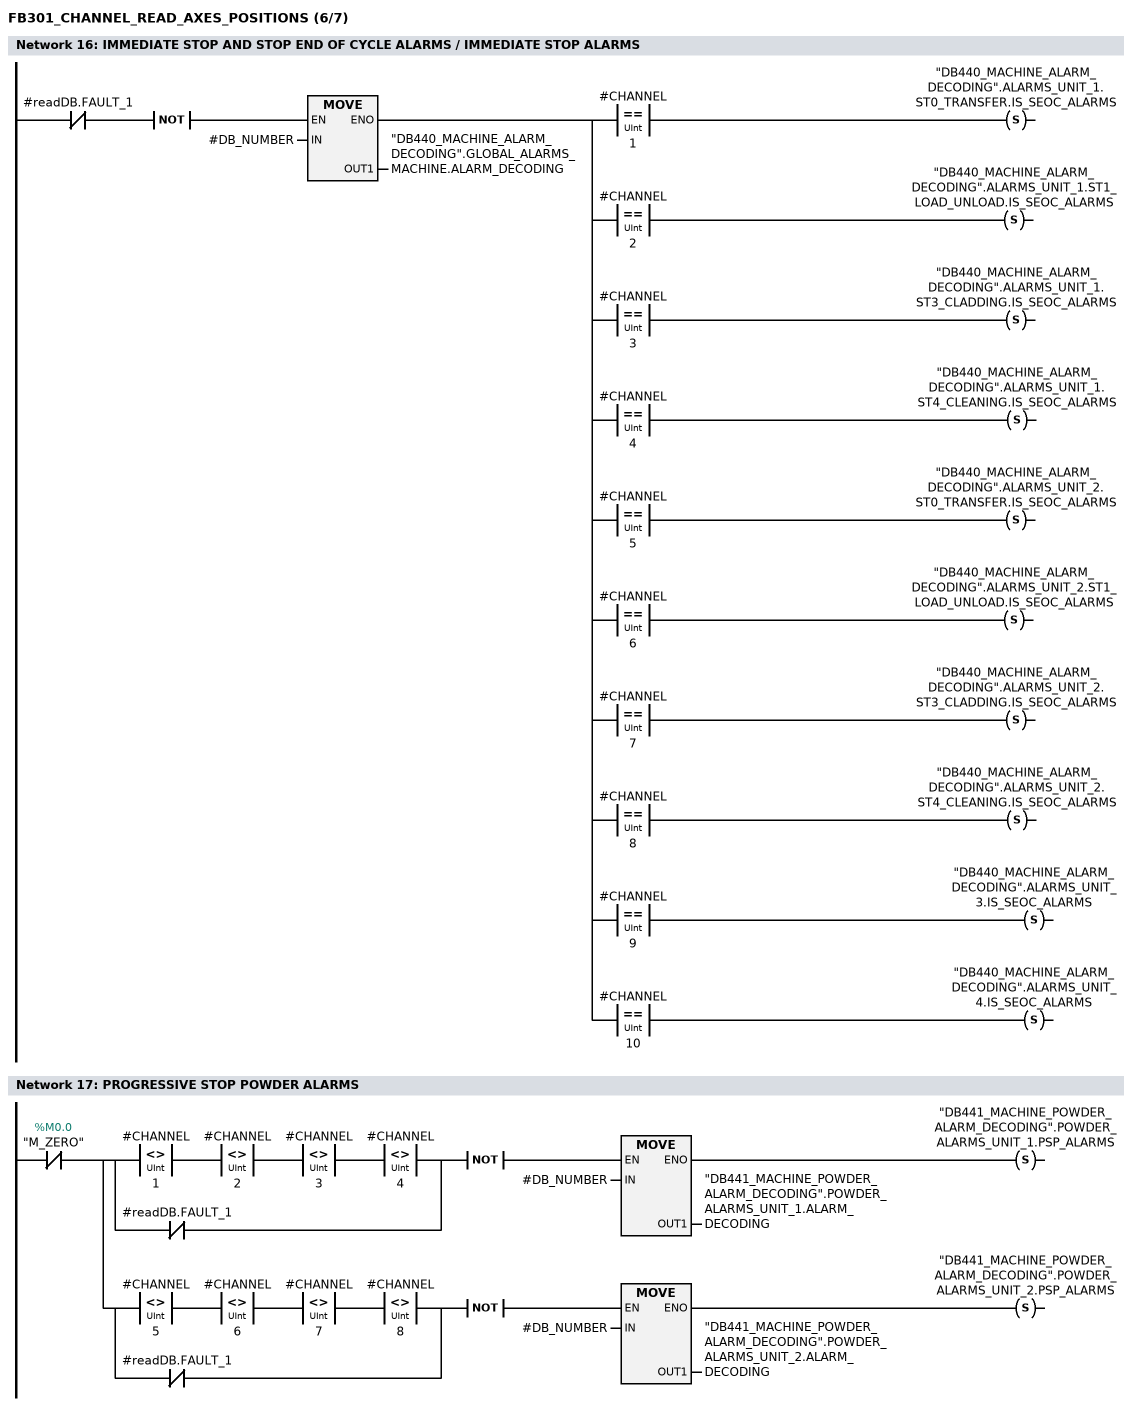
   RUNG wire#powerrail
      I_Contact( #readDB.FAULT_1 )
      Not()
      { S7_GenerateENO := "TRUE" } Move(in := #DB_NUMBER, out1 => "DB440_MACHINE_ALARM_DECODING".GLOBAL_ALARMS_MACHINE.ALARM_DECODING)
      wire#w1
      { S7_Templates := "SrcType := UInt" } EQ_Contact(in1 := #CHANNEL, in2 := 1)
      S_Coil( "DB440_MACHINE_ALARM_DECODING".ALARMS_UNIT_1.ST0_TRANSFER.IS_SEOC_ALARMS )
   END_RUNG
   RUNG wire#w1
      { S7_Templates := "SrcType := UInt" } EQ_Contact(in1 := #CHANNEL, in2 := 2)
      S_Coil( "DB440_MACHINE_ALARM_DECODING".ALARMS_UNIT_1.ST1_LOAD_UNLOAD.IS_SEOC_ALARMS )
   END_RUNG
   RUNG wire#w1
      { S7_Templates := "SrcType := UInt" } EQ_Contact(in1 := #CHANNEL, in2 := 3)
      S_Coil( "DB440_MACHINE_ALARM_DECODING".ALARMS_UNIT_1.ST3_CLADDING.IS_SEOC_ALARMS )
   END_RUNG
   RUNG wire#w1
      { S7_Templates := "SrcType := UInt" } EQ_Contact(in1 := #CHANNEL, in2 := 4)
      S_Coil( "DB440_MACHINE_ALARM_DECODING".ALARMS_UNIT_1.ST4_CLEANING.IS_SEOC_ALARMS )
   END_RUNG
   RUNG wire#w1
      { S7_Templates := "SrcType := UInt" } EQ_Contact(in1 := #CHANNEL, in2 := 5)
      S_Coil( "DB440_MACHINE_ALARM_DECODING".ALARMS_UNIT_2.ST0_TRANSFER.IS_SEOC_ALARMS )
   END_RUNG
   RUNG wire#w1
      { S7_Templates := "SrcType := UInt" } EQ_Contact(in1 := #CHANNEL, in2 := 6)
      S_Coil( "DB440_MACHINE_ALARM_DECODING".ALARMS_UNIT_2.ST1_LOAD_UNLOAD.IS_SEOC_ALARMS )
   END_RUNG
   RUNG wire#w1
      { S7_Templates := "SrcType := UInt" } EQ_Contact(in1 := #CHANNEL, in2 := 7)
      S_Coil( "DB440_MACHINE_ALARM_DECODING".ALARMS_UNIT_2.ST3_CLADDING.IS_SEOC_ALARMS )
   END_RUNG
   RUNG wire#w1
      { S7_Templates := "SrcType := UInt" } EQ_Contact(in1 := #CHANNEL, in2 := 8)
      S_Coil( "DB440_MACHINE_ALARM_DECODING".ALARMS_UNIT_2.ST4_CLEANING.IS_SEOC_ALARMS )
   END_RUNG
   RUNG wire#w1
      { S7_Templates := "SrcType := UInt" } EQ_Contact(in1 := #CHANNEL, in2 := 9)
      S_Coil( "DB440_MACHINE_ALARM_DECODING".ALARMS_UNIT_3.IS_SEOC_ALARMS )
   END_RUNG
   RUNG wire#w1
      { S7_Templates := "SrcType := UInt" } EQ_Contact(in1 := #CHANNEL, in2 := 10)
      S_Coil( "DB440_MACHINE_ALARM_DECODING".ALARMS_UNIT_4.IS_SEOC_ALARMS )
   END_RUNG
   // the same network as SCL:
   // ENO of a box is taken as its EN; it also drops when the box reports an error
   #_w1 := NOT (NOT #readDB.FAULT_1);
   IF #_w1 THEN "DB440_MACHINE_ALARM_DECODING".GLOBAL_ALARMS_MACHINE.ALARM_DECODING := #DB_NUMBER; END_IF;
   IF #_w1 AND (#CHANNEL = 1) THEN
       "DB440_MACHINE_ALARM_DECODING".ALARMS_UNIT_1.ST0_TRANSFER.IS_SEOC_ALARMS := TRUE;
   END_IF;
   IF #_w1 AND (#CHANNEL = 2) THEN
       "DB440_MACHINE_ALARM_DECODING".ALARMS_UNIT_1.ST1_LOAD_UNLOAD.IS_SEOC_ALARMS := TRUE;
   END_IF;
   IF #_w1 AND (#CHANNEL = 3) THEN
       "DB440_MACHINE_ALARM_DECODING".ALARMS_UNIT_1.ST3_CLADDING.IS_SEOC_ALARMS := TRUE;
   END_IF;
   IF #_w1 AND (#CHANNEL = 4) THEN
       "DB440_MACHINE_ALARM_DECODING".ALARMS_UNIT_1.ST4_CLEANING.IS_SEOC_ALARMS := TRUE;
   END_IF;
   IF #_w1 AND (#CHANNEL = 5) THEN
       "DB440_MACHINE_ALARM_DECODING".ALARMS_UNIT_2.ST0_TRANSFER.IS_SEOC_ALARMS := TRUE;
   END_IF;
   IF #_w1 AND (#CHANNEL = 6) THEN
       "DB440_MACHINE_ALARM_DECODING".ALARMS_UNIT_2.ST1_LOAD_UNLOAD.IS_SEOC_ALARMS := TRUE;
   END_IF;
   IF #_w1 AND (#CHANNEL = 7) THEN
       "DB440_MACHINE_ALARM_DECODING".ALARMS_UNIT_2.ST3_CLADDING.IS_SEOC_ALARMS := TRUE;
   END_IF;
   IF #_w1 AND (#CHANNEL = 8) THEN
       "DB440_MACHINE_ALARM_DECODING".ALARMS_UNIT_2.ST4_CLEANING.IS_SEOC_ALARMS := TRUE;
   END_IF;
   IF #_w1 AND (#CHANNEL = 9) THEN
       "DB440_MACHINE_ALARM_DECODING".ALARMS_UNIT_3.IS_SEOC_ALARMS := TRUE;
   END_IF;
   IF #_w1 AND (#CHANNEL = 10) THEN
       "DB440_MACHINE_ALARM_DECODING".ALARMS_UNIT_4.IS_SEOC_ALARMS := TRUE;
   END_IF;
END_REGION

REGION Network 17: PROGRESSIVE STOP POWDER ALARMS
   RUNG wire#powerrail
      I_Contact( "M_ZERO" )
      wire#w1
      { S7_Templates := "SrcType := UInt" } NE_Contact(in1 := #CHANNEL, in2 := 1)
      { S7_Templates := "SrcType := UInt" } NE_Contact(in1 := #CHANNEL, in2 := 2)
      { S7_Templates := "SrcType := UInt" } NE_Contact(in1 := #CHANNEL, in2 := 3)
      { S7_Templates := "SrcType := UInt" } NE_Contact(in1 := #CHANNEL, in2 := 4)
      wire#w2
      Not()
      { S7_GenerateENO := "TRUE" } Move(in := #DB_NUMBER, out1 => "DB441_MACHINE_POWDER_ALARM_DECODING".POWDER_ALARMS_UNIT_1.ALARM_DECODING)
      S_Coil( "DB441_MACHINE_POWDER_ALARM_DECODING".POWDER_ALARMS_UNIT_1.PSP_ALARMS )
   END_RUNG
   RUNG wire#w1
      I_Contact( #readDB.FAULT_1 )
   END_RUNG wire#w2
   RUNG wire#w1
      { S7_Templates := "SrcType := UInt" } NE_Contact(in1 := #CHANNEL, in2 := 5)
      { S7_Templates := "SrcType := UInt" } NE_Contact(in1 := #CHANNEL, in2 := 6)
      { S7_Templates := "SrcType := UInt" } NE_Contact(in1 := #CHANNEL, in2 := 7)
      { S7_Templates := "SrcType := UInt" } NE_Contact(in1 := #CHANNEL, in2 := 8)
      wire#w3
      Not()
      { S7_GenerateENO := "TRUE" } Move(in := #DB_NUMBER, out1 => "DB441_MACHINE_POWDER_ALARM_DECODING".POWDER_ALARMS_UNIT_2.ALARM_DECODING)
      S_Coil( "DB441_MACHINE_POWDER_ALARM_DECODING".POWDER_ALARMS_UNIT_2.PSP_ALARMS )
   END_RUNG
   RUNG wire#w1
      I_Contact( #readDB.FAULT_1 )
   END_RUNG wire#w3
   // the same network as SCL:
   // ENO of a box is taken as its EN; it also drops when the box reports an error
   IF NOT (NOT "M_ZERO" AND (((#CHANNEL <> 1) AND (#CHANNEL <> 2) AND (#CHANNEL <> 3) AND (#CHANNEL <> 4)) OR NOT #readDB.FAULT_1)) THEN
       "DB441_MACHINE_POWDER_ALARM_DECODING".POWDER_ALARMS_UNIT_1.ALARM_DECODING := #DB_NUMBER;
       "DB441_MACHINE_POWDER_ALARM_DECODING".POWDER_ALARMS_UNIT_1.PSP_ALARMS := TRUE;
   END_IF;
   IF NOT (NOT "M_ZERO" AND (((#CHANNEL <> 5) AND (#CHANNEL <> 6) AND (#CHANNEL <> 7) AND (#CHANNEL <> 8)) OR NOT #readDB.FAULT_1)) THEN
       "DB441_MACHINE_POWDER_ALARM_DECODING".POWDER_ALARMS_UNIT_2.ALARM_DECODING := #DB_NUMBER;
       "DB441_MACHINE_POWDER_ALARM_DECODING".POWDER_ALARMS_UNIT_2.PSP_ALARMS := TRUE;
   END_IF;
END_REGION

REGION Network 18: PROGRAMMING ALARM
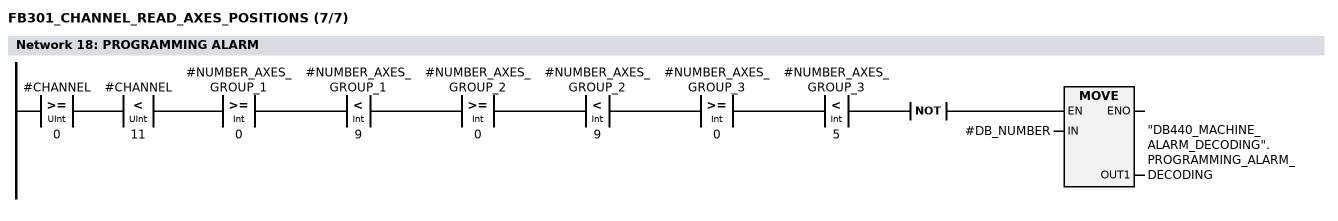
   RUNG wire#powerrail
      { S7_Templates := "SrcType := UInt" } GE_Contact(in1 := #CHANNEL, in2 := 0)
      { S7_Templates := "SrcType := UInt" } LT_Contact(in1 := #CHANNEL, in2 := 11)
      { S7_Templates := "SrcType := Int" } GE_Contact(in1 := #NUMBER_AXES_GROUP_1, in2 := 0)
      { S7_Templates := "SrcType := Int" } LT_Contact(in1 := #NUMBER_AXES_GROUP_1, in2 := 9)
      { S7_Templates := "SrcType := Int" } GE_Contact(in1 := #NUMBER_AXES_GROUP_2, in2 := 0)
      { S7_Templates := "SrcType := Int" } LT_Contact(in1 := #NUMBER_AXES_GROUP_2, in2 := 9)
      { S7_Templates := "SrcType := Int" } GE_Contact(in1 := #NUMBER_AXES_GROUP_3, in2 := 0)
      { S7_Templates := "SrcType := Int" } LT_Contact(in1 := #NUMBER_AXES_GROUP_3, in2 := 5)
      Not()
      Move(in := #DB_NUMBER, out1 => "DB440_MACHINE_ALARM_DECODING".PROGRAMMING_ALARM_DECODING)
   END_RUNG
   // the same network as SCL:
   IF NOT ((#CHANNEL >= 0) AND (#CHANNEL < 11) AND (#NUMBER_AXES_GROUP_1 >= 0) AND (#NUMBER_AXES_GROUP_1 < 9) AND (#NUMBER_AXES_GROUP_2 >= 0) AND (#NUMBER_AXES_GROUP_2 < 9) AND (#NUMBER_AXES_GROUP_3 >= 0) AND (#NUMBER_AXES_GROUP_3 < 5)) THEN
       "DB440_MACHINE_ALARM_DECODING".PROGRAMMING_ALARM_DECODING := #DB_NUMBER;
   END_IF;
END_REGION
END_FUNCTION_BLOCK

FUNCTION_BLOCK "FB311_CHANNEL_PROGRAM_SELECTION"   // FB311, LAD
{ S7_Optimized_Access := 'FALSE' }
AUTHOR : ETXETAR
VERSION : 1.0
// stored: AutoNumber false, IsIECCheckEnabled false, SetENOAutomatically false, UDAEnableTagReadback false
   VAR_INPUT
      CH_MODE_GROUP : Int;   // CHANNEL MODE GROUP
      REQUEST : Bool;   // REQUEST
      SEQ_RUNNING : Bool;   // MACHINE SEQUENCE RUNNING
      MCH_RESET : Bool;   // MACHINE RESET
   END_VAR
   VAR_OUTPUT
      ALARM : Bool;
   END_VAR
   VAR_IN_OUT
      channelDB : "LBP_typeChanX";
   END_VAR
   VAR DB_SPECIFIC
      interlocksDB { S7_SetPoint := 'True'} : "CNC_PLC_INT_CH";
   END_VAR
   VAR
      FB7_INSTANCE { S7_SetPoint := 'True'} : "LBP_ReqPIService";
   END_VAR
   VAR_TEMP
      DB_NUMBER : DInt;   // DB NUMBER FOR ALARM AND HELP DECODING
      CHANNEL : Int;   // CHANNEL NUMBER MAX. NUMBER=10
   END_VAR
   VAR_TEMP   // added for the SCL form of the ladder/FBD networks
      _w1 : Bool;
      _w2 : Bool;
   END_VAR
BEGIN

NETWORK
TITLE = READ INSTANCE DB
      L     DINO;
      +     10#800000;
      T     #DB_NUMBER;
      L     DINO;
      L     10#310;
      -I;
      T     #CHANNEL;



REGION Network 2: RESET SELECTION
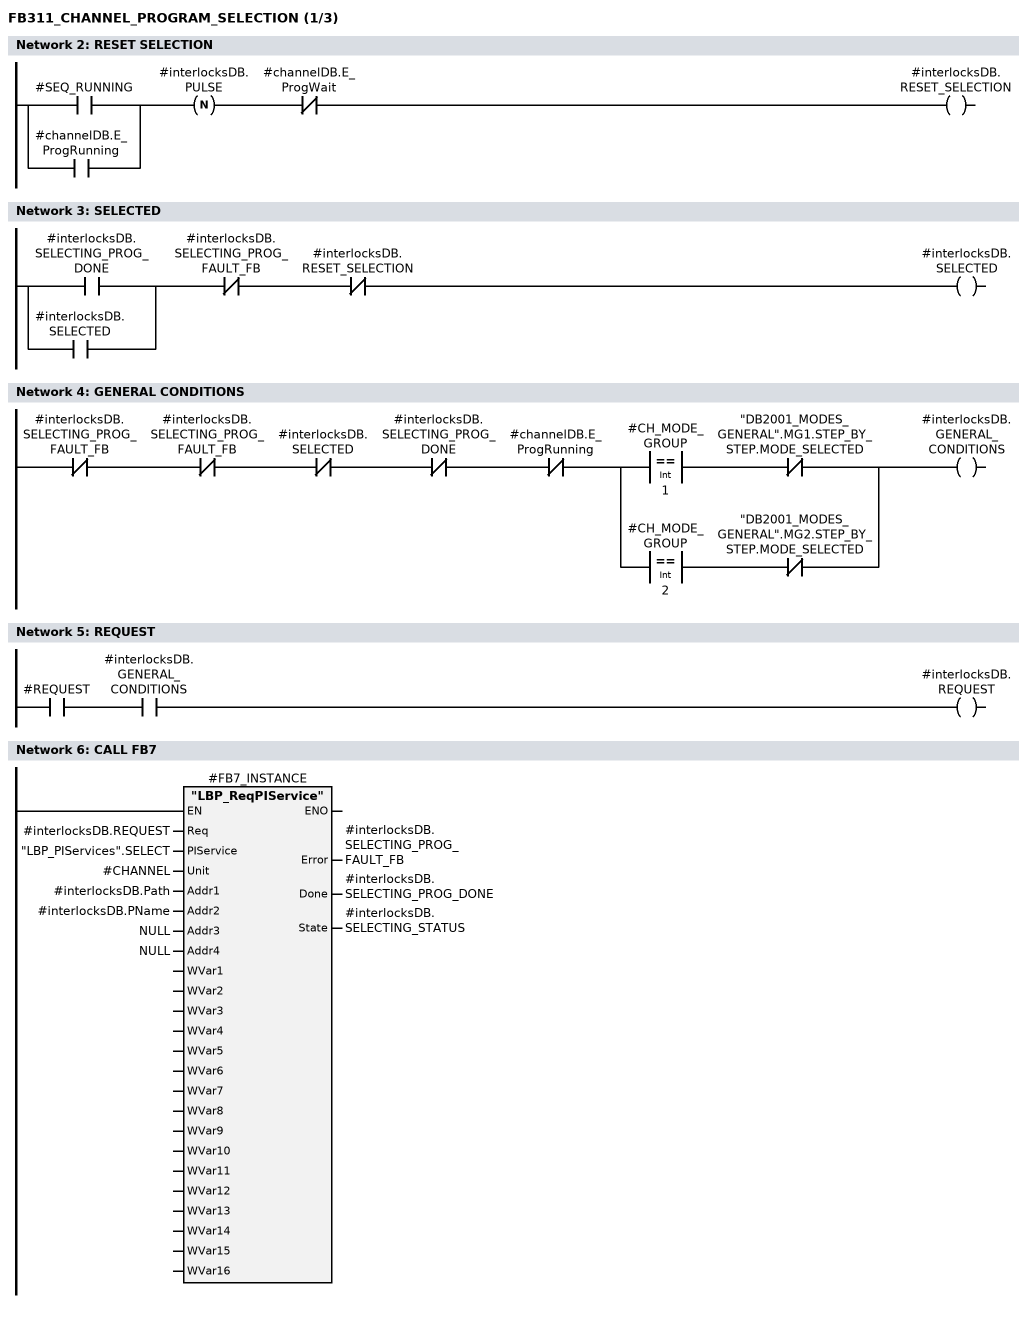
   RUNG wire#powerrail
      Contact( #SEQ_RUNNING )
      wire#w1
      N_Trig( #interlocksDB.PULSE )
      I_Contact( #channelDB.E_ProgWait )
      Coil( #interlocksDB.RESET_SELECTION )
   END_RUNG
   RUNG wire#powerrail
      Contact( #channelDB.E_ProgRunning )
   END_RUNG wire#w1
   // the same network as SCL:
   #_w1 := #SEQ_RUNNING OR #channelDB.E_ProgRunning;
   #_w2 := NOT #_w1 AND #interlocksDB.PULSE;   // falling edge
   #interlocksDB.PULSE := #_w1;
   #interlocksDB.RESET_SELECTION := #_w2 AND NOT #channelDB.E_ProgWait;
END_REGION

REGION Network 3: SELECTED
   RUNG wire#powerrail
      Contact( #interlocksDB.SELECTING_PROG_DONE )
      wire#w1
      I_Contact( #interlocksDB.SELECTING_PROG_FAULT_FB )
      I_Contact( #interlocksDB.RESET_SELECTION )
      Coil( #interlocksDB.SELECTED )
   END_RUNG
   RUNG wire#powerrail
      Contact( #interlocksDB.SELECTED )
   END_RUNG wire#w1
   // the same network as SCL:
   #interlocksDB.SELECTED := (#interlocksDB.SELECTING_PROG_DONE OR #interlocksDB.SELECTED) AND NOT #interlocksDB.SELECTING_PROG_FAULT_FB AND NOT #interlocksDB.RESET_SELECTION;
END_REGION

REGION Network 4: GENERAL CONDITIONS
   RUNG wire#powerrail
      I_Contact( #interlocksDB.SELECTING_PROG_FAULT_FB )
      I_Contact( #interlocksDB.SELECTING_PROG_FAULT_FB )
      I_Contact( #interlocksDB.SELECTED )
      I_Contact( #interlocksDB.SELECTING_PROG_DONE )
      I_Contact( #channelDB.E_ProgRunning )
      wire#w1
      { S7_Templates := "SrcType := Int" } EQ_Contact(in1 := #CH_MODE_GROUP, in2 := 1)
      I_Contact( "DB2001_MODES_GENERAL".MG1.STEP_BY_STEP.MODE_SELECTED )
      wire#w2
      Coil( #interlocksDB.GENERAL_CONDITIONS )
   END_RUNG
   RUNG wire#w1
      { S7_Templates := "SrcType := Int" } EQ_Contact(in1 := #CH_MODE_GROUP, in2 := 2)
      I_Contact( "DB2001_MODES_GENERAL".MG2.STEP_BY_STEP.MODE_SELECTED )
   END_RUNG wire#w2
   // the same network as SCL:
   #interlocksDB.GENERAL_CONDITIONS := NOT #interlocksDB.SELECTING_PROG_FAULT_FB AND NOT #interlocksDB.SELECTING_PROG_FAULT_FB AND NOT #interlocksDB.SELECTED AND NOT #interlocksDB.SELECTING_PROG_DONE AND NOT #channelDB.E_ProgRunning AND (((#CH_MODE_GROUP = 1) AND NOT "DB2001_MODES_GENERAL".MG1.STEP_BY_STEP.MODE_SELECTED) OR ((#CH_MODE_GROUP = 2) AND NOT "DB2001_MODES_GENERAL".MG2.STEP_BY_STEP.MODE_SELECTED));
END_REGION

REGION Network 5: REQUEST
   RUNG wire#powerrail
      Contact( #REQUEST )
      Contact( #interlocksDB.GENERAL_CONDITIONS )
      Coil( #interlocksDB.REQUEST )
   END_RUNG
   // the same network as SCL:
   #interlocksDB.REQUEST := #REQUEST AND #interlocksDB.GENERAL_CONDITIONS;
END_REGION

REGION Network 6: CALL FB7
   RUNG wire#powerrail
      #FB7_INSTANCE(Req := #interlocksDB.REQUEST, PIService := "LBP_PIServices".SELECT, Unit := #CHANNEL, Addr1 := #interlocksDB.Path, Addr2 := #interlocksDB.PName, Addr3 := NULL, Addr4 := NULL, WVar1 :=, WVar2 :=, WVar3 :=, WVar4 :=, WVar5 :=, WVar6 :=, WVar7 :=, WVar8 :=, WVar9 :=, WVar10 :=, WVar11 :=, WVar12 :=, WVar13 :=, WVar14 :=, WVar15 :=, WVar16 :=, Error => #interlocksDB.SELECTING_PROG_FAULT_FB, Done => #interlocksDB.SELECTING_PROG_DONE, State => #interlocksDB.SELECTING_STATUS)
   END_RUNG
   // the same network as SCL:
   #FB7_INSTANCE(Req := #interlocksDB.REQUEST,   // "LBP_ReqPIService"
                 PIService := "LBP_PIServices".SELECT,
                 Unit := #CHANNEL,
                 Addr1 := #interlocksDB.Path,
                 Addr2 := #interlocksDB.PName,
                 Addr3 := NULL,
                 Addr4 := NULL,
                 Error => #interlocksDB.SELECTING_PROG_FAULT_FB,
                 Done => #interlocksDB.SELECTING_PROG_DONE,
                 State => #interlocksDB.SELECTING_STATUS);
END_REGION

REGION Network 7: PROGRAM SELECTION ALARM / FAULT
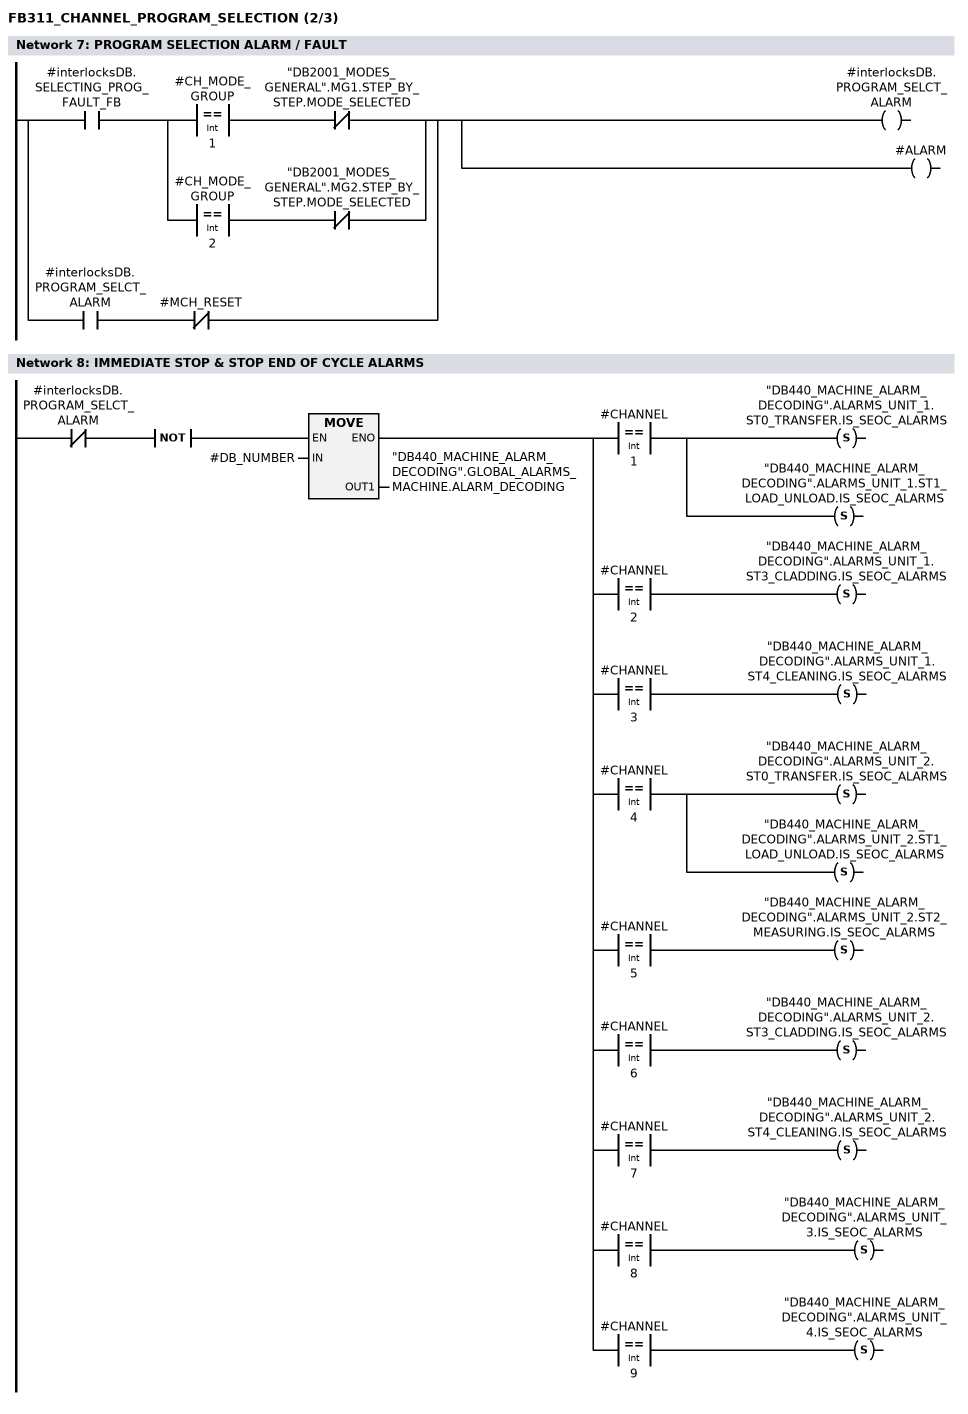
   RUNG wire#powerrail
      Contact( #interlocksDB.SELECTING_PROG_FAULT_FB )
      wire#w1
      { S7_Templates := "SrcType := Int" } EQ_Contact(in1 := #CH_MODE_GROUP, in2 := 1)
      I_Contact( "DB2001_MODES_GENERAL".MG1.STEP_BY_STEP.MODE_SELECTED )
      wire#w2
      Coil( #interlocksDB.PROGRAM_SELCT_ALARM )
   END_RUNG
   RUNG wire#w1
      { S7_Templates := "SrcType := Int" } EQ_Contact(in1 := #CH_MODE_GROUP, in2 := 2)
      I_Contact( "DB2001_MODES_GENERAL".MG2.STEP_BY_STEP.MODE_SELECTED )
   END_RUNG wire#w2
   RUNG wire#powerrail
      Contact( #interlocksDB.PROGRAM_SELCT_ALARM )
      I_Contact( #MCH_RESET )
   END_RUNG wire#w2
   RUNG wire#w2
      Coil( #ALARM )
   END_RUNG
   // the same network as SCL:
   #interlocksDB.PROGRAM_SELCT_ALARM := (#interlocksDB.SELECTING_PROG_FAULT_FB AND (((#CH_MODE_GROUP = 1) AND NOT "DB2001_MODES_GENERAL".MG1.STEP_BY_STEP.MODE_SELECTED) OR ((#CH_MODE_GROUP = 2) AND NOT "DB2001_MODES_GENERAL".MG2.STEP_BY_STEP.MODE_SELECTED))) OR (#interlocksDB.PROGRAM_SELCT_ALARM AND NOT #MCH_RESET);
   #ALARM := #interlocksDB.PROGRAM_SELCT_ALARM;
END_REGION

